// TIA Portal V17 export
// export: Created 2025-03-05T08:00:20.8649217Z, ExportSetting WithDefaults, DisplayName Totally Integrated Automation Portal, DisplayVersion V17 Update 8, DisplayName TIA Portal Openness, DisplayVersion V17 Update 8, DisplayName TIA Portal Version Control Interface, DisplayVersion V17, DisplayName SINAMICS Startdrive Advanced, DisplayVersion V17 SP2, DisplayName SINAMICS Startdrive G110M, G120, G120C, G120D, G120P, G115D, DisplayVersion V17 SP2, DisplayName SINAMICS Startdrive G130, G150, S120, S150, SINAMICS MV, S210, DisplayVersion V17 SP2, DisplayName STEP 7 Professional, DisplayVersion V17 Update 8, DisplayName SINUMERIK ONE STEP 7 Toolbox, DisplayVersion V17 Update 12, DisplayName SINUMERIK 840D sl STEP 7 Toolbox, DisplayVersion V17 Update 12, DisplayName STEP 7 Safety, DisplayVersion V17 Update 6, DisplayName WinCC Advanced, DisplayVersion V17 Update 8
FUNCTION "FC31_CLADDING_SPINDLES" : Void   // FC31, LAD
{ S7_Optimized_Access := 'FALSE' }
AUTHOR : ETXETAR
VERSION : 1.0
// stored: AutoNumber false, IsIECCheckEnabled false, SetENOAutomatically false, UDAEnableTagReadback false
   VAR_TEMP   // added for the SCL form of the ladder/FBD networks
      _w1 : Bool;
      _w2 : Bool;
   END_VAR
BEGIN

REGION Network 1: CALL FB31 SPINDLE C11
   // 2#0000_0001 OPTIONS 0 BIT 0 MEASURING SYSTEM 2 OPTION
   // 2#0000_0010 OPTIONS 0 BIT 1 BELT BROKEN OPTION
   // 2#0000_0100 OPTIONS 0 BIT 2 COOLING OPTION
   // 2#0000_1000 OPTIONS 0 BIT 3 MQL OR HP OPTION
   // 2#0001_0000 OPTIONS 0 BIT 4 ANALOG TEMPERATURE SENSOR OPTION
   // 2#0010_0000 OPTIONS 0 BIT 5 PTC TEMPERATURE SENSOR OPTION
   // 2#0100_0000 OPTIONS 0 BIT 6 TWIN KESSLER VPM READY OPTION
   // 2#1000_0000 OPTIONS 0 BIT 7 MPP SPINDLE OVERRIDE OPTION
   // 
   // 2#0000_0001 OPTIONS 1 BIT 0 SPARE OPTION
   // 2#0000_0010 OPTIONS 1 BIT 1 SPARE OPTION
   // 2#0000_0100 OPTIONS 1 BIT 2 SPARE OPTION
   // 2#0000_1000 OPTIONS 1 BIT 3 SPARE OPTION
   // 2#0001_0000 OPTIONS 1 BIT 4 SPARE OPTION
   // 2#0010_0000 OPTIONS 1 BIT 5 SPARE OPTION
   // 2#0100_0000 OPTIONS 1 BIT 6 SPARE OPTION
   // 2#1000_0000 OPTIONS 1 BIT 7 SPARE OPTION
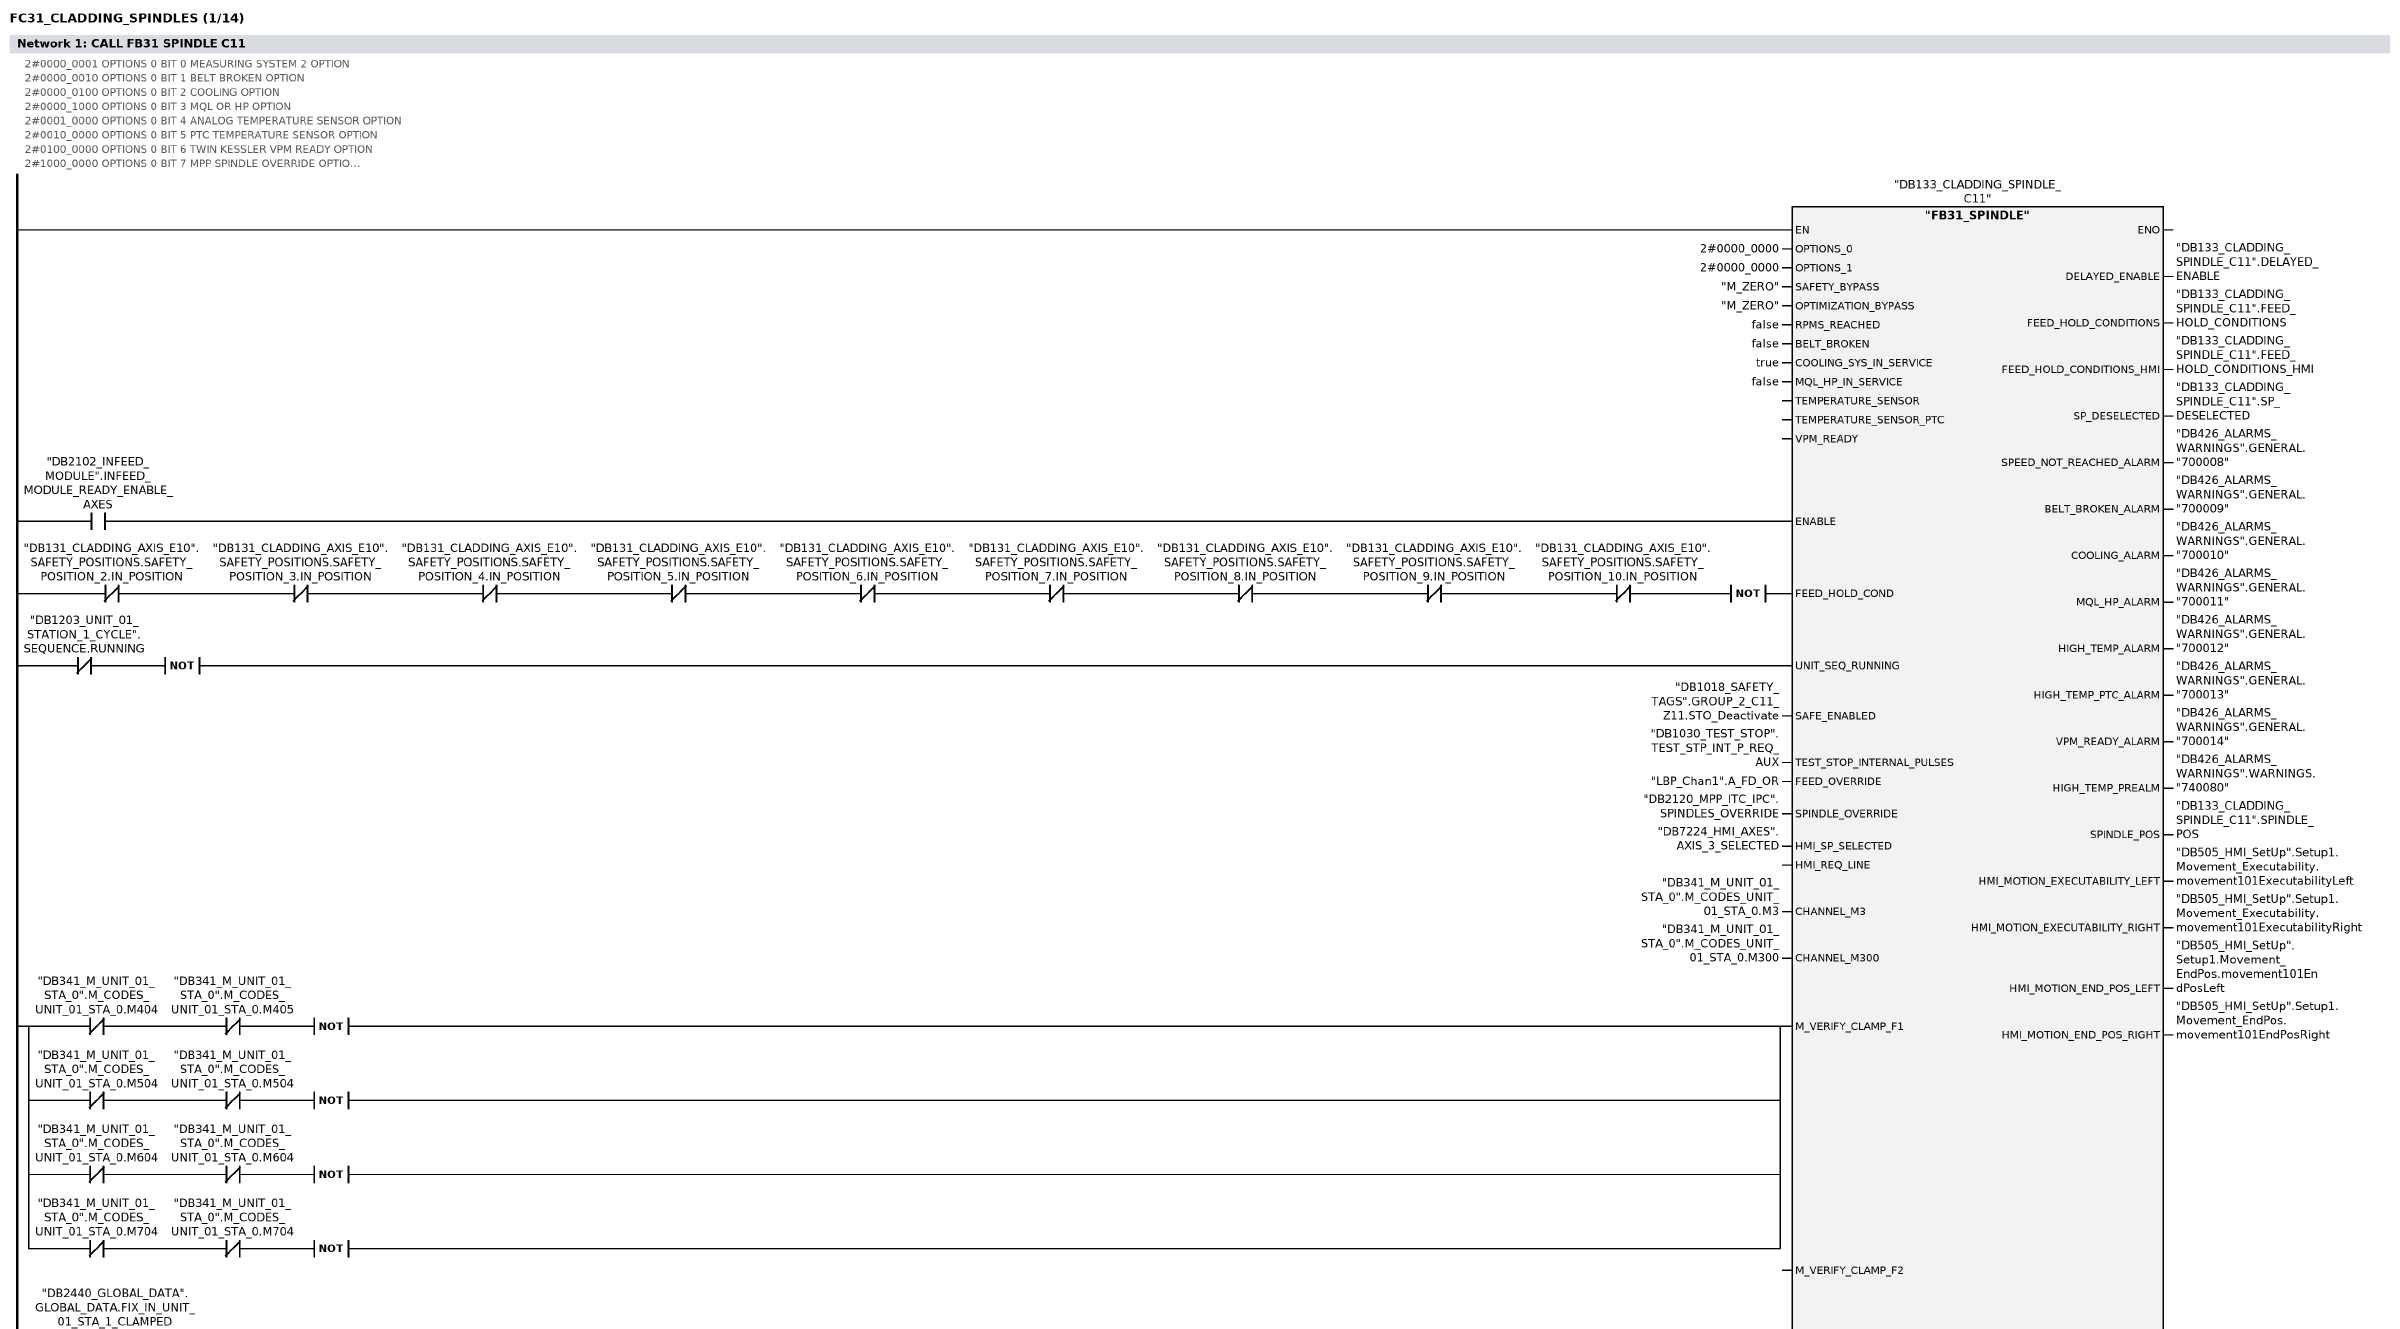
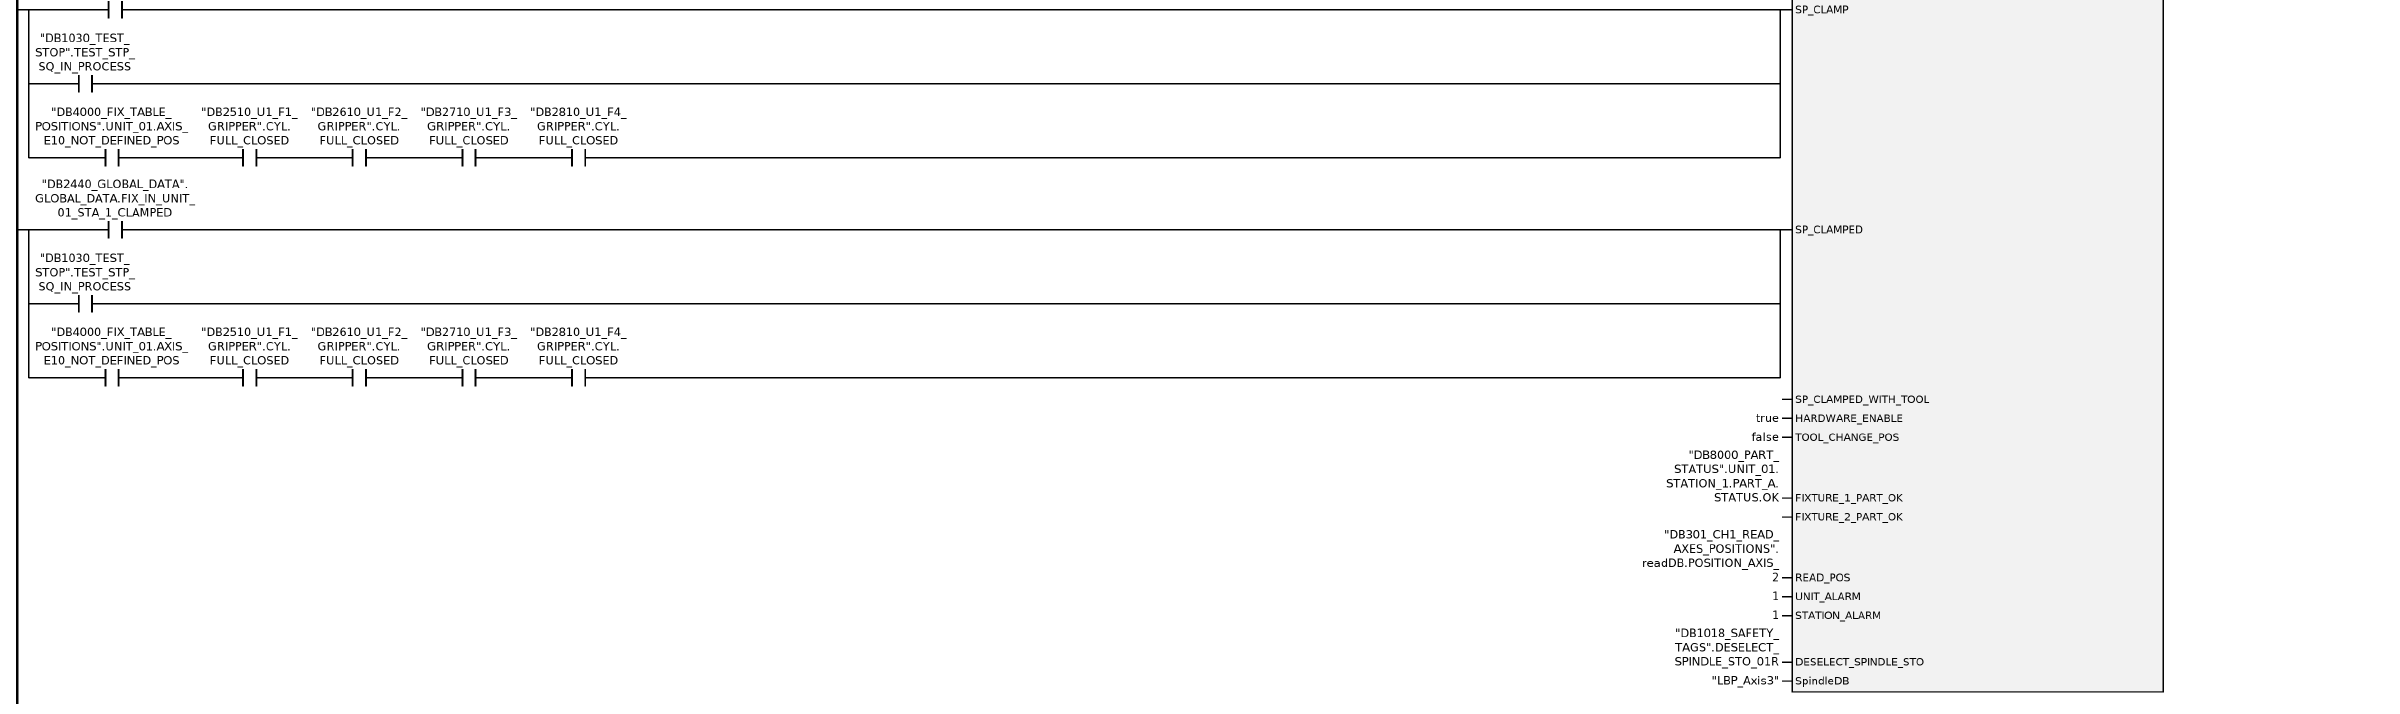
   RUNG wire#powerrail
      "DB133_CLADDING_SPINDLE_C11"(ENABLE := wire#w1, FEED_HOLD_COND := wire#w2, UNIT_SEQ_RUNNING := wire#w3, M_VERIFY_CLAMP_F1 := wire#w4, SP_CLAMP := wire#w5, SP_CLAMPED := wire#w6, OPTIONS_0 := 2#0000_0000, OPTIONS_1 := 2#0000_0000, SAFETY_BYPASS := "M_ZERO", OPTIMIZATION_BYPASS := "M_ZERO", RPMS_REACHED := false, BELT_BROKEN := false, COOLING_SYS_IN_SERVICE := true, MQL_HP_IN_SERVICE := false, TEMPERATURE_SENSOR :=, TEMPERATURE_SENSOR_PTC :=, VPM_READY :=, SAFE_ENABLED := "DB1018_SAFETY_TAGS".GROUP_2_C11_Z11.STO_Deactivate, TEST_STOP_INTERNAL_PULSES := "DB1030_TEST_STOP".TEST_STP_INT_P_REQ_AUX, FEED_OVERRIDE := "LBP_Chan1".A_FD_OR, SPINDLE_OVERRIDE := "DB2120_MPP_ITC_IPC".SPINDLES_OVERRIDE, HMI_SP_SELECTED := "DB7224_HMI_AXES".AXIS_3_SELECTED, HMI_REQ_LINE :=, CHANNEL_M3 := "DB341_M_UNIT_01_STA_0".M_CODES_UNIT_01_STA_0.M3, CHANNEL_M300 := "DB341_M_UNIT_01_STA_0".M_CODES_UNIT_01_STA_0.M300, M_VERIFY_CLAMP_F2 :=, SP_CLAMPED_WITH_TOOL :=, HARDWARE_ENABLE := true, TOOL_CHANGE_POS := false, FIXTURE_1_PART_OK := "DB8000_PART_STATUS".UNIT_01.STATION_1.PART_A.STATUS.OK, FIXTURE_2_PART_OK :=, READ_POS := "DB301_CH1_READ_AXES_POSITIONS".readDB.POSITION_AXIS_2, UNIT_ALARM := 1, STATION_ALARM := 1, DESELECT_SPINDLE_STO := "DB1018_SAFETY_TAGS".DESELECT_SPINDLE_STO_01R, SpindleDB := "LBP_Axis3", DELAYED_ENABLE => "DB133_CLADDING_SPINDLE_C11".DELAYED_ENABLE, FEED_HOLD_CONDITIONS => "DB133_CLADDING_SPINDLE_C11".FEED_HOLD_CONDITIONS, FEED_HOLD_CONDITIONS_HMI => "DB133_CLADDING_SPINDLE_C11".FEED_HOLD_CONDITIONS_HMI, SP_DESELECTED => "DB133_CLADDING_SPINDLE_C11".SP_DESELECTED, SPEED_NOT_REACHED_ALARM => "DB426_ALARMS_WARNINGS".GENERAL."700008", BELT_BROKEN_ALARM => "DB426_ALARMS_WARNINGS".GENERAL."700009", COOLING_ALARM => "DB426_ALARMS_WARNINGS".GENERAL."700010", MQL_HP_ALARM => "DB426_ALARMS_WARNINGS".GENERAL."700011", HIGH_TEMP_ALARM => "DB426_ALARMS_WARNINGS".GENERAL."700012", HIGH_TEMP_PTC_ALARM => "DB426_ALARMS_WARNINGS".GENERAL."700013", VPM_READY_ALARM => "DB426_ALARMS_WARNINGS".GENERAL."700014", HIGH_TEMP_PREALM => "DB426_ALARMS_WARNINGS".WARNINGS."740080", SPINDLE_POS => "DB133_CLADDING_SPINDLE_C11".SPINDLE_POS, HMI_MOTION_EXECUTABILITY_LEFT => "DB505_HMI_SetUp".Setup1.Movement_Executability.movement101ExecutabilityLeft, HMI_MOTION_EXECUTABILITY_RIGHT => "DB505_HMI_SetUp".Setup1.Movement_Executability.movement101ExecutabilityRight, HMI_MOTION_END_POS_LEFT => "DB505_HMI_SetUp".Setup1.Movement_EndPos.movement101EndPosLeft, HMI_MOTION_END_POS_RIGHT => "DB505_HMI_SetUp".Setup1.Movement_EndPos.movement101EndPosRight)
   END_RUNG
   RUNG wire#powerrail
      Contact( "DB2102_INFEED_MODULE".INFEED_MODULE_READY_ENABLE_AXES )
   END_RUNG wire#w1
   RUNG wire#powerrail
      I_Contact( "DB131_CLADDING_AXIS_E10".SAFETY_POSITIONS.SAFETY_POSITION_2.IN_POSITION )
      I_Contact( "DB131_CLADDING_AXIS_E10".SAFETY_POSITIONS.SAFETY_POSITION_3.IN_POSITION )
      I_Contact( "DB131_CLADDING_AXIS_E10".SAFETY_POSITIONS.SAFETY_POSITION_4.IN_POSITION )
      I_Contact( "DB131_CLADDING_AXIS_E10".SAFETY_POSITIONS.SAFETY_POSITION_5.IN_POSITION )
      I_Contact( "DB131_CLADDING_AXIS_E10".SAFETY_POSITIONS.SAFETY_POSITION_6.IN_POSITION )
      I_Contact( "DB131_CLADDING_AXIS_E10".SAFETY_POSITIONS.SAFETY_POSITION_7.IN_POSITION )
      I_Contact( "DB131_CLADDING_AXIS_E10".SAFETY_POSITIONS.SAFETY_POSITION_8.IN_POSITION )
      I_Contact( "DB131_CLADDING_AXIS_E10".SAFETY_POSITIONS.SAFETY_POSITION_9.IN_POSITION )
      I_Contact( "DB131_CLADDING_AXIS_E10".SAFETY_POSITIONS.SAFETY_POSITION_10.IN_POSITION )
      Not()
   END_RUNG wire#w2
   RUNG wire#powerrail
      I_Contact( "DB1203_UNIT_01_STATION_1_CYCLE".SEQUENCE.RUNNING )
      Not()
   END_RUNG wire#w3
   RUNG wire#powerrail
      I_Contact( "DB341_M_UNIT_01_STA_0".M_CODES_UNIT_01_STA_0.M404 )
      I_Contact( "DB341_M_UNIT_01_STA_0".M_CODES_UNIT_01_STA_0.M405 )
      Not()
   END_RUNG wire#w4
   RUNG wire#powerrail
      I_Contact( "DB341_M_UNIT_01_STA_0".M_CODES_UNIT_01_STA_0.M504 )
      I_Contact( "DB341_M_UNIT_01_STA_0".M_CODES_UNIT_01_STA_0.M504 )
      Not()
   END_RUNG wire#w4
   RUNG wire#powerrail
      I_Contact( "DB341_M_UNIT_01_STA_0".M_CODES_UNIT_01_STA_0.M604 )
      I_Contact( "DB341_M_UNIT_01_STA_0".M_CODES_UNIT_01_STA_0.M604 )
      Not()
   END_RUNG wire#w4
   RUNG wire#powerrail
      I_Contact( "DB341_M_UNIT_01_STA_0".M_CODES_UNIT_01_STA_0.M704 )
      I_Contact( "DB341_M_UNIT_01_STA_0".M_CODES_UNIT_01_STA_0.M704 )
      Not()
   END_RUNG wire#w4
   RUNG wire#powerrail
      Contact( "DB2440_GLOBAL_DATA".GLOBAL_DATA.FIX_IN_UNIT_01_STA_1_CLAMPED )
   END_RUNG wire#w5
   RUNG wire#powerrail
      Contact( "DB1030_TEST_STOP".TEST_STP_SQ_IN_PROCESS )
   END_RUNG wire#w5
   RUNG wire#powerrail
      Contact( "DB4000_FIX_TABLE_POSITIONS".UNIT_01.AXIS_E10_NOT_DEFINED_POS )
      Contact( "DB2510_U1_F1_GRIPPER".CYL.FULL_CLOSED )
      Contact( "DB2610_U1_F2_GRIPPER".CYL.FULL_CLOSED )
      Contact( "DB2710_U1_F3_GRIPPER".CYL.FULL_CLOSED )
      Contact( "DB2810_U1_F4_GRIPPER".CYL.FULL_CLOSED )
   END_RUNG wire#w5
   RUNG wire#powerrail
      Contact( "DB2440_GLOBAL_DATA".GLOBAL_DATA.FIX_IN_UNIT_01_STA_1_CLAMPED )
   END_RUNG wire#w6
   RUNG wire#powerrail
      Contact( "DB1030_TEST_STOP".TEST_STP_SQ_IN_PROCESS )
   END_RUNG wire#w6
   RUNG wire#powerrail
      Contact( "DB4000_FIX_TABLE_POSITIONS".UNIT_01.AXIS_E10_NOT_DEFINED_POS )
      Contact( "DB2510_U1_F1_GRIPPER".CYL.FULL_CLOSED )
      Contact( "DB2610_U1_F2_GRIPPER".CYL.FULL_CLOSED )
      Contact( "DB2710_U1_F3_GRIPPER".CYL.FULL_CLOSED )
      Contact( "DB2810_U1_F4_GRIPPER".CYL.FULL_CLOSED )
   END_RUNG wire#w6
   // the same network as SCL:
   "DB133_CLADDING_SPINDLE_C11"(OPTIONS_0 := 2#0000_0000,   // "FB31_SPINDLE"
                           OPTIONS_1 := 2#0000_0000,
                           SAFETY_BYPASS := "M_ZERO",
                           OPTIMIZATION_BYPASS := "M_ZERO",
                           RPMS_REACHED := false,
                           BELT_BROKEN := false,
                           COOLING_SYS_IN_SERVICE := true,
                           MQL_HP_IN_SERVICE := false,
                           ENABLE := "DB2102_INFEED_MODULE".INFEED_MODULE_READY_ENABLE_AXES,
                           FEED_HOLD_COND := NOT (NOT "DB131_CLADDING_AXIS_E10".SAFETY_POSITIONS.SAFETY_POSITION_2.IN_POSITION AND NOT "DB131_CLADDING_AXIS_E10".SAFETY_POSITIONS.SAFETY_POSITION_3.IN_POSITION AND NOT "DB131_CLADDING_AXIS_E10".SAFETY_POSITIONS.SAFETY_POSITION_4.IN_POSITION AND NOT "DB131_CLADDING_AXIS_E10".SAFETY_POSITIONS.SAFETY_POSITION_5.IN_POSITION AND NOT "DB131_CLADDING_AXIS_E10".SAFETY_POSITIONS.SAFETY_POSITION_6.IN_POSITION AND NOT "DB131_CLADDING_AXIS_E10".SAFETY_POSITIONS.SAFETY_POSITION_7.IN_POSITION AND NOT "DB131_CLADDING_AXIS_E10".SAFETY_POSITIONS.SAFETY_POSITION_8.IN_POSITION AND NOT "DB131_CLADDING_AXIS_E10".SAFETY_POSITIONS.SAFETY_POSITION_9.IN_POSITION AND NOT "DB131_CLADDING_AXIS_E10".SAFETY_POSITIONS.SAFETY_POSITION_10.IN_POSITION),
                           UNIT_SEQ_RUNNING := NOT (NOT "DB1203_UNIT_01_STATION_1_CYCLE".SEQUENCE.RUNNING),
                           SAFE_ENABLED := "DB1018_SAFETY_TAGS".GROUP_2_C11_Z11.STO_Deactivate,
                           TEST_STOP_INTERNAL_PULSES := "DB1030_TEST_STOP".TEST_STP_INT_P_REQ_AUX,
                           FEED_OVERRIDE := "LBP_Chan1".A_FD_OR,
                           SPINDLE_OVERRIDE := "DB2120_MPP_ITC_IPC".SPINDLES_OVERRIDE,
                           HMI_SP_SELECTED := "DB7224_HMI_AXES".AXIS_3_SELECTED,
                           CHANNEL_M3 := "DB341_M_UNIT_01_STA_0".M_CODES_UNIT_01_STA_0.M3,
                           CHANNEL_M300 := "DB341_M_UNIT_01_STA_0".M_CODES_UNIT_01_STA_0.M300,
                           M_VERIFY_CLAMP_F1 := NOT (NOT "DB341_M_UNIT_01_STA_0".M_CODES_UNIT_01_STA_0.M404 AND NOT "DB341_M_UNIT_01_STA_0".M_CODES_UNIT_01_STA_0.M405) OR NOT (NOT "DB341_M_UNIT_01_STA_0".M_CODES_UNIT_01_STA_0.M504 AND NOT "DB341_M_UNIT_01_STA_0".M_CODES_UNIT_01_STA_0.M504) OR NOT (NOT "DB341_M_UNIT_01_STA_0".M_CODES_UNIT_01_STA_0.M604 AND NOT "DB341_M_UNIT_01_STA_0".M_CODES_UNIT_01_STA_0.M604) OR NOT (NOT "DB341_M_UNIT_01_STA_0".M_CODES_UNIT_01_STA_0.M704 AND NOT "DB341_M_UNIT_01_STA_0".M_CODES_UNIT_01_STA_0.M704),
                           SP_CLAMP := "DB2440_GLOBAL_DATA".GLOBAL_DATA.FIX_IN_UNIT_01_STA_1_CLAMPED OR "DB1030_TEST_STOP".TEST_STP_SQ_IN_PROCESS OR ("DB4000_FIX_TABLE_POSITIONS".UNIT_01.AXIS_E10_NOT_DEFINED_POS AND "DB2510_U1_F1_GRIPPER".CYL.FULL_CLOSED AND "DB2610_U1_F2_GRIPPER".CYL.FULL_CLOSED AND "DB2710_U1_F3_GRIPPER".CYL.FULL_CLOSED AND "DB2810_U1_F4_GRIPPER".CYL.FULL_CLOSED),
                           SP_CLAMPED := "DB2440_GLOBAL_DATA".GLOBAL_DATA.FIX_IN_UNIT_01_STA_1_CLAMPED OR "DB1030_TEST_STOP".TEST_STP_SQ_IN_PROCESS OR ("DB4000_FIX_TABLE_POSITIONS".UNIT_01.AXIS_E10_NOT_DEFINED_POS AND "DB2510_U1_F1_GRIPPER".CYL.FULL_CLOSED AND "DB2610_U1_F2_GRIPPER".CYL.FULL_CLOSED AND "DB2710_U1_F3_GRIPPER".CYL.FULL_CLOSED AND "DB2810_U1_F4_GRIPPER".CYL.FULL_CLOSED),
                           HARDWARE_ENABLE := true,
                           TOOL_CHANGE_POS := false,
                           FIXTURE_1_PART_OK := "DB8000_PART_STATUS".UNIT_01.STATION_1.PART_A.STATUS.OK,
                           READ_POS := "DB301_CH1_READ_AXES_POSITIONS".readDB.POSITION_AXIS_2,
                           UNIT_ALARM := 1,
                           STATION_ALARM := 1,
                           DESELECT_SPINDLE_STO := "DB1018_SAFETY_TAGS".DESELECT_SPINDLE_STO_01R,
                           SpindleDB := "LBP_Axis3",
                           DELAYED_ENABLE => "DB133_CLADDING_SPINDLE_C11".DELAYED_ENABLE,
                           FEED_HOLD_CONDITIONS => "DB133_CLADDING_SPINDLE_C11".FEED_HOLD_CONDITIONS,
                           FEED_HOLD_CONDITIONS_HMI => "DB133_CLADDING_SPINDLE_C11".FEED_HOLD_CONDITIONS_HMI,
                           SP_DESELECTED => "DB133_CLADDING_SPINDLE_C11".SP_DESELECTED,
                           SPEED_NOT_REACHED_ALARM => "DB426_ALARMS_WARNINGS".GENERAL."700008",
                           BELT_BROKEN_ALARM => "DB426_ALARMS_WARNINGS".GENERAL."700009",
                           COOLING_ALARM => "DB426_ALARMS_WARNINGS".GENERAL."700010",
                           MQL_HP_ALARM => "DB426_ALARMS_WARNINGS".GENERAL."700011",
                           HIGH_TEMP_ALARM => "DB426_ALARMS_WARNINGS".GENERAL."700012",
                           HIGH_TEMP_PTC_ALARM => "DB426_ALARMS_WARNINGS".GENERAL."700013",
                           VPM_READY_ALARM => "DB426_ALARMS_WARNINGS".GENERAL."700014",
                           HIGH_TEMP_PREALM => "DB426_ALARMS_WARNINGS".WARNINGS."740080",
                           SPINDLE_POS => "DB133_CLADDING_SPINDLE_C11".SPINDLE_POS,
                           HMI_MOTION_EXECUTABILITY_LEFT => "DB505_HMI_SetUp".Setup1.Movement_Executability.movement101ExecutabilityLeft,
                           HMI_MOTION_EXECUTABILITY_RIGHT => "DB505_HMI_SetUp".Setup1.Movement_Executability.movement101ExecutabilityRight,
                           HMI_MOTION_END_POS_LEFT => "DB505_HMI_SetUp".Setup1.Movement_EndPos.movement101EndPosLeft,
                           HMI_MOTION_END_POS_RIGHT => "DB505_HMI_SetUp".Setup1.Movement_EndPos.movement101EndPosRight);
END_REGION

REGION Network 2: SPINDLE C11 OPERATOR HELP
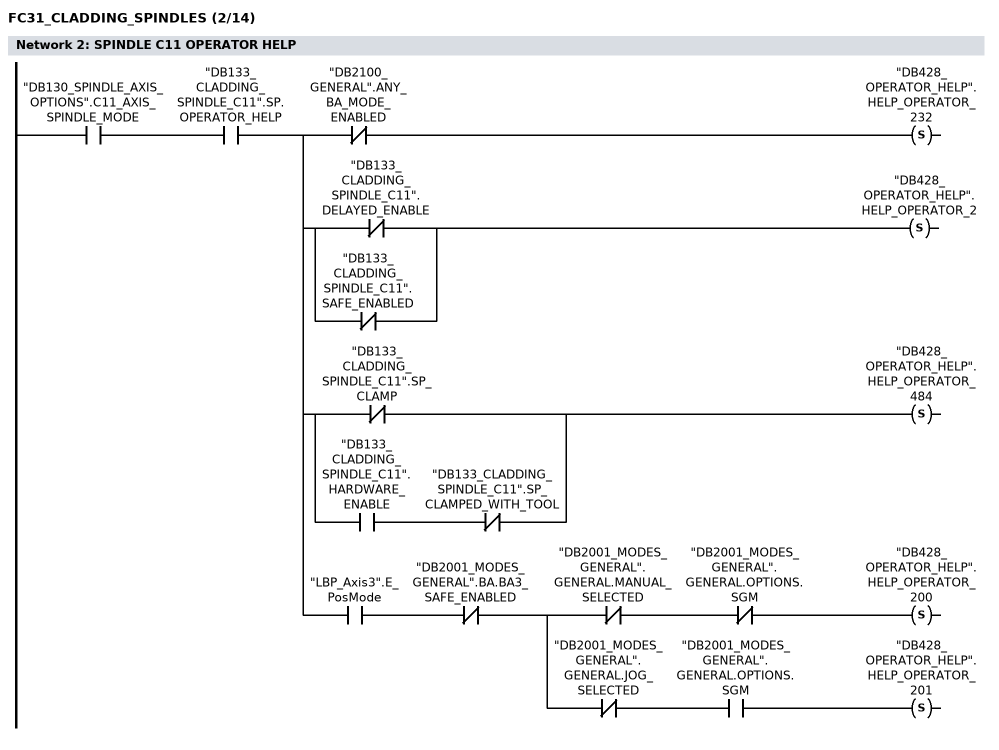
   RUNG wire#powerrail
      Contact( "DB130_SPINDLE_AXIS_OPTIONS".C11_AXIS_SPINDLE_MODE )
      Contact( "DB133_CLADDING_SPINDLE_C11".SP.OPERATOR_HELP )
      wire#w1
      I_Contact( "DB2100_GENERAL".ANY_BA_MODE_ENABLED )
      S_Coil( "DB428_OPERATOR_HELP".HELP_OPERATOR_232 )
   END_RUNG
   RUNG wire#w1
      I_Contact( "DB133_CLADDING_SPINDLE_C11".DELAYED_ENABLE )
      wire#w2
      S_Coil( "DB428_OPERATOR_HELP".HELP_OPERATOR_2 )
   END_RUNG
   RUNG wire#w1
      I_Contact( "DB133_CLADDING_SPINDLE_C11".SAFE_ENABLED )
   END_RUNG wire#w2
   RUNG wire#w1
      I_Contact( "DB133_CLADDING_SPINDLE_C11".SP_CLAMP )
      wire#w3
      S_Coil( "DB428_OPERATOR_HELP".HELP_OPERATOR_484 )
   END_RUNG
   RUNG wire#w1
      Contact( "DB133_CLADDING_SPINDLE_C11".HARDWARE_ENABLE )
      I_Contact( "DB133_CLADDING_SPINDLE_C11".SP_CLAMPED_WITH_TOOL )
   END_RUNG wire#w3
   RUNG wire#w1
      Contact( "LBP_Axis3".E_PosMode )
      I_Contact( "DB2001_MODES_GENERAL".BA.BA3_SAFE_ENABLED )
      wire#w4
      I_Contact( "DB2001_MODES_GENERAL".GENERAL.MANUAL_SELECTED )
      I_Contact( "DB2001_MODES_GENERAL".GENERAL.OPTIONS.SGM )
      S_Coil( "DB428_OPERATOR_HELP".HELP_OPERATOR_200 )
   END_RUNG
   RUNG wire#w4
      I_Contact( "DB2001_MODES_GENERAL".GENERAL.JOG_SELECTED )
      Contact( "DB2001_MODES_GENERAL".GENERAL.OPTIONS.SGM )
      S_Coil( "DB428_OPERATOR_HELP".HELP_OPERATOR_201 )
   END_RUNG
   // the same network as SCL:
   #_w1 := "DB130_SPINDLE_AXIS_OPTIONS".C11_AXIS_SPINDLE_MODE AND "DB133_CLADDING_SPINDLE_C11".SP.OPERATOR_HELP;
   IF #_w1 AND NOT "DB2100_GENERAL".ANY_BA_MODE_ENABLED THEN
       "DB428_OPERATOR_HELP".HELP_OPERATOR_232 := TRUE;
   END_IF;
   IF #_w1 AND (NOT "DB133_CLADDING_SPINDLE_C11".DELAYED_ENABLE OR NOT "DB133_CLADDING_SPINDLE_C11".SAFE_ENABLED) THEN
       "DB428_OPERATOR_HELP".HELP_OPERATOR_2 := TRUE;
   END_IF;
   IF #_w1 AND (NOT "DB133_CLADDING_SPINDLE_C11".SP_CLAMP OR ("DB133_CLADDING_SPINDLE_C11".HARDWARE_ENABLE AND NOT "DB133_CLADDING_SPINDLE_C11".SP_CLAMPED_WITH_TOOL)) THEN
       "DB428_OPERATOR_HELP".HELP_OPERATOR_484 := TRUE;
   END_IF;
   #_w2 := #_w1 AND "LBP_Axis3".E_PosMode AND NOT "DB2001_MODES_GENERAL".BA.BA3_SAFE_ENABLED;
   IF #_w2 AND NOT "DB2001_MODES_GENERAL".GENERAL.MANUAL_SELECTED AND NOT "DB2001_MODES_GENERAL".GENERAL.OPTIONS.SGM THEN
       "DB428_OPERATOR_HELP".HELP_OPERATOR_200 := TRUE;
   END_IF;
   IF #_w2 AND NOT "DB2001_MODES_GENERAL".GENERAL.JOG_SELECTED AND "DB2001_MODES_GENERAL".GENERAL.OPTIONS.SGM THEN
       "DB428_OPERATOR_HELP".HELP_OPERATOR_201 := TRUE;
   END_IF;
END_REGION

REGION Network 3: CALL FB31 SPINDLE C12
   // 2#0000_0001 OPTIONS 0 BIT 0 MEASURING SYSTEM 2 OPTION
   // 2#0000_0010 OPTIONS 0 BIT 1 BELT BROKEN OPTION
   // 2#0000_0100 OPTIONS 0 BIT 2 COOLING OPTION
   // 2#0000_1000 OPTIONS 0 BIT 3 MQL OR HP OPTION
   // 2#0001_0000 OPTIONS 0 BIT 4 ANALOG TEMPERATURE SENSOR OPTION
   // 2#0010_0000 OPTIONS 0 BIT 5 PTC TEMPERATURE SENSOR OPTION
   // 2#0100_0000 OPTIONS 0 BIT 6 TWIN KESSLER VPM READY OPTION
   // 2#1000_0000 OPTIONS 0 BIT 7 MPP SPINDLE OVERRIDE OPTION
   // 
   // 2#0000_0001 OPTIONS 1 BIT 0 SPARE OPTION
   // 2#0000_0010 OPTIONS 1 BIT 1 SPARE OPTION
   // 2#0000_0100 OPTIONS 1 BIT 2 SPARE OPTION
   // 2#0000_1000 OPTIONS 1 BIT 3 SPARE OPTION
   // 2#0001_0000 OPTIONS 1 BIT 4 SPARE OPTION
   // 2#0010_0000 OPTIONS 1 BIT 5 SPARE OPTION
   // 2#0100_0000 OPTIONS 1 BIT 6 SPARE OPTION
   // 2#1000_0000 OPTIONS 1 BIT 7 SPARE OPTION
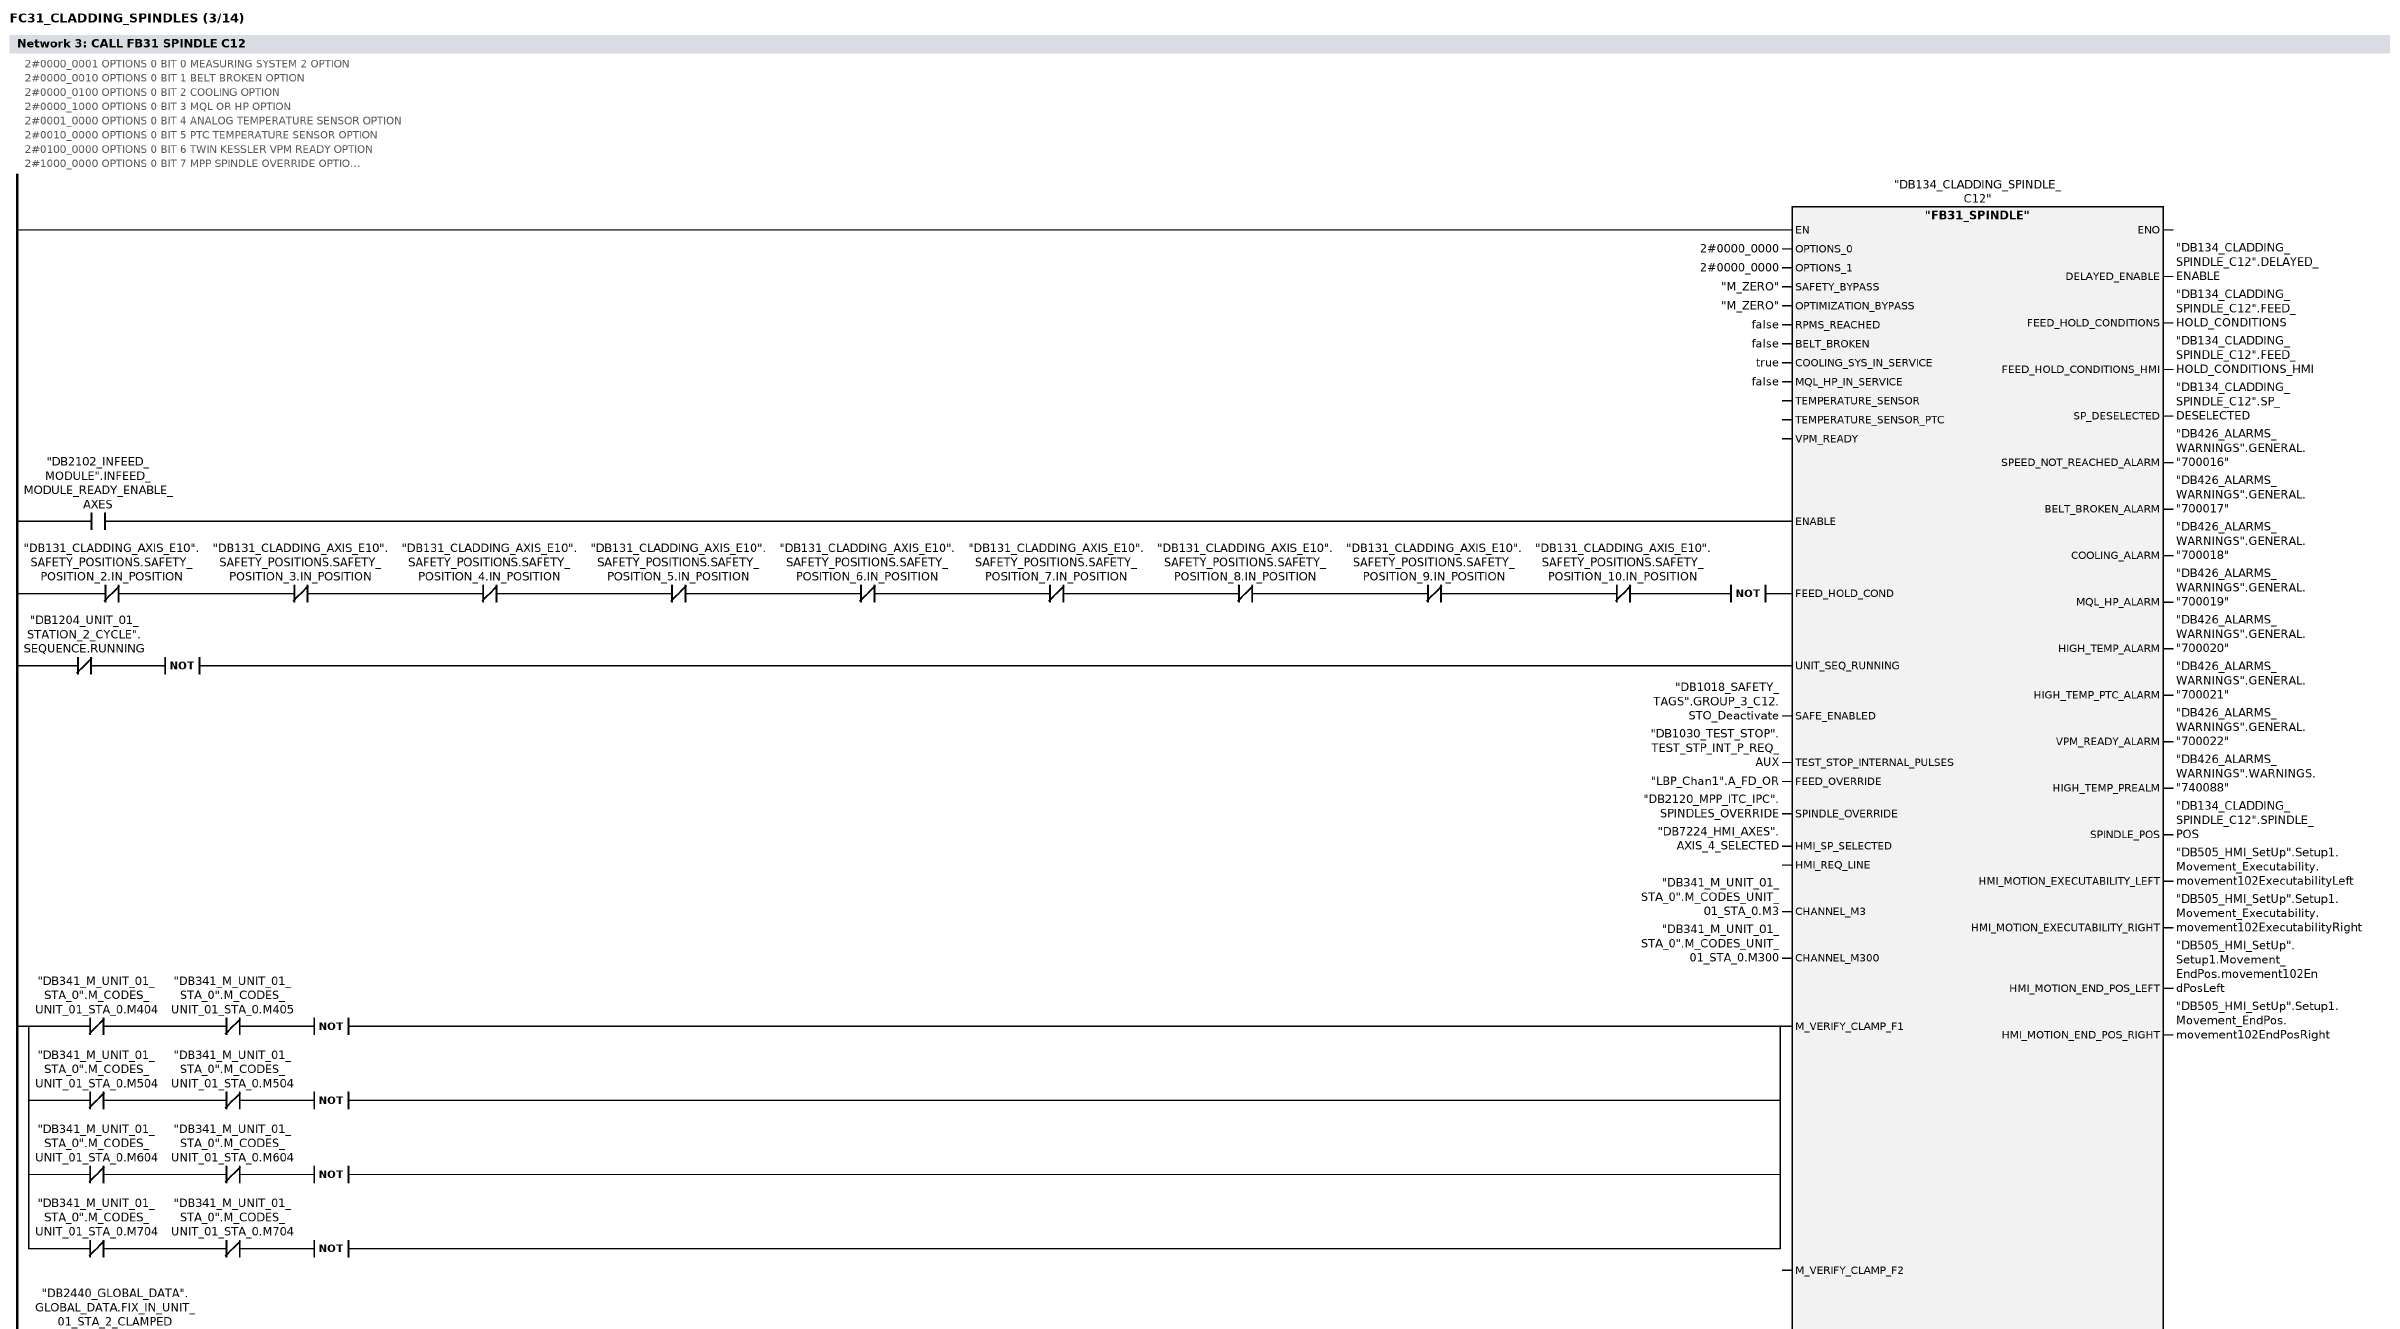
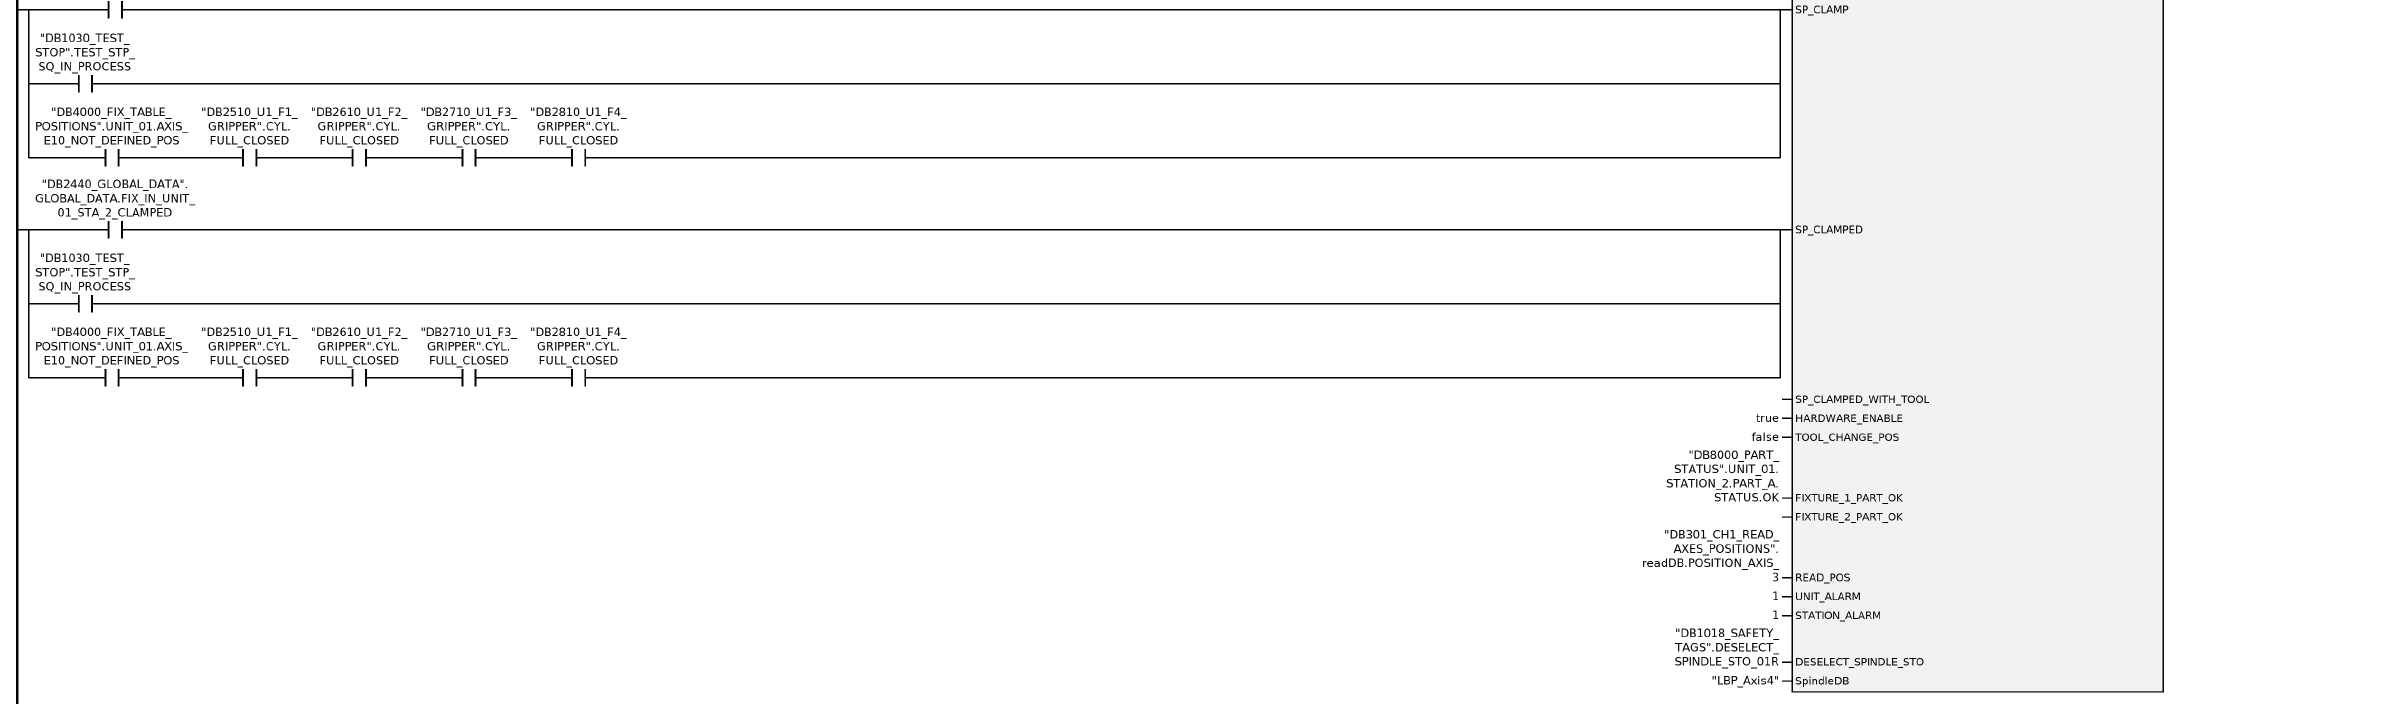
   RUNG wire#powerrail
      "DB134_CLADDING_SPINDLE_C12"(ENABLE := wire#w1, FEED_HOLD_COND := wire#w2, UNIT_SEQ_RUNNING := wire#w3, M_VERIFY_CLAMP_F1 := wire#w4, SP_CLAMP := wire#w5, SP_CLAMPED := wire#w6, OPTIONS_0 := 2#0000_0000, OPTIONS_1 := 2#0000_0000, SAFETY_BYPASS := "M_ZERO", OPTIMIZATION_BYPASS := "M_ZERO", RPMS_REACHED := false, BELT_BROKEN := false, COOLING_SYS_IN_SERVICE := true, MQL_HP_IN_SERVICE := false, TEMPERATURE_SENSOR :=, TEMPERATURE_SENSOR_PTC :=, VPM_READY :=, SAFE_ENABLED := "DB1018_SAFETY_TAGS".GROUP_3_C12.STO_Deactivate, TEST_STOP_INTERNAL_PULSES := "DB1030_TEST_STOP".TEST_STP_INT_P_REQ_AUX, FEED_OVERRIDE := "LBP_Chan1".A_FD_OR, SPINDLE_OVERRIDE := "DB2120_MPP_ITC_IPC".SPINDLES_OVERRIDE, HMI_SP_SELECTED := "DB7224_HMI_AXES".AXIS_4_SELECTED, HMI_REQ_LINE :=, CHANNEL_M3 := "DB341_M_UNIT_01_STA_0".M_CODES_UNIT_01_STA_0.M3, CHANNEL_M300 := "DB341_M_UNIT_01_STA_0".M_CODES_UNIT_01_STA_0.M300, M_VERIFY_CLAMP_F2 :=, SP_CLAMPED_WITH_TOOL :=, HARDWARE_ENABLE := true, TOOL_CHANGE_POS := false, FIXTURE_1_PART_OK := "DB8000_PART_STATUS".UNIT_01.STATION_2.PART_A.STATUS.OK, FIXTURE_2_PART_OK :=, READ_POS := "DB301_CH1_READ_AXES_POSITIONS".readDB.POSITION_AXIS_3, UNIT_ALARM := 1, STATION_ALARM := 1, DESELECT_SPINDLE_STO := "DB1018_SAFETY_TAGS".DESELECT_SPINDLE_STO_01R, SpindleDB := "LBP_Axis4", DELAYED_ENABLE => "DB134_CLADDING_SPINDLE_C12".DELAYED_ENABLE, FEED_HOLD_CONDITIONS => "DB134_CLADDING_SPINDLE_C12".FEED_HOLD_CONDITIONS, FEED_HOLD_CONDITIONS_HMI => "DB134_CLADDING_SPINDLE_C12".FEED_HOLD_CONDITIONS_HMI, SP_DESELECTED => "DB134_CLADDING_SPINDLE_C12".SP_DESELECTED, SPEED_NOT_REACHED_ALARM => "DB426_ALARMS_WARNINGS".GENERAL."700016", BELT_BROKEN_ALARM => "DB426_ALARMS_WARNINGS".GENERAL."700017", COOLING_ALARM => "DB426_ALARMS_WARNINGS".GENERAL."700018", MQL_HP_ALARM => "DB426_ALARMS_WARNINGS".GENERAL."700019", HIGH_TEMP_ALARM => "DB426_ALARMS_WARNINGS".GENERAL."700020", HIGH_TEMP_PTC_ALARM => "DB426_ALARMS_WARNINGS".GENERAL."700021", VPM_READY_ALARM => "DB426_ALARMS_WARNINGS".GENERAL."700022", HIGH_TEMP_PREALM => "DB426_ALARMS_WARNINGS".WARNINGS."740088", SPINDLE_POS => "DB134_CLADDING_SPINDLE_C12".SPINDLE_POS, HMI_MOTION_EXECUTABILITY_LEFT => "DB505_HMI_SetUp".Setup1.Movement_Executability.movement102ExecutabilityLeft, HMI_MOTION_EXECUTABILITY_RIGHT => "DB505_HMI_SetUp".Setup1.Movement_Executability.movement102ExecutabilityRight, HMI_MOTION_END_POS_LEFT => "DB505_HMI_SetUp".Setup1.Movement_EndPos.movement102EndPosLeft, HMI_MOTION_END_POS_RIGHT => "DB505_HMI_SetUp".Setup1.Movement_EndPos.movement102EndPosRight)
   END_RUNG
   RUNG wire#powerrail
      Contact( "DB2102_INFEED_MODULE".INFEED_MODULE_READY_ENABLE_AXES )
   END_RUNG wire#w1
   RUNG wire#powerrail
      I_Contact( "DB131_CLADDING_AXIS_E10".SAFETY_POSITIONS.SAFETY_POSITION_2.IN_POSITION )
      I_Contact( "DB131_CLADDING_AXIS_E10".SAFETY_POSITIONS.SAFETY_POSITION_3.IN_POSITION )
      I_Contact( "DB131_CLADDING_AXIS_E10".SAFETY_POSITIONS.SAFETY_POSITION_4.IN_POSITION )
      I_Contact( "DB131_CLADDING_AXIS_E10".SAFETY_POSITIONS.SAFETY_POSITION_5.IN_POSITION )
      I_Contact( "DB131_CLADDING_AXIS_E10".SAFETY_POSITIONS.SAFETY_POSITION_6.IN_POSITION )
      I_Contact( "DB131_CLADDING_AXIS_E10".SAFETY_POSITIONS.SAFETY_POSITION_7.IN_POSITION )
      I_Contact( "DB131_CLADDING_AXIS_E10".SAFETY_POSITIONS.SAFETY_POSITION_8.IN_POSITION )
      I_Contact( "DB131_CLADDING_AXIS_E10".SAFETY_POSITIONS.SAFETY_POSITION_9.IN_POSITION )
      I_Contact( "DB131_CLADDING_AXIS_E10".SAFETY_POSITIONS.SAFETY_POSITION_10.IN_POSITION )
      Not()
   END_RUNG wire#w2
   RUNG wire#powerrail
      I_Contact( "DB1204_UNIT_01_STATION_2_CYCLE".SEQUENCE.RUNNING )
      Not()
   END_RUNG wire#w3
   RUNG wire#powerrail
      I_Contact( "DB341_M_UNIT_01_STA_0".M_CODES_UNIT_01_STA_0.M404 )
      I_Contact( "DB341_M_UNIT_01_STA_0".M_CODES_UNIT_01_STA_0.M405 )
      Not()
   END_RUNG wire#w4
   RUNG wire#powerrail
      I_Contact( "DB341_M_UNIT_01_STA_0".M_CODES_UNIT_01_STA_0.M504 )
      I_Contact( "DB341_M_UNIT_01_STA_0".M_CODES_UNIT_01_STA_0.M504 )
      Not()
   END_RUNG wire#w4
   RUNG wire#powerrail
      I_Contact( "DB341_M_UNIT_01_STA_0".M_CODES_UNIT_01_STA_0.M604 )
      I_Contact( "DB341_M_UNIT_01_STA_0".M_CODES_UNIT_01_STA_0.M604 )
      Not()
   END_RUNG wire#w4
   RUNG wire#powerrail
      I_Contact( "DB341_M_UNIT_01_STA_0".M_CODES_UNIT_01_STA_0.M704 )
      I_Contact( "DB341_M_UNIT_01_STA_0".M_CODES_UNIT_01_STA_0.M704 )
      Not()
   END_RUNG wire#w4
   RUNG wire#powerrail
      Contact( "DB2440_GLOBAL_DATA".GLOBAL_DATA.FIX_IN_UNIT_01_STA_2_CLAMPED )
   END_RUNG wire#w5
   RUNG wire#powerrail
      Contact( "DB1030_TEST_STOP".TEST_STP_SQ_IN_PROCESS )
   END_RUNG wire#w5
   RUNG wire#powerrail
      Contact( "DB4000_FIX_TABLE_POSITIONS".UNIT_01.AXIS_E10_NOT_DEFINED_POS )
      Contact( "DB2510_U1_F1_GRIPPER".CYL.FULL_CLOSED )
      Contact( "DB2610_U1_F2_GRIPPER".CYL.FULL_CLOSED )
      Contact( "DB2710_U1_F3_GRIPPER".CYL.FULL_CLOSED )
      Contact( "DB2810_U1_F4_GRIPPER".CYL.FULL_CLOSED )
   END_RUNG wire#w5
   RUNG wire#powerrail
      Contact( "DB2440_GLOBAL_DATA".GLOBAL_DATA.FIX_IN_UNIT_01_STA_2_CLAMPED )
   END_RUNG wire#w6
   RUNG wire#powerrail
      Contact( "DB1030_TEST_STOP".TEST_STP_SQ_IN_PROCESS )
   END_RUNG wire#w6
   RUNG wire#powerrail
      Contact( "DB4000_FIX_TABLE_POSITIONS".UNIT_01.AXIS_E10_NOT_DEFINED_POS )
      Contact( "DB2510_U1_F1_GRIPPER".CYL.FULL_CLOSED )
      Contact( "DB2610_U1_F2_GRIPPER".CYL.FULL_CLOSED )
      Contact( "DB2710_U1_F3_GRIPPER".CYL.FULL_CLOSED )
      Contact( "DB2810_U1_F4_GRIPPER".CYL.FULL_CLOSED )
   END_RUNG wire#w6
   // the same network as SCL:
   "DB134_CLADDING_SPINDLE_C12"(OPTIONS_0 := 2#0000_0000,   // "FB31_SPINDLE"
                           OPTIONS_1 := 2#0000_0000,
                           SAFETY_BYPASS := "M_ZERO",
                           OPTIMIZATION_BYPASS := "M_ZERO",
                           RPMS_REACHED := false,
                           BELT_BROKEN := false,
                           COOLING_SYS_IN_SERVICE := true,
                           MQL_HP_IN_SERVICE := false,
                           ENABLE := "DB2102_INFEED_MODULE".INFEED_MODULE_READY_ENABLE_AXES,
                           FEED_HOLD_COND := NOT (NOT "DB131_CLADDING_AXIS_E10".SAFETY_POSITIONS.SAFETY_POSITION_2.IN_POSITION AND NOT "DB131_CLADDING_AXIS_E10".SAFETY_POSITIONS.SAFETY_POSITION_3.IN_POSITION AND NOT "DB131_CLADDING_AXIS_E10".SAFETY_POSITIONS.SAFETY_POSITION_4.IN_POSITION AND NOT "DB131_CLADDING_AXIS_E10".SAFETY_POSITIONS.SAFETY_POSITION_5.IN_POSITION AND NOT "DB131_CLADDING_AXIS_E10".SAFETY_POSITIONS.SAFETY_POSITION_6.IN_POSITION AND NOT "DB131_CLADDING_AXIS_E10".SAFETY_POSITIONS.SAFETY_POSITION_7.IN_POSITION AND NOT "DB131_CLADDING_AXIS_E10".SAFETY_POSITIONS.SAFETY_POSITION_8.IN_POSITION AND NOT "DB131_CLADDING_AXIS_E10".SAFETY_POSITIONS.SAFETY_POSITION_9.IN_POSITION AND NOT "DB131_CLADDING_AXIS_E10".SAFETY_POSITIONS.SAFETY_POSITION_10.IN_POSITION),
                           UNIT_SEQ_RUNNING := NOT (NOT "DB1204_UNIT_01_STATION_2_CYCLE".SEQUENCE.RUNNING),
                           SAFE_ENABLED := "DB1018_SAFETY_TAGS".GROUP_3_C12.STO_Deactivate,
                           TEST_STOP_INTERNAL_PULSES := "DB1030_TEST_STOP".TEST_STP_INT_P_REQ_AUX,
                           FEED_OVERRIDE := "LBP_Chan1".A_FD_OR,
                           SPINDLE_OVERRIDE := "DB2120_MPP_ITC_IPC".SPINDLES_OVERRIDE,
                           HMI_SP_SELECTED := "DB7224_HMI_AXES".AXIS_4_SELECTED,
                           CHANNEL_M3 := "DB341_M_UNIT_01_STA_0".M_CODES_UNIT_01_STA_0.M3,
                           CHANNEL_M300 := "DB341_M_UNIT_01_STA_0".M_CODES_UNIT_01_STA_0.M300,
                           M_VERIFY_CLAMP_F1 := NOT (NOT "DB341_M_UNIT_01_STA_0".M_CODES_UNIT_01_STA_0.M404 AND NOT "DB341_M_UNIT_01_STA_0".M_CODES_UNIT_01_STA_0.M405) OR NOT (NOT "DB341_M_UNIT_01_STA_0".M_CODES_UNIT_01_STA_0.M504 AND NOT "DB341_M_UNIT_01_STA_0".M_CODES_UNIT_01_STA_0.M504) OR NOT (NOT "DB341_M_UNIT_01_STA_0".M_CODES_UNIT_01_STA_0.M604 AND NOT "DB341_M_UNIT_01_STA_0".M_CODES_UNIT_01_STA_0.M604) OR NOT (NOT "DB341_M_UNIT_01_STA_0".M_CODES_UNIT_01_STA_0.M704 AND NOT "DB341_M_UNIT_01_STA_0".M_CODES_UNIT_01_STA_0.M704),
                           SP_CLAMP := "DB2440_GLOBAL_DATA".GLOBAL_DATA.FIX_IN_UNIT_01_STA_2_CLAMPED OR "DB1030_TEST_STOP".TEST_STP_SQ_IN_PROCESS OR ("DB4000_FIX_TABLE_POSITIONS".UNIT_01.AXIS_E10_NOT_DEFINED_POS AND "DB2510_U1_F1_GRIPPER".CYL.FULL_CLOSED AND "DB2610_U1_F2_GRIPPER".CYL.FULL_CLOSED AND "DB2710_U1_F3_GRIPPER".CYL.FULL_CLOSED AND "DB2810_U1_F4_GRIPPER".CYL.FULL_CLOSED),
                           SP_CLAMPED := "DB2440_GLOBAL_DATA".GLOBAL_DATA.FIX_IN_UNIT_01_STA_2_CLAMPED OR "DB1030_TEST_STOP".TEST_STP_SQ_IN_PROCESS OR ("DB4000_FIX_TABLE_POSITIONS".UNIT_01.AXIS_E10_NOT_DEFINED_POS AND "DB2510_U1_F1_GRIPPER".CYL.FULL_CLOSED AND "DB2610_U1_F2_GRIPPER".CYL.FULL_CLOSED AND "DB2710_U1_F3_GRIPPER".CYL.FULL_CLOSED AND "DB2810_U1_F4_GRIPPER".CYL.FULL_CLOSED),
                           HARDWARE_ENABLE := true,
                           TOOL_CHANGE_POS := false,
                           FIXTURE_1_PART_OK := "DB8000_PART_STATUS".UNIT_01.STATION_2.PART_A.STATUS.OK,
                           READ_POS := "DB301_CH1_READ_AXES_POSITIONS".readDB.POSITION_AXIS_3,
                           UNIT_ALARM := 1,
                           STATION_ALARM := 1,
                           DESELECT_SPINDLE_STO := "DB1018_SAFETY_TAGS".DESELECT_SPINDLE_STO_01R,
                           SpindleDB := "LBP_Axis4",
                           DELAYED_ENABLE => "DB134_CLADDING_SPINDLE_C12".DELAYED_ENABLE,
                           FEED_HOLD_CONDITIONS => "DB134_CLADDING_SPINDLE_C12".FEED_HOLD_CONDITIONS,
                           FEED_HOLD_CONDITIONS_HMI => "DB134_CLADDING_SPINDLE_C12".FEED_HOLD_CONDITIONS_HMI,
                           SP_DESELECTED => "DB134_CLADDING_SPINDLE_C12".SP_DESELECTED,
                           SPEED_NOT_REACHED_ALARM => "DB426_ALARMS_WARNINGS".GENERAL."700016",
                           BELT_BROKEN_ALARM => "DB426_ALARMS_WARNINGS".GENERAL."700017",
                           COOLING_ALARM => "DB426_ALARMS_WARNINGS".GENERAL."700018",
                           MQL_HP_ALARM => "DB426_ALARMS_WARNINGS".GENERAL."700019",
                           HIGH_TEMP_ALARM => "DB426_ALARMS_WARNINGS".GENERAL."700020",
                           HIGH_TEMP_PTC_ALARM => "DB426_ALARMS_WARNINGS".GENERAL."700021",
                           VPM_READY_ALARM => "DB426_ALARMS_WARNINGS".GENERAL."700022",
                           HIGH_TEMP_PREALM => "DB426_ALARMS_WARNINGS".WARNINGS."740088",
                           SPINDLE_POS => "DB134_CLADDING_SPINDLE_C12".SPINDLE_POS,
                           HMI_MOTION_EXECUTABILITY_LEFT => "DB505_HMI_SetUp".Setup1.Movement_Executability.movement102ExecutabilityLeft,
                           HMI_MOTION_EXECUTABILITY_RIGHT => "DB505_HMI_SetUp".Setup1.Movement_Executability.movement102ExecutabilityRight,
                           HMI_MOTION_END_POS_LEFT => "DB505_HMI_SetUp".Setup1.Movement_EndPos.movement102EndPosLeft,
                           HMI_MOTION_END_POS_RIGHT => "DB505_HMI_SetUp".Setup1.Movement_EndPos.movement102EndPosRight);
END_REGION

REGION Network 4: SPINDLE C12 OPERATOR HELP
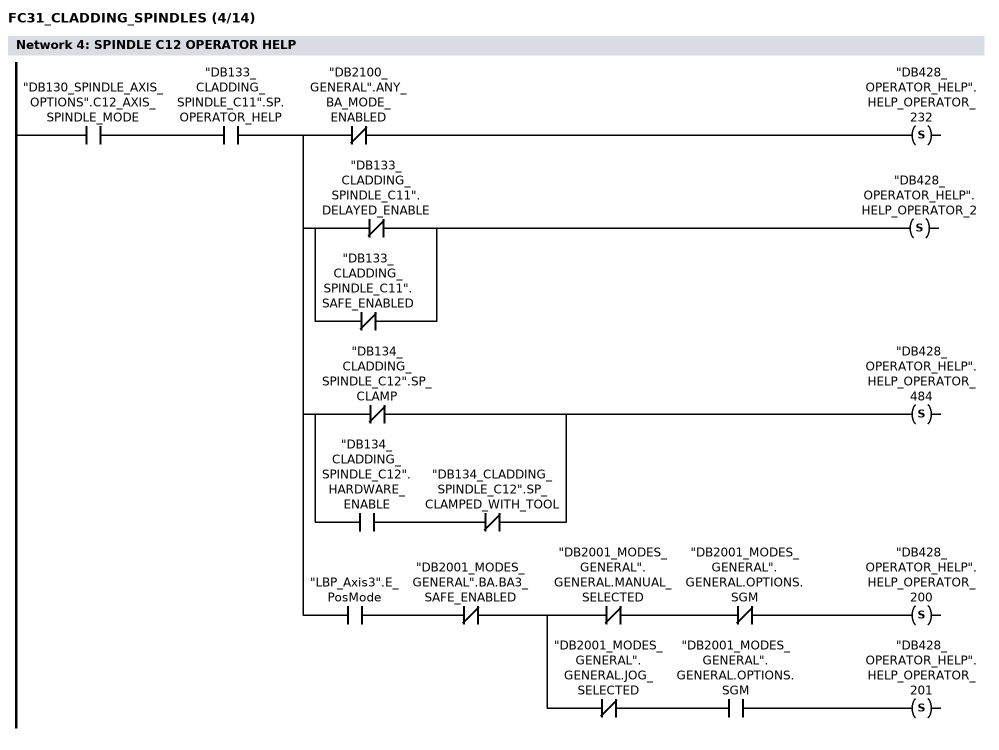
   RUNG wire#powerrail
      Contact( "DB130_SPINDLE_AXIS_OPTIONS".C12_AXIS_SPINDLE_MODE )
      Contact( "DB133_CLADDING_SPINDLE_C11".SP.OPERATOR_HELP )
      wire#w1
      I_Contact( "DB2100_GENERAL".ANY_BA_MODE_ENABLED )
      S_Coil( "DB428_OPERATOR_HELP".HELP_OPERATOR_232 )
   END_RUNG
   RUNG wire#w1
      I_Contact( "DB133_CLADDING_SPINDLE_C11".DELAYED_ENABLE )
      wire#w2
      S_Coil( "DB428_OPERATOR_HELP".HELP_OPERATOR_2 )
   END_RUNG
   RUNG wire#w1
      I_Contact( "DB133_CLADDING_SPINDLE_C11".SAFE_ENABLED )
   END_RUNG wire#w2
   RUNG wire#w1
      I_Contact( "DB134_CLADDING_SPINDLE_C12".SP_CLAMP )
      wire#w3
      S_Coil( "DB428_OPERATOR_HELP".HELP_OPERATOR_484 )
   END_RUNG
   RUNG wire#w1
      Contact( "DB134_CLADDING_SPINDLE_C12".HARDWARE_ENABLE )
      I_Contact( "DB134_CLADDING_SPINDLE_C12".SP_CLAMPED_WITH_TOOL )
   END_RUNG wire#w3
   RUNG wire#w1
      Contact( "LBP_Axis3".E_PosMode )
      I_Contact( "DB2001_MODES_GENERAL".BA.BA3_SAFE_ENABLED )
      wire#w4
      I_Contact( "DB2001_MODES_GENERAL".GENERAL.MANUAL_SELECTED )
      I_Contact( "DB2001_MODES_GENERAL".GENERAL.OPTIONS.SGM )
      S_Coil( "DB428_OPERATOR_HELP".HELP_OPERATOR_200 )
   END_RUNG
   RUNG wire#w4
      I_Contact( "DB2001_MODES_GENERAL".GENERAL.JOG_SELECTED )
      Contact( "DB2001_MODES_GENERAL".GENERAL.OPTIONS.SGM )
      S_Coil( "DB428_OPERATOR_HELP".HELP_OPERATOR_201 )
   END_RUNG
   // the same network as SCL:
   #_w1 := "DB130_SPINDLE_AXIS_OPTIONS".C12_AXIS_SPINDLE_MODE AND "DB133_CLADDING_SPINDLE_C11".SP.OPERATOR_HELP;
   IF #_w1 AND NOT "DB2100_GENERAL".ANY_BA_MODE_ENABLED THEN
       "DB428_OPERATOR_HELP".HELP_OPERATOR_232 := TRUE;
   END_IF;
   IF #_w1 AND (NOT "DB133_CLADDING_SPINDLE_C11".DELAYED_ENABLE OR NOT "DB133_CLADDING_SPINDLE_C11".SAFE_ENABLED) THEN
       "DB428_OPERATOR_HELP".HELP_OPERATOR_2 := TRUE;
   END_IF;
   IF #_w1 AND (NOT "DB134_CLADDING_SPINDLE_C12".SP_CLAMP OR ("DB134_CLADDING_SPINDLE_C12".HARDWARE_ENABLE AND NOT "DB134_CLADDING_SPINDLE_C12".SP_CLAMPED_WITH_TOOL)) THEN
       "DB428_OPERATOR_HELP".HELP_OPERATOR_484 := TRUE;
   END_IF;
   #_w2 := #_w1 AND "LBP_Axis3".E_PosMode AND NOT "DB2001_MODES_GENERAL".BA.BA3_SAFE_ENABLED;
   IF #_w2 AND NOT "DB2001_MODES_GENERAL".GENERAL.MANUAL_SELECTED AND NOT "DB2001_MODES_GENERAL".GENERAL.OPTIONS.SGM THEN
       "DB428_OPERATOR_HELP".HELP_OPERATOR_200 := TRUE;
   END_IF;
   IF #_w2 AND NOT "DB2001_MODES_GENERAL".GENERAL.JOG_SELECTED AND "DB2001_MODES_GENERAL".GENERAL.OPTIONS.SGM THEN
       "DB428_OPERATOR_HELP".HELP_OPERATOR_201 := TRUE;
   END_IF;
END_REGION

REGION Network 5: CALL FB31 SPINDLE C13
   // 2#0000_0001 OPTIONS 0 BIT 0 MEASURING SYSTEM 2 OPTION
   // 2#0000_0010 OPTIONS 0 BIT 1 BELT BROKEN OPTION
   // 2#0000_0100 OPTIONS 0 BIT 2 COOLING OPTION
   // 2#0000_1000 OPTIONS 0 BIT 3 MQL OR HP OPTION
   // 2#0001_0000 OPTIONS 0 BIT 4 ANALOG TEMPERATURE SENSOR OPTION
   // 2#0010_0000 OPTIONS 0 BIT 5 PTC TEMPERATURE SENSOR OPTION
   // 2#0100_0000 OPTIONS 0 BIT 6 TWIN KESSLER VPM READY OPTION
   // 2#1000_0000 OPTIONS 0 BIT 7 MPP SPINDLE OVERRIDE OPTION
   // 
   // 2#0000_0001 OPTIONS 1 BIT 0 SPARE OPTION
   // 2#0000_0010 OPTIONS 1 BIT 1 SPARE OPTION
   // 2#0000_0100 OPTIONS 1 BIT 2 SPARE OPTION
   // 2#0000_1000 OPTIONS 1 BIT 3 SPARE OPTION
   // 2#0001_0000 OPTIONS 1 BIT 4 SPARE OPTION
   // 2#0010_0000 OPTIONS 1 BIT 5 SPARE OPTION
   // 2#0100_0000 OPTIONS 1 BIT 6 SPARE OPTION
   // 2#1000_0000 OPTIONS 1 BIT 7 SPARE OPTION
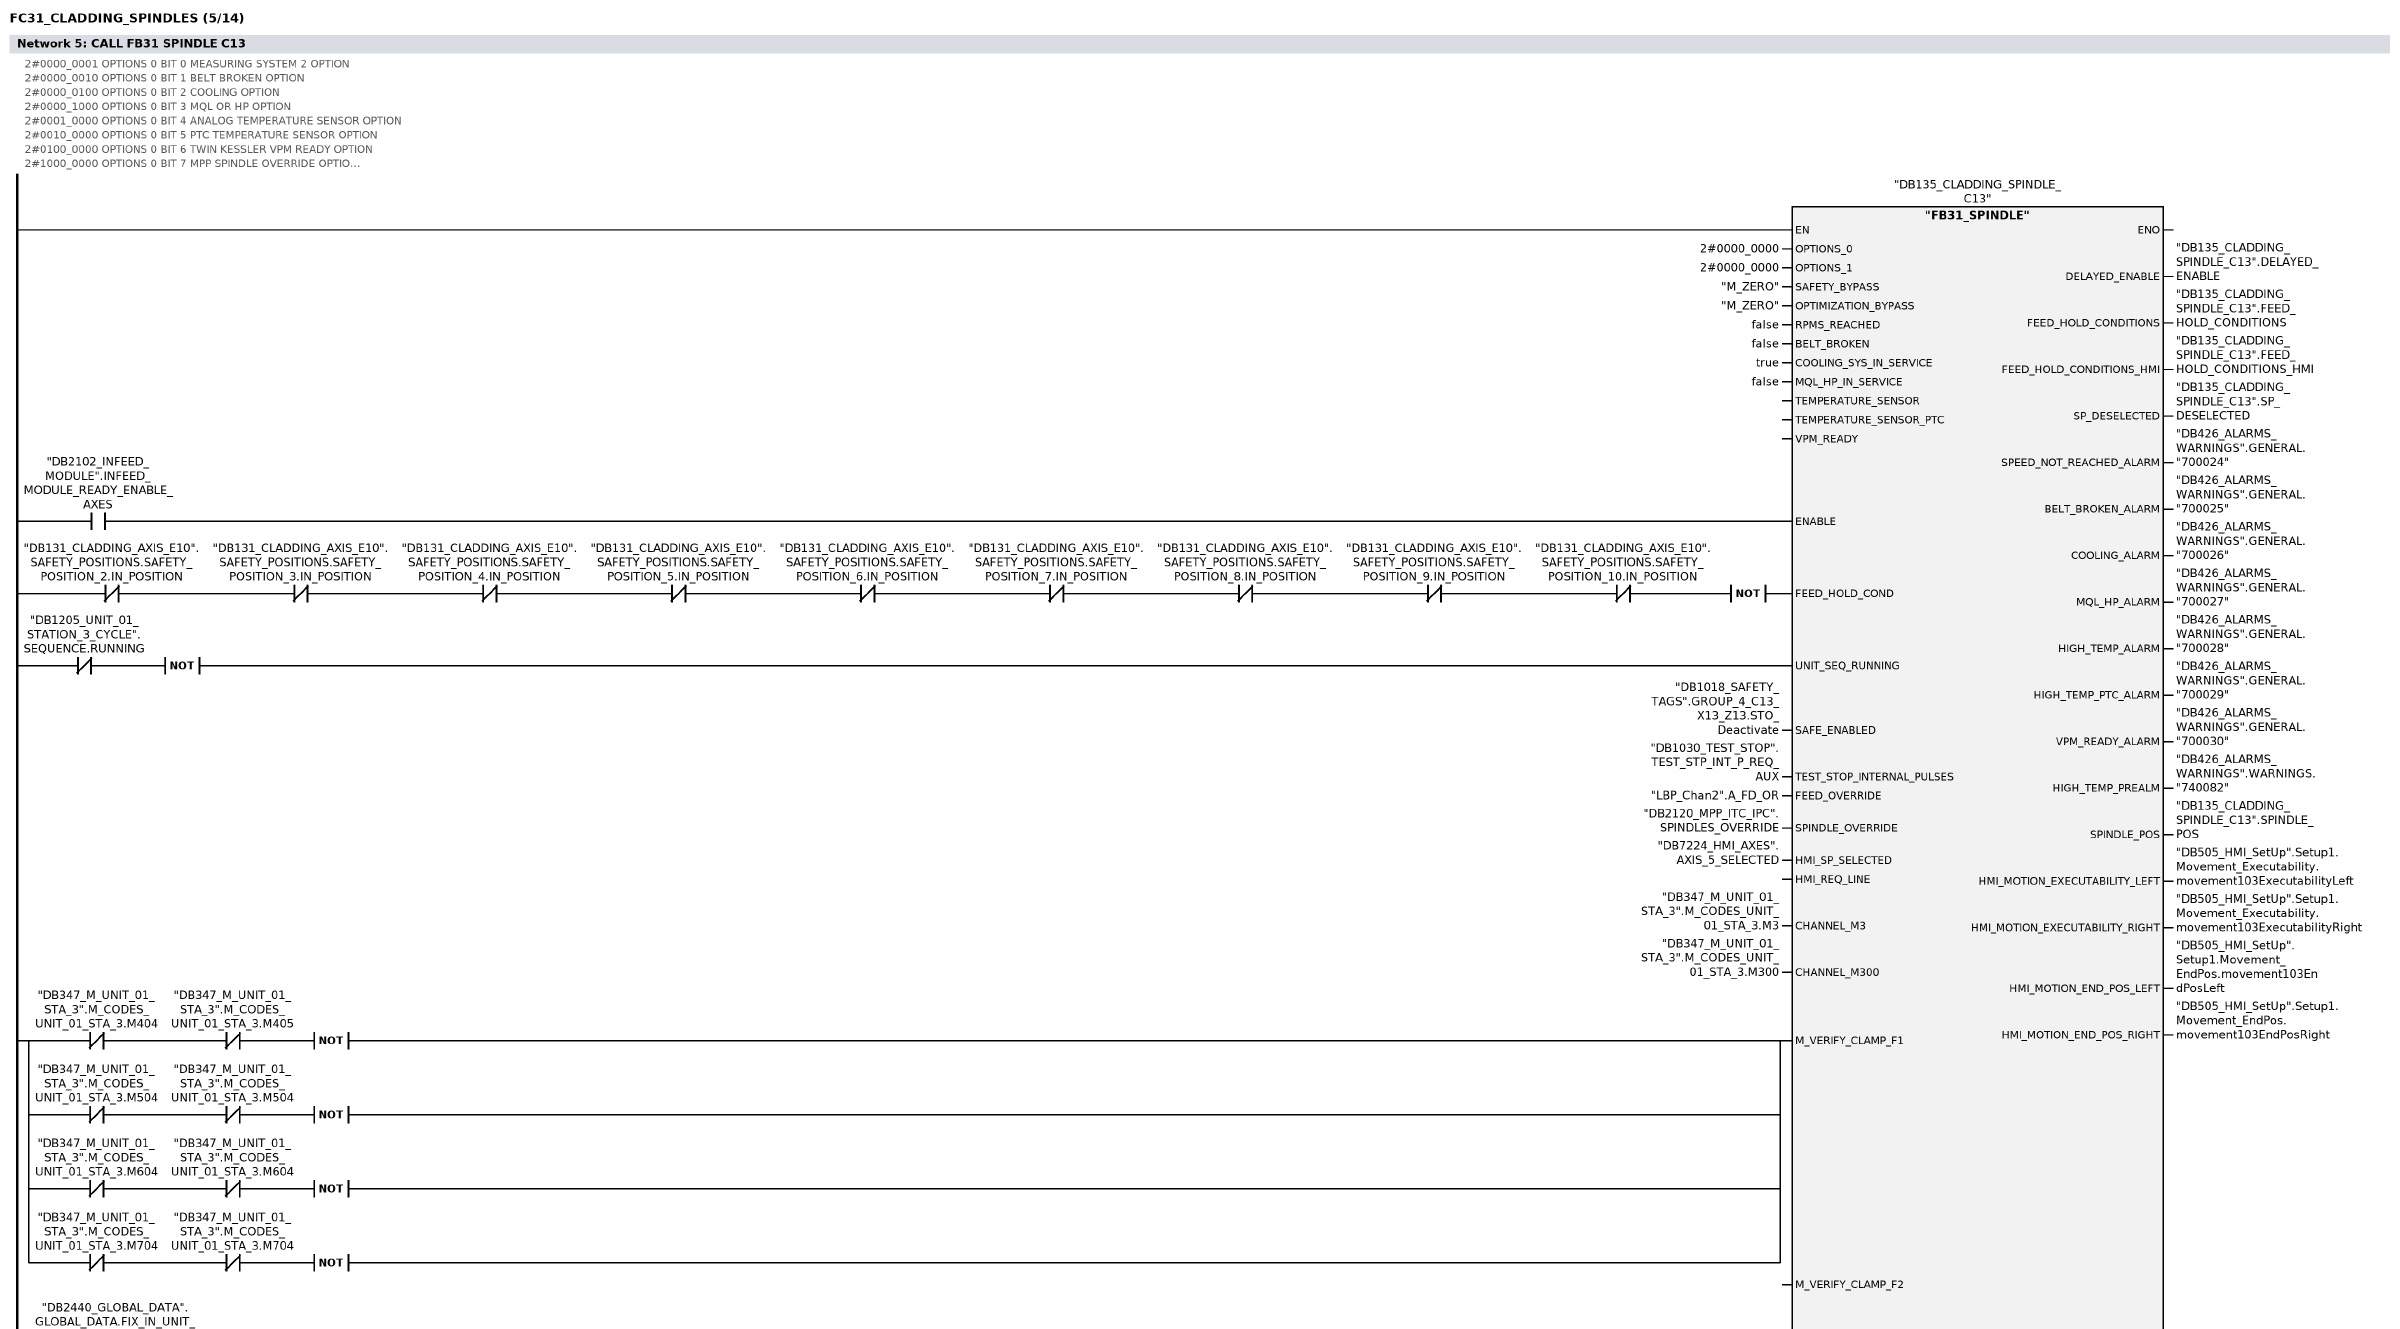
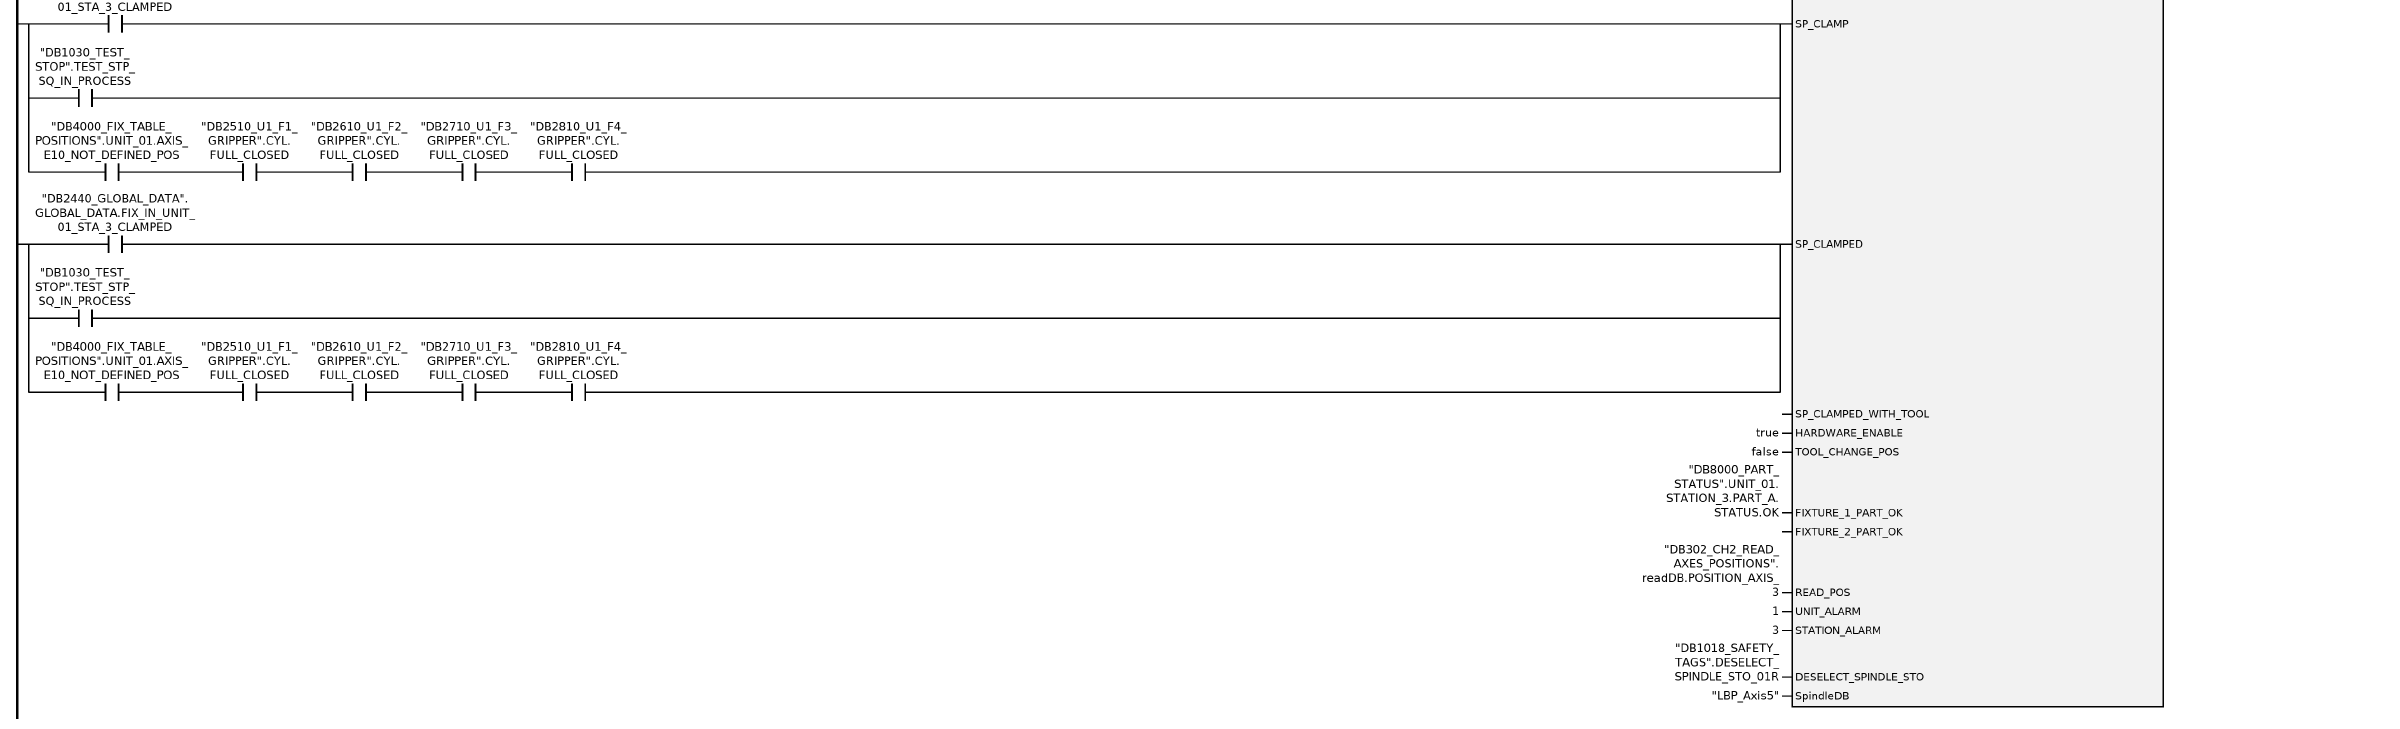
   RUNG wire#powerrail
      "DB135_CLADDING_SPINDLE_C13"(ENABLE := wire#w1, FEED_HOLD_COND := wire#w2, UNIT_SEQ_RUNNING := wire#w3, M_VERIFY_CLAMP_F1 := wire#w4, SP_CLAMP := wire#w5, SP_CLAMPED := wire#w6, OPTIONS_0 := 2#0000_0000, OPTIONS_1 := 2#0000_0000, SAFETY_BYPASS := "M_ZERO", OPTIMIZATION_BYPASS := "M_ZERO", RPMS_REACHED := false, BELT_BROKEN := false, COOLING_SYS_IN_SERVICE := true, MQL_HP_IN_SERVICE := false, TEMPERATURE_SENSOR :=, TEMPERATURE_SENSOR_PTC :=, VPM_READY :=, SAFE_ENABLED := "DB1018_SAFETY_TAGS".GROUP_4_C13_X13_Z13.STO_Deactivate, TEST_STOP_INTERNAL_PULSES := "DB1030_TEST_STOP".TEST_STP_INT_P_REQ_AUX, FEED_OVERRIDE := "LBP_Chan2".A_FD_OR, SPINDLE_OVERRIDE := "DB2120_MPP_ITC_IPC".SPINDLES_OVERRIDE, HMI_SP_SELECTED := "DB7224_HMI_AXES".AXIS_5_SELECTED, HMI_REQ_LINE :=, CHANNEL_M3 := "DB347_M_UNIT_01_STA_3".M_CODES_UNIT_01_STA_3.M3, CHANNEL_M300 := "DB347_M_UNIT_01_STA_3".M_CODES_UNIT_01_STA_3.M300, M_VERIFY_CLAMP_F2 :=, SP_CLAMPED_WITH_TOOL :=, HARDWARE_ENABLE := true, TOOL_CHANGE_POS := false, FIXTURE_1_PART_OK := "DB8000_PART_STATUS".UNIT_01.STATION_3.PART_A.STATUS.OK, FIXTURE_2_PART_OK :=, READ_POS := "DB302_CH2_READ_AXES_POSITIONS".readDB.POSITION_AXIS_3, UNIT_ALARM := 1, STATION_ALARM := 3, DESELECT_SPINDLE_STO := "DB1018_SAFETY_TAGS".DESELECT_SPINDLE_STO_01R, SpindleDB := "LBP_Axis5", DELAYED_ENABLE => "DB135_CLADDING_SPINDLE_C13".DELAYED_ENABLE, FEED_HOLD_CONDITIONS => "DB135_CLADDING_SPINDLE_C13".FEED_HOLD_CONDITIONS, FEED_HOLD_CONDITIONS_HMI => "DB135_CLADDING_SPINDLE_C13".FEED_HOLD_CONDITIONS_HMI, SP_DESELECTED => "DB135_CLADDING_SPINDLE_C13".SP_DESELECTED, SPEED_NOT_REACHED_ALARM => "DB426_ALARMS_WARNINGS".GENERAL."700024", BELT_BROKEN_ALARM => "DB426_ALARMS_WARNINGS".GENERAL."700025", COOLING_ALARM => "DB426_ALARMS_WARNINGS".GENERAL."700026", MQL_HP_ALARM => "DB426_ALARMS_WARNINGS".GENERAL."700027", HIGH_TEMP_ALARM => "DB426_ALARMS_WARNINGS".GENERAL."700028", HIGH_TEMP_PTC_ALARM => "DB426_ALARMS_WARNINGS".GENERAL."700029", VPM_READY_ALARM => "DB426_ALARMS_WARNINGS".GENERAL."700030", HIGH_TEMP_PREALM => "DB426_ALARMS_WARNINGS".WARNINGS."740082", SPINDLE_POS => "DB135_CLADDING_SPINDLE_C13".SPINDLE_POS, HMI_MOTION_EXECUTABILITY_LEFT => "DB505_HMI_SetUp".Setup1.Movement_Executability.movement103ExecutabilityLeft, HMI_MOTION_EXECUTABILITY_RIGHT => "DB505_HMI_SetUp".Setup1.Movement_Executability.movement103ExecutabilityRight, HMI_MOTION_END_POS_LEFT => "DB505_HMI_SetUp".Setup1.Movement_EndPos.movement103EndPosLeft, HMI_MOTION_END_POS_RIGHT => "DB505_HMI_SetUp".Setup1.Movement_EndPos.movement103EndPosRight)
   END_RUNG
   RUNG wire#powerrail
      Contact( "DB2102_INFEED_MODULE".INFEED_MODULE_READY_ENABLE_AXES )
   END_RUNG wire#w1
   RUNG wire#powerrail
      I_Contact( "DB131_CLADDING_AXIS_E10".SAFETY_POSITIONS.SAFETY_POSITION_2.IN_POSITION )
      I_Contact( "DB131_CLADDING_AXIS_E10".SAFETY_POSITIONS.SAFETY_POSITION_3.IN_POSITION )
      I_Contact( "DB131_CLADDING_AXIS_E10".SAFETY_POSITIONS.SAFETY_POSITION_4.IN_POSITION )
      I_Contact( "DB131_CLADDING_AXIS_E10".SAFETY_POSITIONS.SAFETY_POSITION_5.IN_POSITION )
      I_Contact( "DB131_CLADDING_AXIS_E10".SAFETY_POSITIONS.SAFETY_POSITION_6.IN_POSITION )
      I_Contact( "DB131_CLADDING_AXIS_E10".SAFETY_POSITIONS.SAFETY_POSITION_7.IN_POSITION )
      I_Contact( "DB131_CLADDING_AXIS_E10".SAFETY_POSITIONS.SAFETY_POSITION_8.IN_POSITION )
      I_Contact( "DB131_CLADDING_AXIS_E10".SAFETY_POSITIONS.SAFETY_POSITION_9.IN_POSITION )
      I_Contact( "DB131_CLADDING_AXIS_E10".SAFETY_POSITIONS.SAFETY_POSITION_10.IN_POSITION )
      Not()
   END_RUNG wire#w2
   RUNG wire#powerrail
      I_Contact( "DB1205_UNIT_01_STATION_3_CYCLE".SEQUENCE.RUNNING )
      Not()
   END_RUNG wire#w3
   RUNG wire#powerrail
      I_Contact( "DB347_M_UNIT_01_STA_3".M_CODES_UNIT_01_STA_3.M404 )
      I_Contact( "DB347_M_UNIT_01_STA_3".M_CODES_UNIT_01_STA_3.M405 )
      Not()
   END_RUNG wire#w4
   RUNG wire#powerrail
      I_Contact( "DB347_M_UNIT_01_STA_3".M_CODES_UNIT_01_STA_3.M504 )
      I_Contact( "DB347_M_UNIT_01_STA_3".M_CODES_UNIT_01_STA_3.M504 )
      Not()
   END_RUNG wire#w4
   RUNG wire#powerrail
      I_Contact( "DB347_M_UNIT_01_STA_3".M_CODES_UNIT_01_STA_3.M604 )
      I_Contact( "DB347_M_UNIT_01_STA_3".M_CODES_UNIT_01_STA_3.M604 )
      Not()
   END_RUNG wire#w4
   RUNG wire#powerrail
      I_Contact( "DB347_M_UNIT_01_STA_3".M_CODES_UNIT_01_STA_3.M704 )
      I_Contact( "DB347_M_UNIT_01_STA_3".M_CODES_UNIT_01_STA_3.M704 )
      Not()
   END_RUNG wire#w4
   RUNG wire#powerrail
      Contact( "DB2440_GLOBAL_DATA".GLOBAL_DATA.FIX_IN_UNIT_01_STA_3_CLAMPED )
   END_RUNG wire#w5
   RUNG wire#powerrail
      Contact( "DB1030_TEST_STOP".TEST_STP_SQ_IN_PROCESS )
   END_RUNG wire#w5
   RUNG wire#powerrail
      Contact( "DB4000_FIX_TABLE_POSITIONS".UNIT_01.AXIS_E10_NOT_DEFINED_POS )
      Contact( "DB2510_U1_F1_GRIPPER".CYL.FULL_CLOSED )
      Contact( "DB2610_U1_F2_GRIPPER".CYL.FULL_CLOSED )
      Contact( "DB2710_U1_F3_GRIPPER".CYL.FULL_CLOSED )
      Contact( "DB2810_U1_F4_GRIPPER".CYL.FULL_CLOSED )
   END_RUNG wire#w5
   RUNG wire#powerrail
      Contact( "DB2440_GLOBAL_DATA".GLOBAL_DATA.FIX_IN_UNIT_01_STA_3_CLAMPED )
   END_RUNG wire#w6
   RUNG wire#powerrail
      Contact( "DB1030_TEST_STOP".TEST_STP_SQ_IN_PROCESS )
   END_RUNG wire#w6
   RUNG wire#powerrail
      Contact( "DB4000_FIX_TABLE_POSITIONS".UNIT_01.AXIS_E10_NOT_DEFINED_POS )
      Contact( "DB2510_U1_F1_GRIPPER".CYL.FULL_CLOSED )
      Contact( "DB2610_U1_F2_GRIPPER".CYL.FULL_CLOSED )
      Contact( "DB2710_U1_F3_GRIPPER".CYL.FULL_CLOSED )
      Contact( "DB2810_U1_F4_GRIPPER".CYL.FULL_CLOSED )
   END_RUNG wire#w6
   // the same network as SCL:
   "DB135_CLADDING_SPINDLE_C13"(OPTIONS_0 := 2#0000_0000,   // "FB31_SPINDLE"
                           OPTIONS_1 := 2#0000_0000,
                           SAFETY_BYPASS := "M_ZERO",
                           OPTIMIZATION_BYPASS := "M_ZERO",
                           RPMS_REACHED := false,
                           BELT_BROKEN := false,
                           COOLING_SYS_IN_SERVICE := true,
                           MQL_HP_IN_SERVICE := false,
                           ENABLE := "DB2102_INFEED_MODULE".INFEED_MODULE_READY_ENABLE_AXES,
                           FEED_HOLD_COND := NOT (NOT "DB131_CLADDING_AXIS_E10".SAFETY_POSITIONS.SAFETY_POSITION_2.IN_POSITION AND NOT "DB131_CLADDING_AXIS_E10".SAFETY_POSITIONS.SAFETY_POSITION_3.IN_POSITION AND NOT "DB131_CLADDING_AXIS_E10".SAFETY_POSITIONS.SAFETY_POSITION_4.IN_POSITION AND NOT "DB131_CLADDING_AXIS_E10".SAFETY_POSITIONS.SAFETY_POSITION_5.IN_POSITION AND NOT "DB131_CLADDING_AXIS_E10".SAFETY_POSITIONS.SAFETY_POSITION_6.IN_POSITION AND NOT "DB131_CLADDING_AXIS_E10".SAFETY_POSITIONS.SAFETY_POSITION_7.IN_POSITION AND NOT "DB131_CLADDING_AXIS_E10".SAFETY_POSITIONS.SAFETY_POSITION_8.IN_POSITION AND NOT "DB131_CLADDING_AXIS_E10".SAFETY_POSITIONS.SAFETY_POSITION_9.IN_POSITION AND NOT "DB131_CLADDING_AXIS_E10".SAFETY_POSITIONS.SAFETY_POSITION_10.IN_POSITION),
                           UNIT_SEQ_RUNNING := NOT (NOT "DB1205_UNIT_01_STATION_3_CYCLE".SEQUENCE.RUNNING),
                           SAFE_ENABLED := "DB1018_SAFETY_TAGS".GROUP_4_C13_X13_Z13.STO_Deactivate,
                           TEST_STOP_INTERNAL_PULSES := "DB1030_TEST_STOP".TEST_STP_INT_P_REQ_AUX,
                           FEED_OVERRIDE := "LBP_Chan2".A_FD_OR,
                           SPINDLE_OVERRIDE := "DB2120_MPP_ITC_IPC".SPINDLES_OVERRIDE,
                           HMI_SP_SELECTED := "DB7224_HMI_AXES".AXIS_5_SELECTED,
                           CHANNEL_M3 := "DB347_M_UNIT_01_STA_3".M_CODES_UNIT_01_STA_3.M3,
                           CHANNEL_M300 := "DB347_M_UNIT_01_STA_3".M_CODES_UNIT_01_STA_3.M300,
                           M_VERIFY_CLAMP_F1 := NOT (NOT "DB347_M_UNIT_01_STA_3".M_CODES_UNIT_01_STA_3.M404 AND NOT "DB347_M_UNIT_01_STA_3".M_CODES_UNIT_01_STA_3.M405) OR NOT (NOT "DB347_M_UNIT_01_STA_3".M_CODES_UNIT_01_STA_3.M504 AND NOT "DB347_M_UNIT_01_STA_3".M_CODES_UNIT_01_STA_3.M504) OR NOT (NOT "DB347_M_UNIT_01_STA_3".M_CODES_UNIT_01_STA_3.M604 AND NOT "DB347_M_UNIT_01_STA_3".M_CODES_UNIT_01_STA_3.M604) OR NOT (NOT "DB347_M_UNIT_01_STA_3".M_CODES_UNIT_01_STA_3.M704 AND NOT "DB347_M_UNIT_01_STA_3".M_CODES_UNIT_01_STA_3.M704),
                           SP_CLAMP := "DB2440_GLOBAL_DATA".GLOBAL_DATA.FIX_IN_UNIT_01_STA_3_CLAMPED OR "DB1030_TEST_STOP".TEST_STP_SQ_IN_PROCESS OR ("DB4000_FIX_TABLE_POSITIONS".UNIT_01.AXIS_E10_NOT_DEFINED_POS AND "DB2510_U1_F1_GRIPPER".CYL.FULL_CLOSED AND "DB2610_U1_F2_GRIPPER".CYL.FULL_CLOSED AND "DB2710_U1_F3_GRIPPER".CYL.FULL_CLOSED AND "DB2810_U1_F4_GRIPPER".CYL.FULL_CLOSED),
                           SP_CLAMPED := "DB2440_GLOBAL_DATA".GLOBAL_DATA.FIX_IN_UNIT_01_STA_3_CLAMPED OR "DB1030_TEST_STOP".TEST_STP_SQ_IN_PROCESS OR ("DB4000_FIX_TABLE_POSITIONS".UNIT_01.AXIS_E10_NOT_DEFINED_POS AND "DB2510_U1_F1_GRIPPER".CYL.FULL_CLOSED AND "DB2610_U1_F2_GRIPPER".CYL.FULL_CLOSED AND "DB2710_U1_F3_GRIPPER".CYL.FULL_CLOSED AND "DB2810_U1_F4_GRIPPER".CYL.FULL_CLOSED),
                           HARDWARE_ENABLE := true,
                           TOOL_CHANGE_POS := false,
                           FIXTURE_1_PART_OK := "DB8000_PART_STATUS".UNIT_01.STATION_3.PART_A.STATUS.OK,
                           READ_POS := "DB302_CH2_READ_AXES_POSITIONS".readDB.POSITION_AXIS_3,
                           UNIT_ALARM := 1,
                           STATION_ALARM := 3,
                           DESELECT_SPINDLE_STO := "DB1018_SAFETY_TAGS".DESELECT_SPINDLE_STO_01R,
                           SpindleDB := "LBP_Axis5",
                           DELAYED_ENABLE => "DB135_CLADDING_SPINDLE_C13".DELAYED_ENABLE,
                           FEED_HOLD_CONDITIONS => "DB135_CLADDING_SPINDLE_C13".FEED_HOLD_CONDITIONS,
                           FEED_HOLD_CONDITIONS_HMI => "DB135_CLADDING_SPINDLE_C13".FEED_HOLD_CONDITIONS_HMI,
                           SP_DESELECTED => "DB135_CLADDING_SPINDLE_C13".SP_DESELECTED,
                           SPEED_NOT_REACHED_ALARM => "DB426_ALARMS_WARNINGS".GENERAL."700024",
                           BELT_BROKEN_ALARM => "DB426_ALARMS_WARNINGS".GENERAL."700025",
                           COOLING_ALARM => "DB426_ALARMS_WARNINGS".GENERAL."700026",
                           MQL_HP_ALARM => "DB426_ALARMS_WARNINGS".GENERAL."700027",
                           HIGH_TEMP_ALARM => "DB426_ALARMS_WARNINGS".GENERAL."700028",
                           HIGH_TEMP_PTC_ALARM => "DB426_ALARMS_WARNINGS".GENERAL."700029",
                           VPM_READY_ALARM => "DB426_ALARMS_WARNINGS".GENERAL."700030",
                           HIGH_TEMP_PREALM => "DB426_ALARMS_WARNINGS".WARNINGS."740082",
                           SPINDLE_POS => "DB135_CLADDING_SPINDLE_C13".SPINDLE_POS,
                           HMI_MOTION_EXECUTABILITY_LEFT => "DB505_HMI_SetUp".Setup1.Movement_Executability.movement103ExecutabilityLeft,
                           HMI_MOTION_EXECUTABILITY_RIGHT => "DB505_HMI_SetUp".Setup1.Movement_Executability.movement103ExecutabilityRight,
                           HMI_MOTION_END_POS_LEFT => "DB505_HMI_SetUp".Setup1.Movement_EndPos.movement103EndPosLeft,
                           HMI_MOTION_END_POS_RIGHT => "DB505_HMI_SetUp".Setup1.Movement_EndPos.movement103EndPosRight);
END_REGION

REGION Network 6: SPINDLE C13 OPERATOR HELP
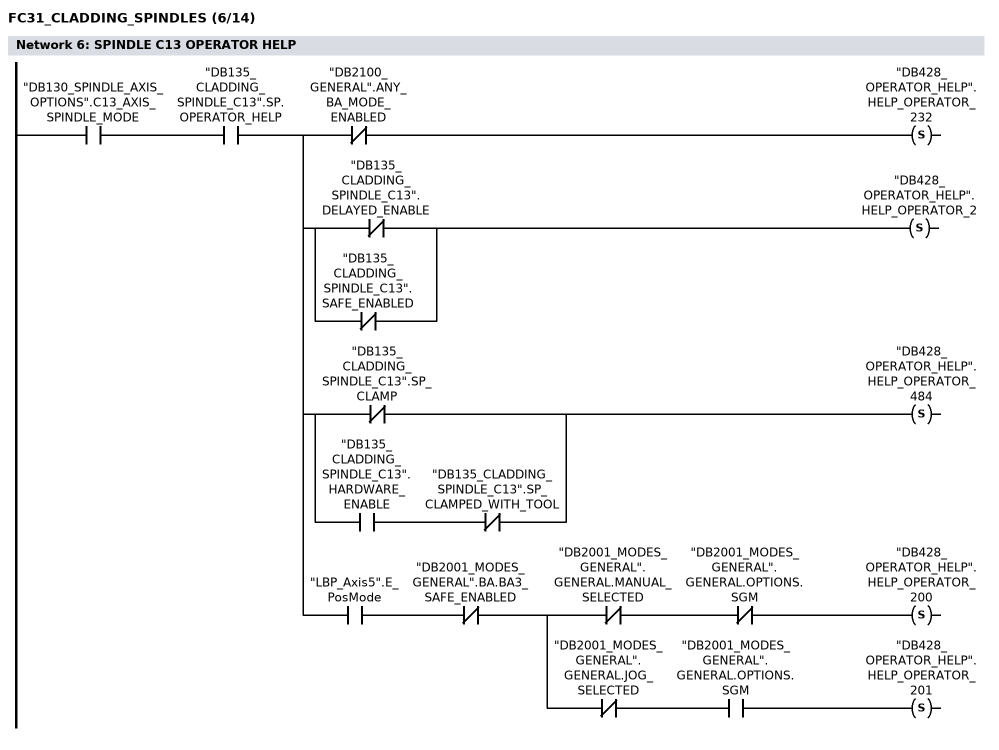
   RUNG wire#powerrail
      Contact( "DB130_SPINDLE_AXIS_OPTIONS".C13_AXIS_SPINDLE_MODE )
      Contact( "DB135_CLADDING_SPINDLE_C13".SP.OPERATOR_HELP )
      wire#w1
      I_Contact( "DB2100_GENERAL".ANY_BA_MODE_ENABLED )
      S_Coil( "DB428_OPERATOR_HELP".HELP_OPERATOR_232 )
   END_RUNG
   RUNG wire#w1
      I_Contact( "DB135_CLADDING_SPINDLE_C13".DELAYED_ENABLE )
      wire#w2
      S_Coil( "DB428_OPERATOR_HELP".HELP_OPERATOR_2 )
   END_RUNG
   RUNG wire#w1
      I_Contact( "DB135_CLADDING_SPINDLE_C13".SAFE_ENABLED )
   END_RUNG wire#w2
   RUNG wire#w1
      I_Contact( "DB135_CLADDING_SPINDLE_C13".SP_CLAMP )
      wire#w3
      S_Coil( "DB428_OPERATOR_HELP".HELP_OPERATOR_484 )
   END_RUNG
   RUNG wire#w1
      Contact( "DB135_CLADDING_SPINDLE_C13".HARDWARE_ENABLE )
      I_Contact( "DB135_CLADDING_SPINDLE_C13".SP_CLAMPED_WITH_TOOL )
   END_RUNG wire#w3
   RUNG wire#w1
      Contact( "LBP_Axis5".E_PosMode )
      I_Contact( "DB2001_MODES_GENERAL".BA.BA3_SAFE_ENABLED )
      wire#w4
      I_Contact( "DB2001_MODES_GENERAL".GENERAL.MANUAL_SELECTED )
      I_Contact( "DB2001_MODES_GENERAL".GENERAL.OPTIONS.SGM )
      S_Coil( "DB428_OPERATOR_HELP".HELP_OPERATOR_200 )
   END_RUNG
   RUNG wire#w4
      I_Contact( "DB2001_MODES_GENERAL".GENERAL.JOG_SELECTED )
      Contact( "DB2001_MODES_GENERAL".GENERAL.OPTIONS.SGM )
      S_Coil( "DB428_OPERATOR_HELP".HELP_OPERATOR_201 )
   END_RUNG
   // the same network as SCL:
   #_w1 := "DB130_SPINDLE_AXIS_OPTIONS".C13_AXIS_SPINDLE_MODE AND "DB135_CLADDING_SPINDLE_C13".SP.OPERATOR_HELP;
   IF #_w1 AND NOT "DB2100_GENERAL".ANY_BA_MODE_ENABLED THEN
       "DB428_OPERATOR_HELP".HELP_OPERATOR_232 := TRUE;
   END_IF;
   IF #_w1 AND (NOT "DB135_CLADDING_SPINDLE_C13".DELAYED_ENABLE OR NOT "DB135_CLADDING_SPINDLE_C13".SAFE_ENABLED) THEN
       "DB428_OPERATOR_HELP".HELP_OPERATOR_2 := TRUE;
   END_IF;
   IF #_w1 AND (NOT "DB135_CLADDING_SPINDLE_C13".SP_CLAMP OR ("DB135_CLADDING_SPINDLE_C13".HARDWARE_ENABLE AND NOT "DB135_CLADDING_SPINDLE_C13".SP_CLAMPED_WITH_TOOL)) THEN
       "DB428_OPERATOR_HELP".HELP_OPERATOR_484 := TRUE;
   END_IF;
   #_w2 := #_w1 AND "LBP_Axis5".E_PosMode AND NOT "DB2001_MODES_GENERAL".BA.BA3_SAFE_ENABLED;
   IF #_w2 AND NOT "DB2001_MODES_GENERAL".GENERAL.MANUAL_SELECTED AND NOT "DB2001_MODES_GENERAL".GENERAL.OPTIONS.SGM THEN
       "DB428_OPERATOR_HELP".HELP_OPERATOR_200 := TRUE;
   END_IF;
   IF #_w2 AND NOT "DB2001_MODES_GENERAL".GENERAL.JOG_SELECTED AND "DB2001_MODES_GENERAL".GENERAL.OPTIONS.SGM THEN
       "DB428_OPERATOR_HELP".HELP_OPERATOR_201 := TRUE;
   END_IF;
END_REGION

REGION Network 7: CALL FB31 SPINDLE C14
   // 2#0000_0001 OPTIONS 0 BIT 0 MEASURING SYSTEM 2 OPTION
   // 2#0000_0010 OPTIONS 0 BIT 1 BELT BROKEN OPTION
   // 2#0000_0100 OPTIONS 0 BIT 2 COOLING OPTION
   // 2#0000_1000 OPTIONS 0 BIT 3 MQL OR HP OPTION
   // 2#0001_0000 OPTIONS 0 BIT 4 ANALOG TEMPERATURE SENSOR OPTION
   // 2#0010_0000 OPTIONS 0 BIT 5 PTC TEMPERATURE SENSOR OPTION
   // 2#0100_0000 OPTIONS 0 BIT 6 TWIN KESSLER VPM READY OPTION
   // 2#1000_0000 OPTIONS 0 BIT 7 MPP SPINDLE OVERRIDE OPTION
   // 
   // 2#0000_0001 OPTIONS 1 BIT 0 SPARE OPTION
   // 2#0000_0010 OPTIONS 1 BIT 1 SPARE OPTION
   // 2#0000_0100 OPTIONS 1 BIT 2 SPARE OPTION
   // 2#0000_1000 OPTIONS 1 BIT 3 SPARE OPTION
   // 2#0001_0000 OPTIONS 1 BIT 4 SPARE OPTION
   // 2#0010_0000 OPTIONS 1 BIT 5 SPARE OPTION
   // 2#0100_0000 OPTIONS 1 BIT 6 SPARE OPTION
   // 2#1000_0000 OPTIONS 1 BIT 7 SPARE OPTION
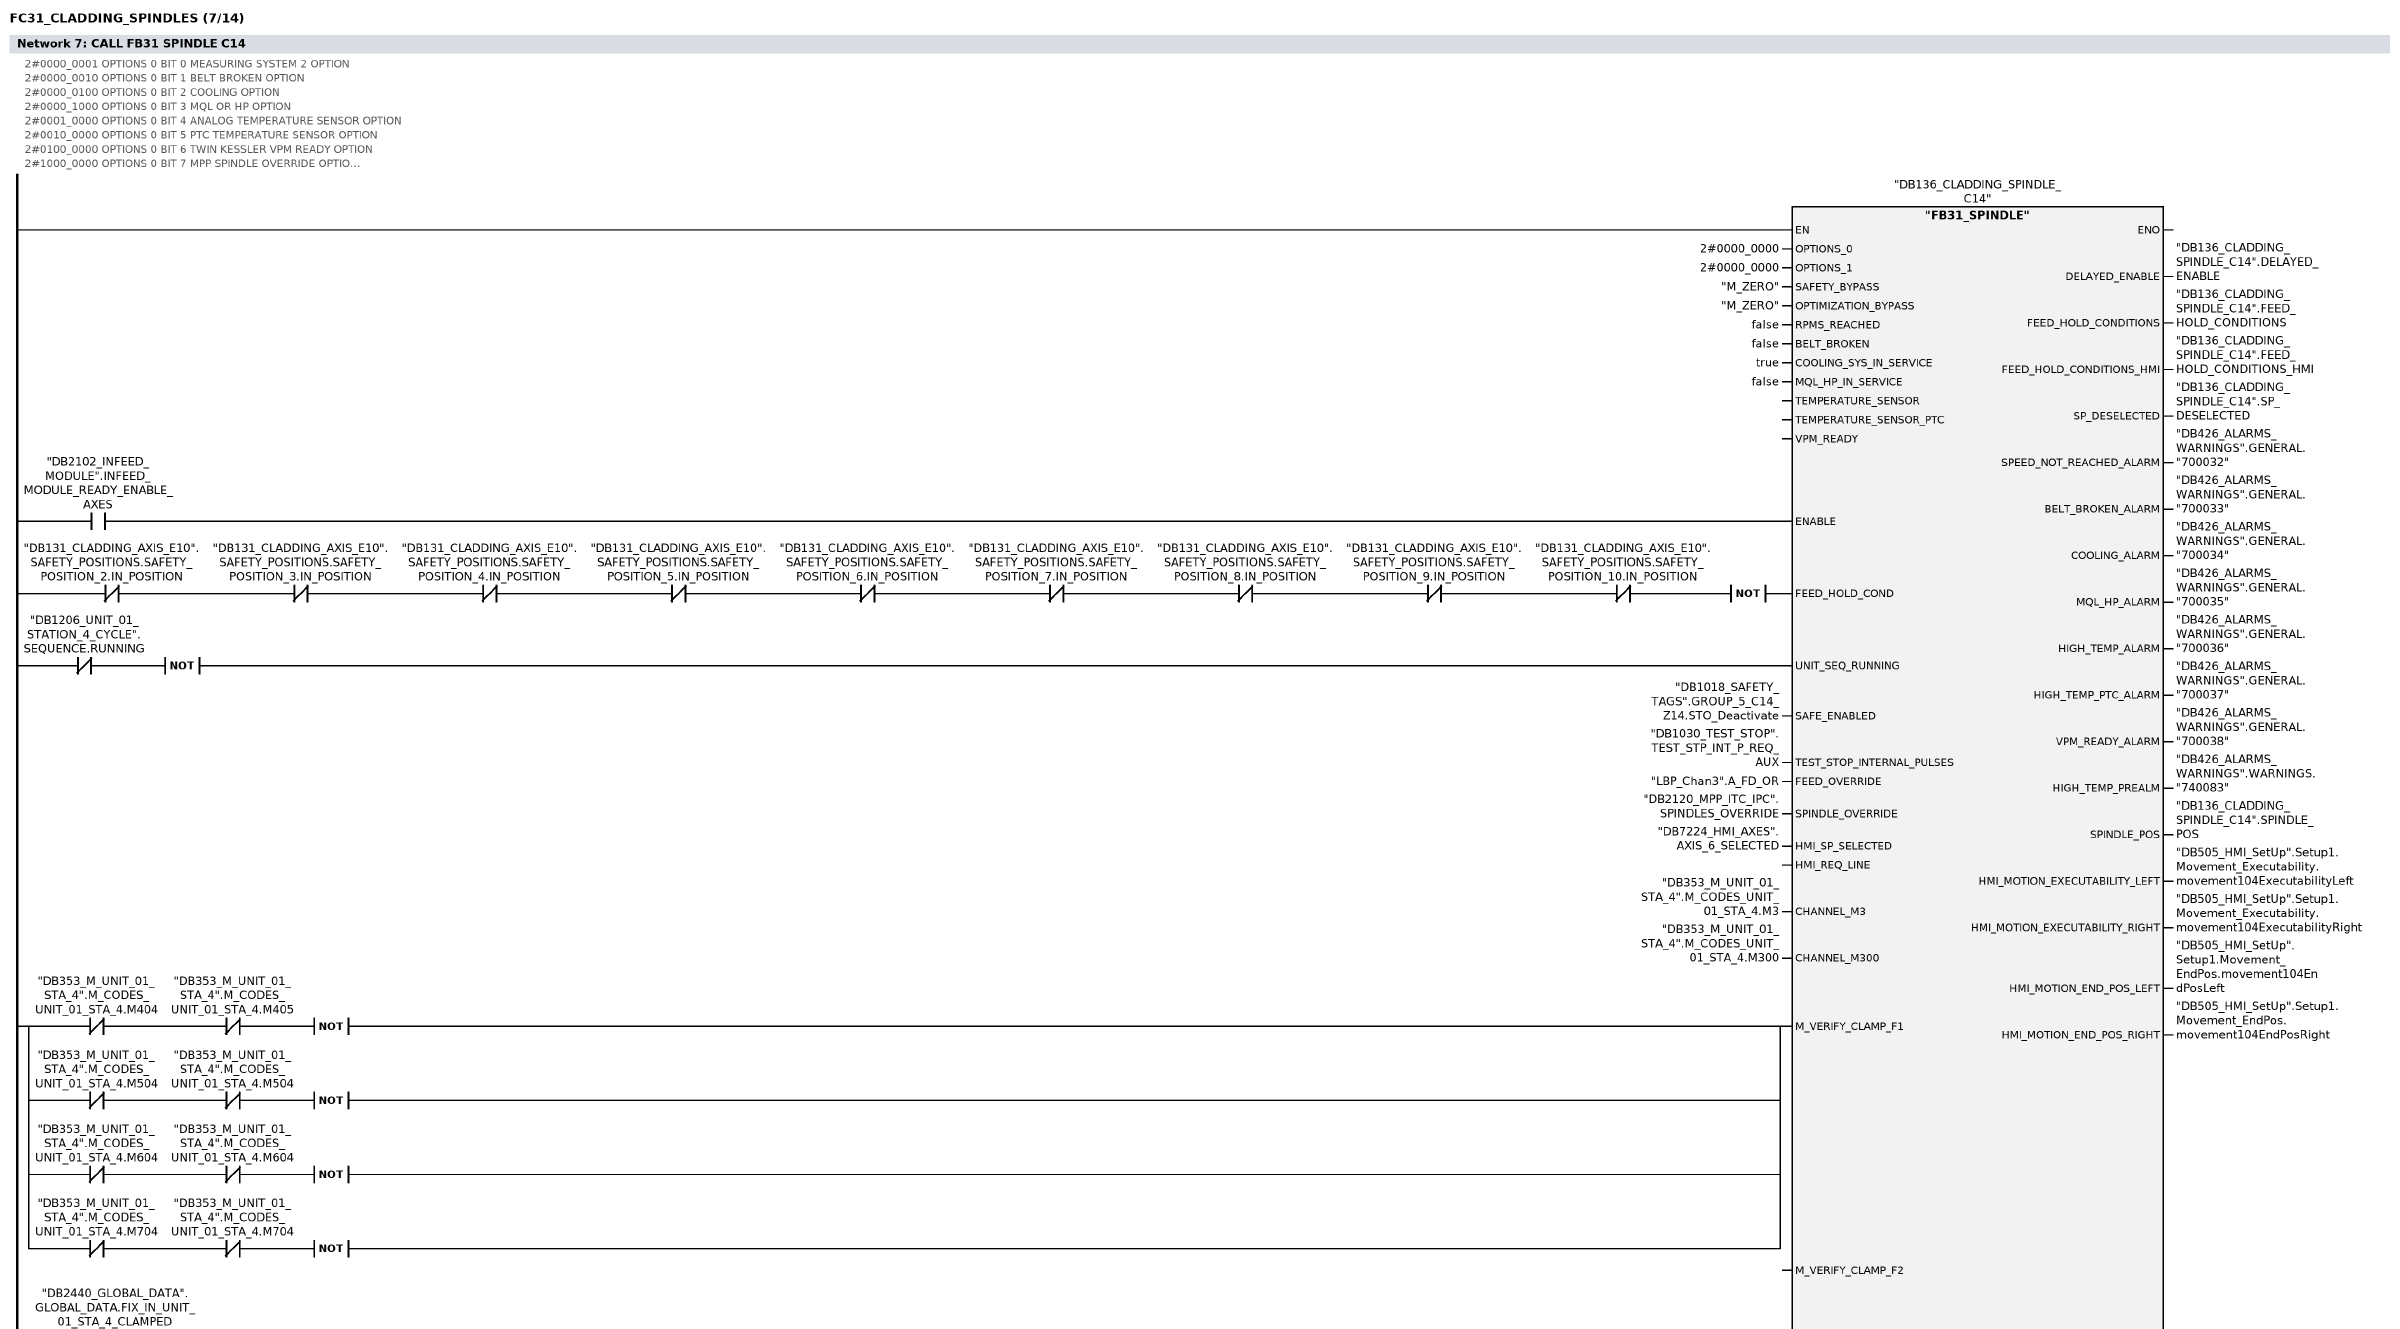
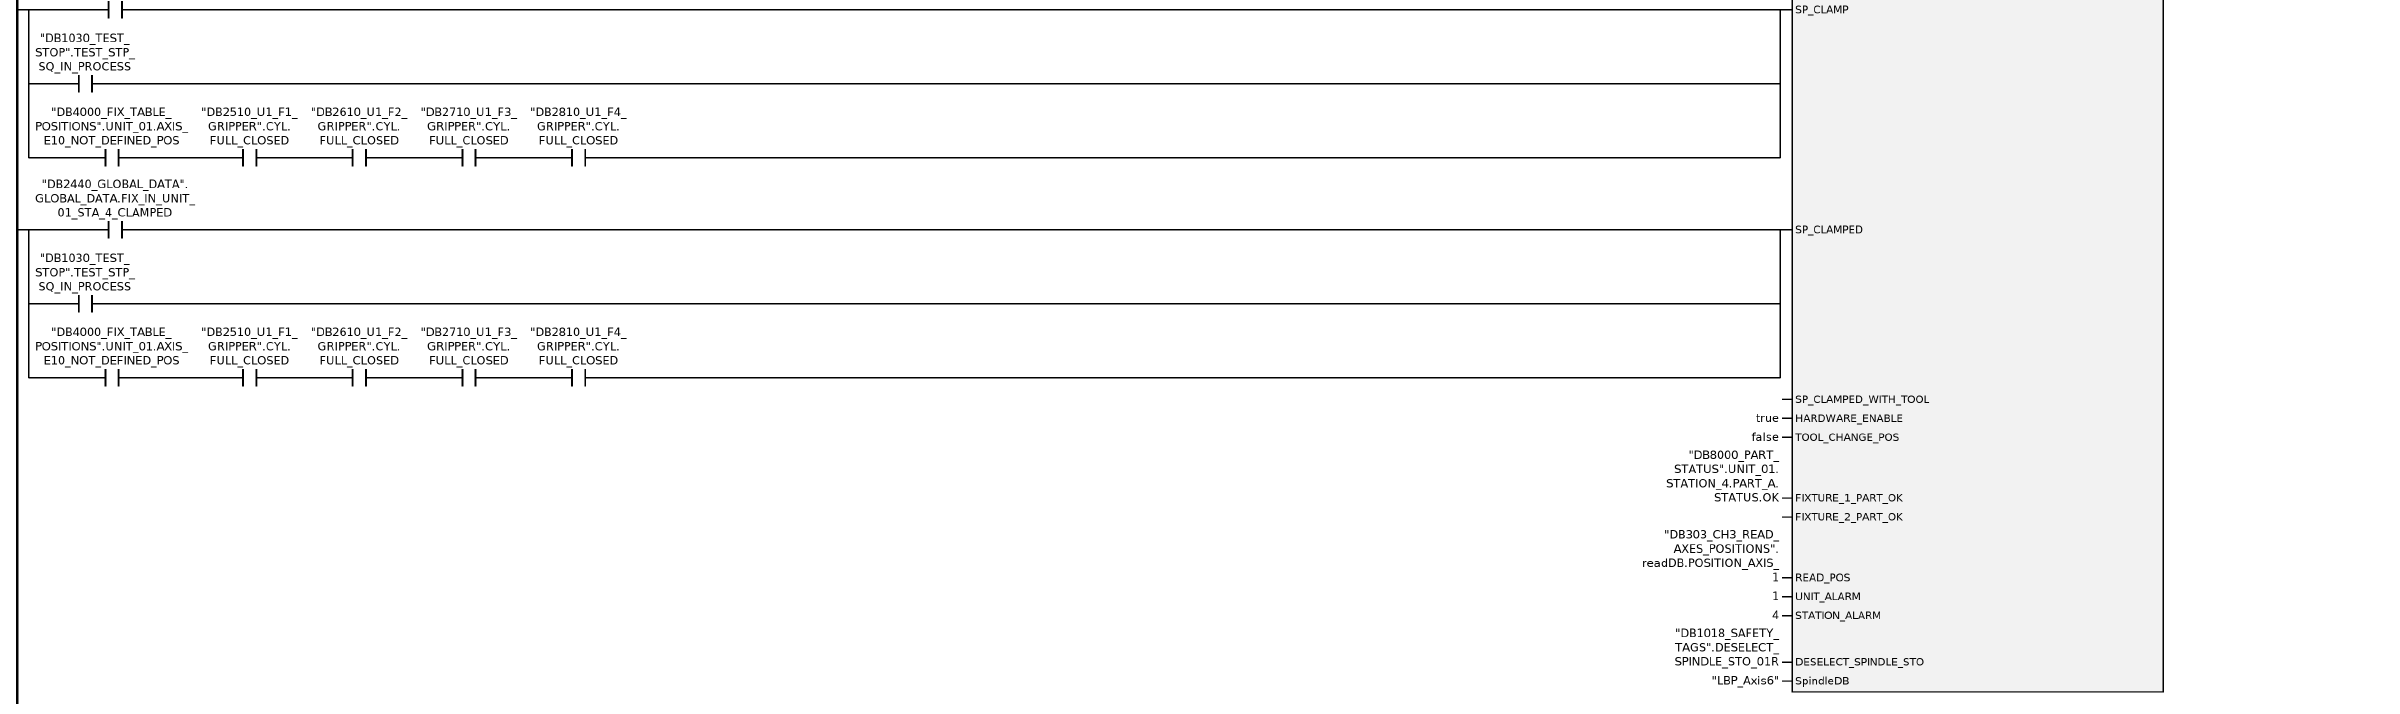
   RUNG wire#powerrail
      "DB136_CLADDING_SPINDLE_C14"(ENABLE := wire#w1, FEED_HOLD_COND := wire#w2, UNIT_SEQ_RUNNING := wire#w3, M_VERIFY_CLAMP_F1 := wire#w4, SP_CLAMP := wire#w5, SP_CLAMPED := wire#w6, OPTIONS_0 := 2#0000_0000, OPTIONS_1 := 2#0000_0000, SAFETY_BYPASS := "M_ZERO", OPTIMIZATION_BYPASS := "M_ZERO", RPMS_REACHED := false, BELT_BROKEN := false, COOLING_SYS_IN_SERVICE := true, MQL_HP_IN_SERVICE := false, TEMPERATURE_SENSOR :=, TEMPERATURE_SENSOR_PTC :=, VPM_READY :=, SAFE_ENABLED := "DB1018_SAFETY_TAGS".GROUP_5_C14_Z14.STO_Deactivate, TEST_STOP_INTERNAL_PULSES := "DB1030_TEST_STOP".TEST_STP_INT_P_REQ_AUX, FEED_OVERRIDE := "LBP_Chan3".A_FD_OR, SPINDLE_OVERRIDE := "DB2120_MPP_ITC_IPC".SPINDLES_OVERRIDE, HMI_SP_SELECTED := "DB7224_HMI_AXES".AXIS_6_SELECTED, HMI_REQ_LINE :=, CHANNEL_M3 := "DB353_M_UNIT_01_STA_4".M_CODES_UNIT_01_STA_4.M3, CHANNEL_M300 := "DB353_M_UNIT_01_STA_4".M_CODES_UNIT_01_STA_4.M300, M_VERIFY_CLAMP_F2 :=, SP_CLAMPED_WITH_TOOL :=, HARDWARE_ENABLE := true, TOOL_CHANGE_POS := false, FIXTURE_1_PART_OK := "DB8000_PART_STATUS".UNIT_01.STATION_4.PART_A.STATUS.OK, FIXTURE_2_PART_OK :=, READ_POS := "DB303_CH3_READ_AXES_POSITIONS".readDB.POSITION_AXIS_1, UNIT_ALARM := 1, STATION_ALARM := 4, DESELECT_SPINDLE_STO := "DB1018_SAFETY_TAGS".DESELECT_SPINDLE_STO_01R, SpindleDB := "LBP_Axis6", DELAYED_ENABLE => "DB136_CLADDING_SPINDLE_C14".DELAYED_ENABLE, FEED_HOLD_CONDITIONS => "DB136_CLADDING_SPINDLE_C14".FEED_HOLD_CONDITIONS, FEED_HOLD_CONDITIONS_HMI => "DB136_CLADDING_SPINDLE_C14".FEED_HOLD_CONDITIONS_HMI, SP_DESELECTED => "DB136_CLADDING_SPINDLE_C14".SP_DESELECTED, SPEED_NOT_REACHED_ALARM => "DB426_ALARMS_WARNINGS".GENERAL."700032", BELT_BROKEN_ALARM => "DB426_ALARMS_WARNINGS".GENERAL."700033", COOLING_ALARM => "DB426_ALARMS_WARNINGS".GENERAL."700034", MQL_HP_ALARM => "DB426_ALARMS_WARNINGS".GENERAL."700035", HIGH_TEMP_ALARM => "DB426_ALARMS_WARNINGS".GENERAL."700036", HIGH_TEMP_PTC_ALARM => "DB426_ALARMS_WARNINGS".GENERAL."700037", VPM_READY_ALARM => "DB426_ALARMS_WARNINGS".GENERAL."700038", HIGH_TEMP_PREALM => "DB426_ALARMS_WARNINGS".WARNINGS."740083", SPINDLE_POS => "DB136_CLADDING_SPINDLE_C14".SPINDLE_POS, HMI_MOTION_EXECUTABILITY_LEFT => "DB505_HMI_SetUp".Setup1.Movement_Executability.movement104ExecutabilityLeft, HMI_MOTION_EXECUTABILITY_RIGHT => "DB505_HMI_SetUp".Setup1.Movement_Executability.movement104ExecutabilityRight, HMI_MOTION_END_POS_LEFT => "DB505_HMI_SetUp".Setup1.Movement_EndPos.movement104EndPosLeft, HMI_MOTION_END_POS_RIGHT => "DB505_HMI_SetUp".Setup1.Movement_EndPos.movement104EndPosRight)
   END_RUNG
   RUNG wire#powerrail
      Contact( "DB2102_INFEED_MODULE".INFEED_MODULE_READY_ENABLE_AXES )
   END_RUNG wire#w1
   RUNG wire#powerrail
      I_Contact( "DB131_CLADDING_AXIS_E10".SAFETY_POSITIONS.SAFETY_POSITION_2.IN_POSITION )
      I_Contact( "DB131_CLADDING_AXIS_E10".SAFETY_POSITIONS.SAFETY_POSITION_3.IN_POSITION )
      I_Contact( "DB131_CLADDING_AXIS_E10".SAFETY_POSITIONS.SAFETY_POSITION_4.IN_POSITION )
      I_Contact( "DB131_CLADDING_AXIS_E10".SAFETY_POSITIONS.SAFETY_POSITION_5.IN_POSITION )
      I_Contact( "DB131_CLADDING_AXIS_E10".SAFETY_POSITIONS.SAFETY_POSITION_6.IN_POSITION )
      I_Contact( "DB131_CLADDING_AXIS_E10".SAFETY_POSITIONS.SAFETY_POSITION_7.IN_POSITION )
      I_Contact( "DB131_CLADDING_AXIS_E10".SAFETY_POSITIONS.SAFETY_POSITION_8.IN_POSITION )
      I_Contact( "DB131_CLADDING_AXIS_E10".SAFETY_POSITIONS.SAFETY_POSITION_9.IN_POSITION )
      I_Contact( "DB131_CLADDING_AXIS_E10".SAFETY_POSITIONS.SAFETY_POSITION_10.IN_POSITION )
      Not()
   END_RUNG wire#w2
   RUNG wire#powerrail
      I_Contact( "DB1206_UNIT_01_STATION_4_CYCLE".SEQUENCE.RUNNING )
      Not()
   END_RUNG wire#w3
   RUNG wire#powerrail
      I_Contact( "DB353_M_UNIT_01_STA_4".M_CODES_UNIT_01_STA_4.M404 )
      I_Contact( "DB353_M_UNIT_01_STA_4".M_CODES_UNIT_01_STA_4.M405 )
      Not()
   END_RUNG wire#w4
   RUNG wire#powerrail
      I_Contact( "DB353_M_UNIT_01_STA_4".M_CODES_UNIT_01_STA_4.M504 )
      I_Contact( "DB353_M_UNIT_01_STA_4".M_CODES_UNIT_01_STA_4.M504 )
      Not()
   END_RUNG wire#w4
   RUNG wire#powerrail
      I_Contact( "DB353_M_UNIT_01_STA_4".M_CODES_UNIT_01_STA_4.M604 )
      I_Contact( "DB353_M_UNIT_01_STA_4".M_CODES_UNIT_01_STA_4.M604 )
      Not()
   END_RUNG wire#w4
   RUNG wire#powerrail
      I_Contact( "DB353_M_UNIT_01_STA_4".M_CODES_UNIT_01_STA_4.M704 )
      I_Contact( "DB353_M_UNIT_01_STA_4".M_CODES_UNIT_01_STA_4.M704 )
      Not()
   END_RUNG wire#w4
   RUNG wire#powerrail
      Contact( "DB2440_GLOBAL_DATA".GLOBAL_DATA.FIX_IN_UNIT_01_STA_4_CLAMPED )
   END_RUNG wire#w5
   RUNG wire#powerrail
      Contact( "DB1030_TEST_STOP".TEST_STP_SQ_IN_PROCESS )
   END_RUNG wire#w5
   RUNG wire#powerrail
      Contact( "DB4000_FIX_TABLE_POSITIONS".UNIT_01.AXIS_E10_NOT_DEFINED_POS )
      Contact( "DB2510_U1_F1_GRIPPER".CYL.FULL_CLOSED )
      Contact( "DB2610_U1_F2_GRIPPER".CYL.FULL_CLOSED )
      Contact( "DB2710_U1_F3_GRIPPER".CYL.FULL_CLOSED )
      Contact( "DB2810_U1_F4_GRIPPER".CYL.FULL_CLOSED )
   END_RUNG wire#w5
   RUNG wire#powerrail
      Contact( "DB2440_GLOBAL_DATA".GLOBAL_DATA.FIX_IN_UNIT_01_STA_4_CLAMPED )
   END_RUNG wire#w6
   RUNG wire#powerrail
      Contact( "DB1030_TEST_STOP".TEST_STP_SQ_IN_PROCESS )
   END_RUNG wire#w6
   RUNG wire#powerrail
      Contact( "DB4000_FIX_TABLE_POSITIONS".UNIT_01.AXIS_E10_NOT_DEFINED_POS )
      Contact( "DB2510_U1_F1_GRIPPER".CYL.FULL_CLOSED )
      Contact( "DB2610_U1_F2_GRIPPER".CYL.FULL_CLOSED )
      Contact( "DB2710_U1_F3_GRIPPER".CYL.FULL_CLOSED )
      Contact( "DB2810_U1_F4_GRIPPER".CYL.FULL_CLOSED )
   END_RUNG wire#w6
   // the same network as SCL:
   "DB136_CLADDING_SPINDLE_C14"(OPTIONS_0 := 2#0000_0000,   // "FB31_SPINDLE"
                           OPTIONS_1 := 2#0000_0000,
                           SAFETY_BYPASS := "M_ZERO",
                           OPTIMIZATION_BYPASS := "M_ZERO",
                           RPMS_REACHED := false,
                           BELT_BROKEN := false,
                           COOLING_SYS_IN_SERVICE := true,
                           MQL_HP_IN_SERVICE := false,
                           ENABLE := "DB2102_INFEED_MODULE".INFEED_MODULE_READY_ENABLE_AXES,
                           FEED_HOLD_COND := NOT (NOT "DB131_CLADDING_AXIS_E10".SAFETY_POSITIONS.SAFETY_POSITION_2.IN_POSITION AND NOT "DB131_CLADDING_AXIS_E10".SAFETY_POSITIONS.SAFETY_POSITION_3.IN_POSITION AND NOT "DB131_CLADDING_AXIS_E10".SAFETY_POSITIONS.SAFETY_POSITION_4.IN_POSITION AND NOT "DB131_CLADDING_AXIS_E10".SAFETY_POSITIONS.SAFETY_POSITION_5.IN_POSITION AND NOT "DB131_CLADDING_AXIS_E10".SAFETY_POSITIONS.SAFETY_POSITION_6.IN_POSITION AND NOT "DB131_CLADDING_AXIS_E10".SAFETY_POSITIONS.SAFETY_POSITION_7.IN_POSITION AND NOT "DB131_CLADDING_AXIS_E10".SAFETY_POSITIONS.SAFETY_POSITION_8.IN_POSITION AND NOT "DB131_CLADDING_AXIS_E10".SAFETY_POSITIONS.SAFETY_POSITION_9.IN_POSITION AND NOT "DB131_CLADDING_AXIS_E10".SAFETY_POSITIONS.SAFETY_POSITION_10.IN_POSITION),
                           UNIT_SEQ_RUNNING := NOT (NOT "DB1206_UNIT_01_STATION_4_CYCLE".SEQUENCE.RUNNING),
                           SAFE_ENABLED := "DB1018_SAFETY_TAGS".GROUP_5_C14_Z14.STO_Deactivate,
                           TEST_STOP_INTERNAL_PULSES := "DB1030_TEST_STOP".TEST_STP_INT_P_REQ_AUX,
                           FEED_OVERRIDE := "LBP_Chan3".A_FD_OR,
                           SPINDLE_OVERRIDE := "DB2120_MPP_ITC_IPC".SPINDLES_OVERRIDE,
                           HMI_SP_SELECTED := "DB7224_HMI_AXES".AXIS_6_SELECTED,
                           CHANNEL_M3 := "DB353_M_UNIT_01_STA_4".M_CODES_UNIT_01_STA_4.M3,
                           CHANNEL_M300 := "DB353_M_UNIT_01_STA_4".M_CODES_UNIT_01_STA_4.M300,
                           M_VERIFY_CLAMP_F1 := NOT (NOT "DB353_M_UNIT_01_STA_4".M_CODES_UNIT_01_STA_4.M404 AND NOT "DB353_M_UNIT_01_STA_4".M_CODES_UNIT_01_STA_4.M405) OR NOT (NOT "DB353_M_UNIT_01_STA_4".M_CODES_UNIT_01_STA_4.M504 AND NOT "DB353_M_UNIT_01_STA_4".M_CODES_UNIT_01_STA_4.M504) OR NOT (NOT "DB353_M_UNIT_01_STA_4".M_CODES_UNIT_01_STA_4.M604 AND NOT "DB353_M_UNIT_01_STA_4".M_CODES_UNIT_01_STA_4.M604) OR NOT (NOT "DB353_M_UNIT_01_STA_4".M_CODES_UNIT_01_STA_4.M704 AND NOT "DB353_M_UNIT_01_STA_4".M_CODES_UNIT_01_STA_4.M704),
                           SP_CLAMP := "DB2440_GLOBAL_DATA".GLOBAL_DATA.FIX_IN_UNIT_01_STA_4_CLAMPED OR "DB1030_TEST_STOP".TEST_STP_SQ_IN_PROCESS OR ("DB4000_FIX_TABLE_POSITIONS".UNIT_01.AXIS_E10_NOT_DEFINED_POS AND "DB2510_U1_F1_GRIPPER".CYL.FULL_CLOSED AND "DB2610_U1_F2_GRIPPER".CYL.FULL_CLOSED AND "DB2710_U1_F3_GRIPPER".CYL.FULL_CLOSED AND "DB2810_U1_F4_GRIPPER".CYL.FULL_CLOSED),
                           SP_CLAMPED := "DB2440_GLOBAL_DATA".GLOBAL_DATA.FIX_IN_UNIT_01_STA_4_CLAMPED OR "DB1030_TEST_STOP".TEST_STP_SQ_IN_PROCESS OR ("DB4000_FIX_TABLE_POSITIONS".UNIT_01.AXIS_E10_NOT_DEFINED_POS AND "DB2510_U1_F1_GRIPPER".CYL.FULL_CLOSED AND "DB2610_U1_F2_GRIPPER".CYL.FULL_CLOSED AND "DB2710_U1_F3_GRIPPER".CYL.FULL_CLOSED AND "DB2810_U1_F4_GRIPPER".CYL.FULL_CLOSED),
                           HARDWARE_ENABLE := true,
                           TOOL_CHANGE_POS := false,
                           FIXTURE_1_PART_OK := "DB8000_PART_STATUS".UNIT_01.STATION_4.PART_A.STATUS.OK,
                           READ_POS := "DB303_CH3_READ_AXES_POSITIONS".readDB.POSITION_AXIS_1,
                           UNIT_ALARM := 1,
                           STATION_ALARM := 4,
                           DESELECT_SPINDLE_STO := "DB1018_SAFETY_TAGS".DESELECT_SPINDLE_STO_01R,
                           SpindleDB := "LBP_Axis6",
                           DELAYED_ENABLE => "DB136_CLADDING_SPINDLE_C14".DELAYED_ENABLE,
                           FEED_HOLD_CONDITIONS => "DB136_CLADDING_SPINDLE_C14".FEED_HOLD_CONDITIONS,
                           FEED_HOLD_CONDITIONS_HMI => "DB136_CLADDING_SPINDLE_C14".FEED_HOLD_CONDITIONS_HMI,
                           SP_DESELECTED => "DB136_CLADDING_SPINDLE_C14".SP_DESELECTED,
                           SPEED_NOT_REACHED_ALARM => "DB426_ALARMS_WARNINGS".GENERAL."700032",
                           BELT_BROKEN_ALARM => "DB426_ALARMS_WARNINGS".GENERAL."700033",
                           COOLING_ALARM => "DB426_ALARMS_WARNINGS".GENERAL."700034",
                           MQL_HP_ALARM => "DB426_ALARMS_WARNINGS".GENERAL."700035",
                           HIGH_TEMP_ALARM => "DB426_ALARMS_WARNINGS".GENERAL."700036",
                           HIGH_TEMP_PTC_ALARM => "DB426_ALARMS_WARNINGS".GENERAL."700037",
                           VPM_READY_ALARM => "DB426_ALARMS_WARNINGS".GENERAL."700038",
                           HIGH_TEMP_PREALM => "DB426_ALARMS_WARNINGS".WARNINGS."740083",
                           SPINDLE_POS => "DB136_CLADDING_SPINDLE_C14".SPINDLE_POS,
                           HMI_MOTION_EXECUTABILITY_LEFT => "DB505_HMI_SetUp".Setup1.Movement_Executability.movement104ExecutabilityLeft,
                           HMI_MOTION_EXECUTABILITY_RIGHT => "DB505_HMI_SetUp".Setup1.Movement_Executability.movement104ExecutabilityRight,
                           HMI_MOTION_END_POS_LEFT => "DB505_HMI_SetUp".Setup1.Movement_EndPos.movement104EndPosLeft,
                           HMI_MOTION_END_POS_RIGHT => "DB505_HMI_SetUp".Setup1.Movement_EndPos.movement104EndPosRight);
END_REGION

REGION Network 8: SPINDLE C14 OPERATOR HELP
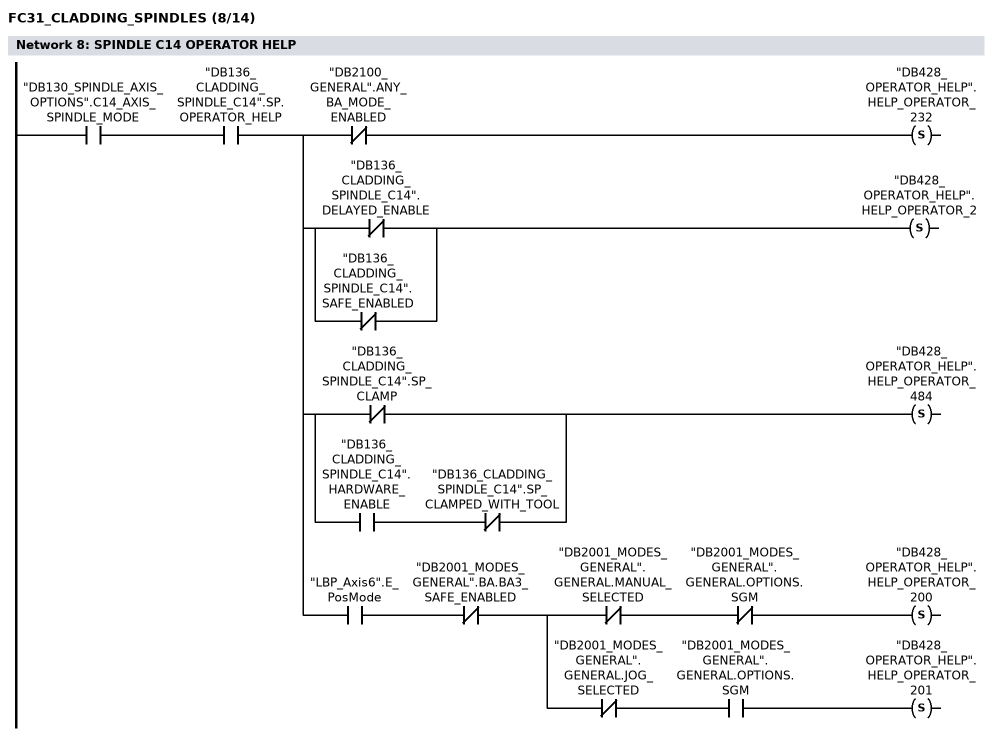
   RUNG wire#powerrail
      Contact( "DB130_SPINDLE_AXIS_OPTIONS".C14_AXIS_SPINDLE_MODE )
      Contact( "DB136_CLADDING_SPINDLE_C14".SP.OPERATOR_HELP )
      wire#w1
      I_Contact( "DB2100_GENERAL".ANY_BA_MODE_ENABLED )
      S_Coil( "DB428_OPERATOR_HELP".HELP_OPERATOR_232 )
   END_RUNG
   RUNG wire#w1
      I_Contact( "DB136_CLADDING_SPINDLE_C14".DELAYED_ENABLE )
      wire#w2
      S_Coil( "DB428_OPERATOR_HELP".HELP_OPERATOR_2 )
   END_RUNG
   RUNG wire#w1
      I_Contact( "DB136_CLADDING_SPINDLE_C14".SAFE_ENABLED )
   END_RUNG wire#w2
   RUNG wire#w1
      I_Contact( "DB136_CLADDING_SPINDLE_C14".SP_CLAMP )
      wire#w3
      S_Coil( "DB428_OPERATOR_HELP".HELP_OPERATOR_484 )
   END_RUNG
   RUNG wire#w1
      Contact( "DB136_CLADDING_SPINDLE_C14".HARDWARE_ENABLE )
      I_Contact( "DB136_CLADDING_SPINDLE_C14".SP_CLAMPED_WITH_TOOL )
   END_RUNG wire#w3
   RUNG wire#w1
      Contact( "LBP_Axis6".E_PosMode )
      I_Contact( "DB2001_MODES_GENERAL".BA.BA3_SAFE_ENABLED )
      wire#w4
      I_Contact( "DB2001_MODES_GENERAL".GENERAL.MANUAL_SELECTED )
      I_Contact( "DB2001_MODES_GENERAL".GENERAL.OPTIONS.SGM )
      S_Coil( "DB428_OPERATOR_HELP".HELP_OPERATOR_200 )
   END_RUNG
   RUNG wire#w4
      I_Contact( "DB2001_MODES_GENERAL".GENERAL.JOG_SELECTED )
      Contact( "DB2001_MODES_GENERAL".GENERAL.OPTIONS.SGM )
      S_Coil( "DB428_OPERATOR_HELP".HELP_OPERATOR_201 )
   END_RUNG
   // the same network as SCL:
   #_w1 := "DB130_SPINDLE_AXIS_OPTIONS".C14_AXIS_SPINDLE_MODE AND "DB136_CLADDING_SPINDLE_C14".SP.OPERATOR_HELP;
   IF #_w1 AND NOT "DB2100_GENERAL".ANY_BA_MODE_ENABLED THEN
       "DB428_OPERATOR_HELP".HELP_OPERATOR_232 := TRUE;
   END_IF;
   IF #_w1 AND (NOT "DB136_CLADDING_SPINDLE_C14".DELAYED_ENABLE OR NOT "DB136_CLADDING_SPINDLE_C14".SAFE_ENABLED) THEN
       "DB428_OPERATOR_HELP".HELP_OPERATOR_2 := TRUE;
   END_IF;
   IF #_w1 AND (NOT "DB136_CLADDING_SPINDLE_C14".SP_CLAMP OR ("DB136_CLADDING_SPINDLE_C14".HARDWARE_ENABLE AND NOT "DB136_CLADDING_SPINDLE_C14".SP_CLAMPED_WITH_TOOL)) THEN
       "DB428_OPERATOR_HELP".HELP_OPERATOR_484 := TRUE;
   END_IF;
   #_w2 := #_w1 AND "LBP_Axis6".E_PosMode AND NOT "DB2001_MODES_GENERAL".BA.BA3_SAFE_ENABLED;
   IF #_w2 AND NOT "DB2001_MODES_GENERAL".GENERAL.MANUAL_SELECTED AND NOT "DB2001_MODES_GENERAL".GENERAL.OPTIONS.SGM THEN
       "DB428_OPERATOR_HELP".HELP_OPERATOR_200 := TRUE;
   END_IF;
   IF #_w2 AND NOT "DB2001_MODES_GENERAL".GENERAL.JOG_SELECTED AND "DB2001_MODES_GENERAL".GENERAL.OPTIONS.SGM THEN
       "DB428_OPERATOR_HELP".HELP_OPERATOR_201 := TRUE;
   END_IF;
END_REGION

REGION Network 9: CALL FB31 SPINDLE C21
   // 2#0000_0001 OPTIONS 0 BIT 0 MEASURING SYSTEM 2 OPTION
   // 2#0000_0010 OPTIONS 0 BIT 1 BELT BROKEN OPTION
   // 2#0000_0100 OPTIONS 0 BIT 2 COOLING OPTION
   // 2#0000_1000 OPTIONS 0 BIT 3 MQL OR HP OPTION
   // 2#0001_0000 OPTIONS 0 BIT 4 ANALOG TEMPERATURE SENSOR OPTION
   // 2#0010_0000 OPTIONS 0 BIT 5 PTC TEMPERATURE SENSOR OPTION
   // 2#0100_0000 OPTIONS 0 BIT 6 TWIN KESSLER VPM READY OPTION
   // 2#1000_0000 OPTIONS 0 BIT 7 MPP SPINDLE OVERRIDE OPTION
   // 
   // 2#0000_0001 OPTIONS 1 BIT 0 SPARE OPTION
   // 2#0000_0010 OPTIONS 1 BIT 1 SPARE OPTION
   // 2#0000_0100 OPTIONS 1 BIT 2 SPARE OPTION
   // 2#0000_1000 OPTIONS 1 BIT 3 SPARE OPTION
   // 2#0001_0000 OPTIONS 1 BIT 4 SPARE OPTION
   // 2#0010_0000 OPTIONS 1 BIT 5 SPARE OPTION
   // 2#0100_0000 OPTIONS 1 BIT 6 SPARE OPTION
   // 2#1000_0000 OPTIONS 1 BIT 7 SPARE OPTION
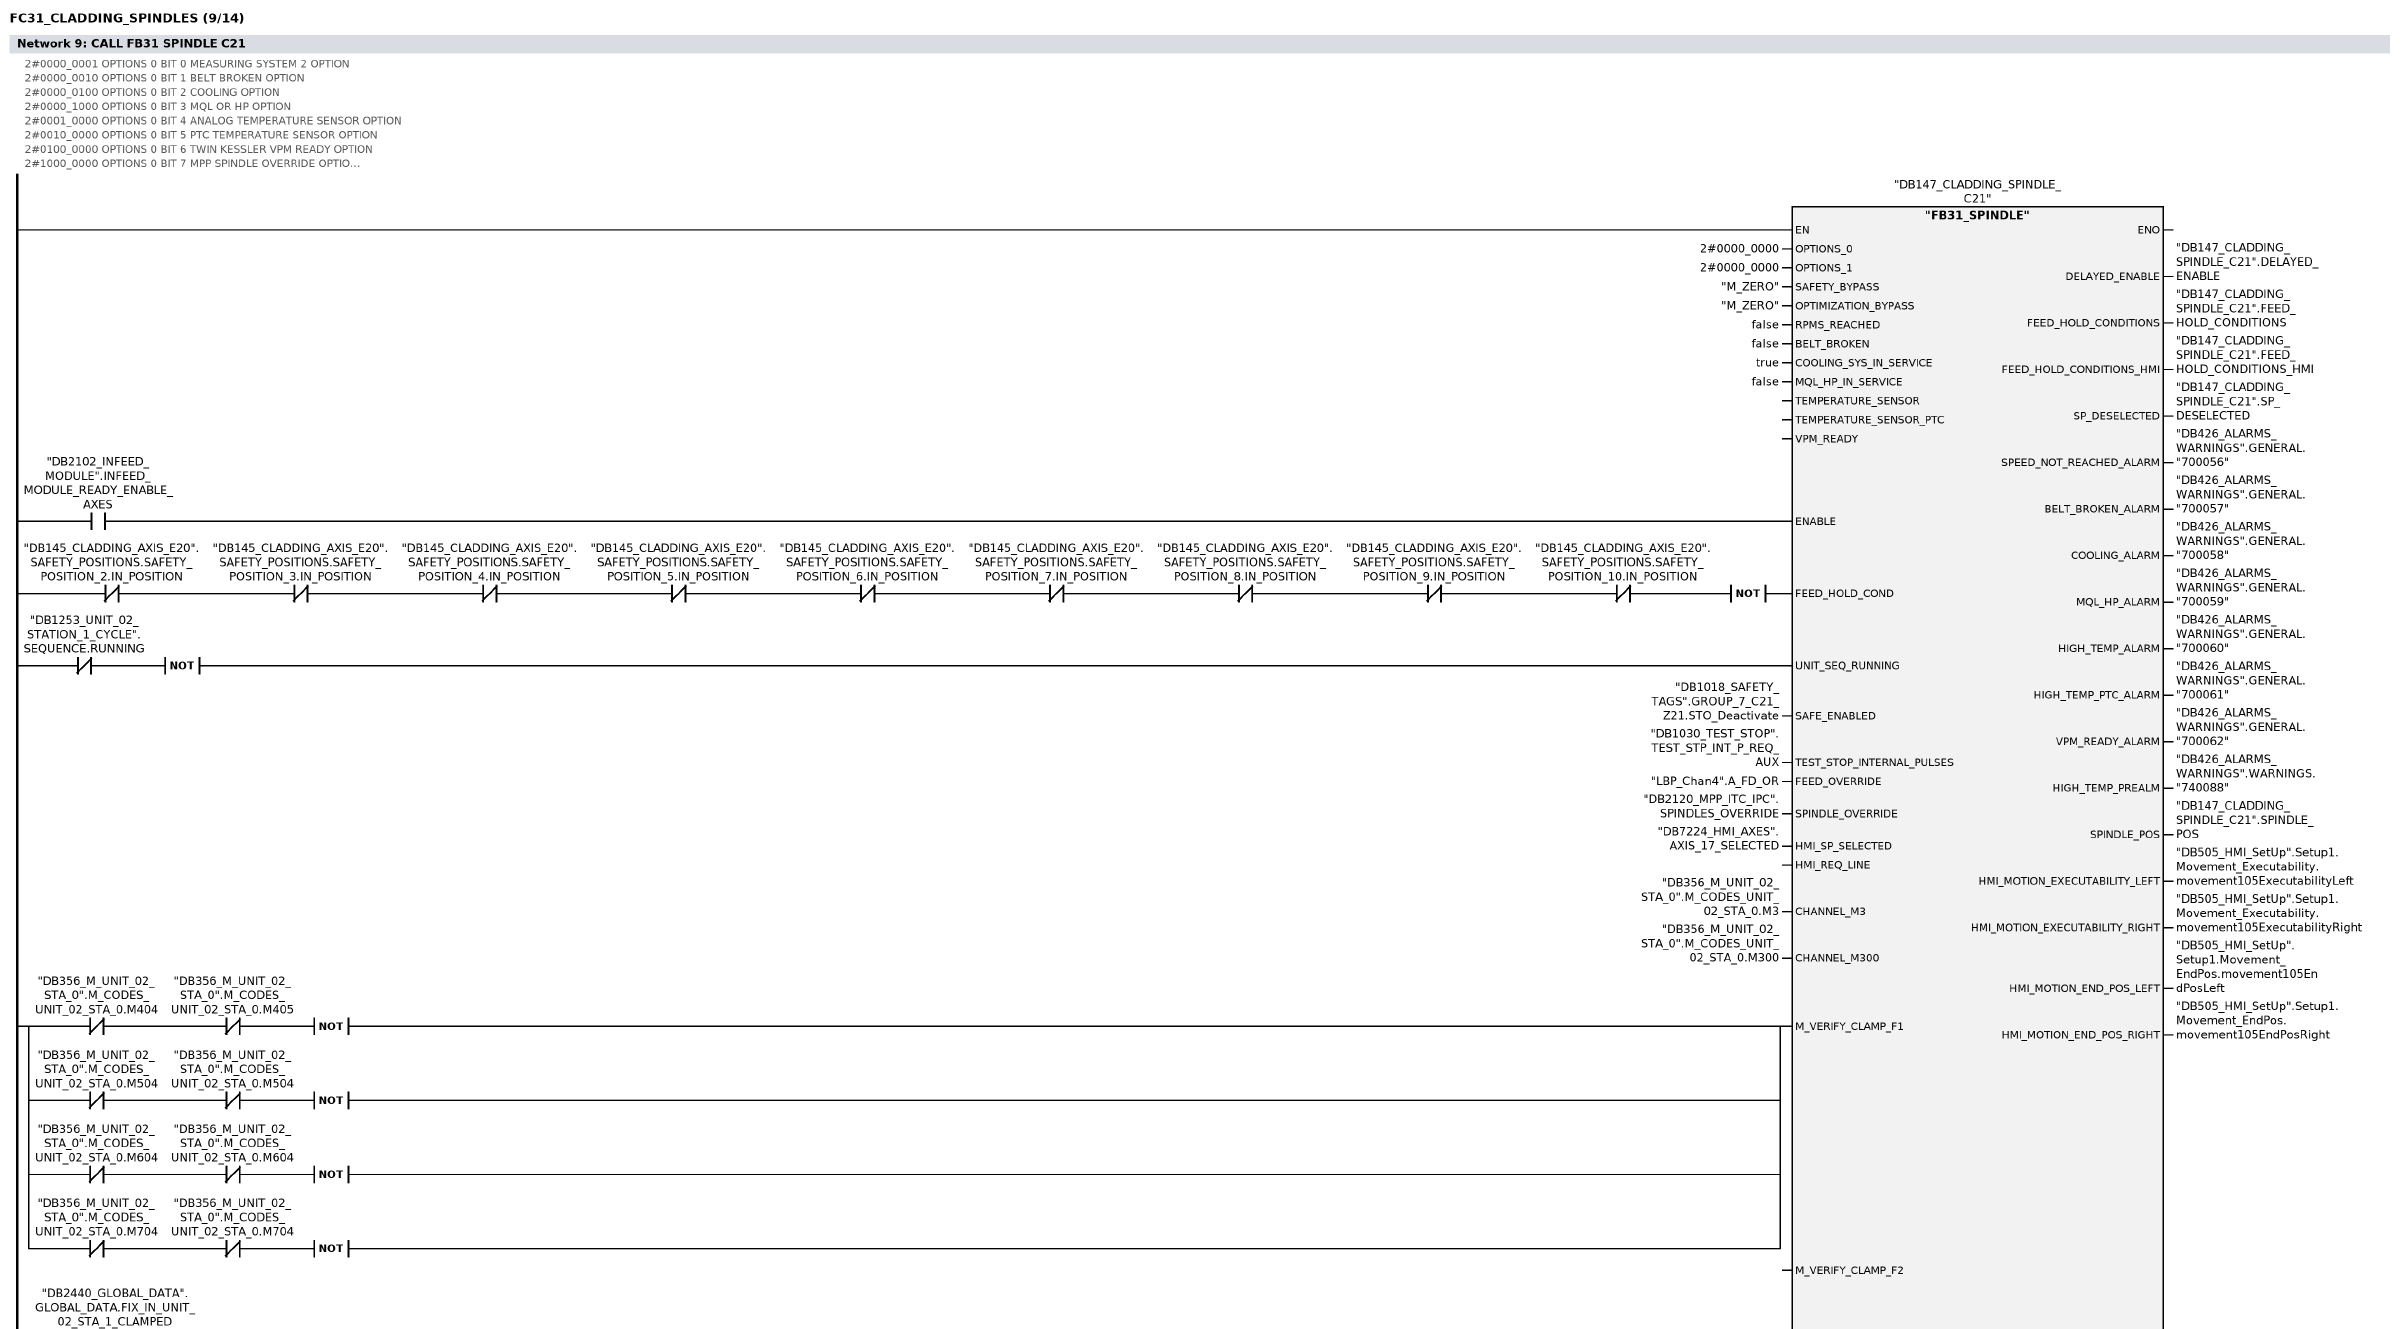
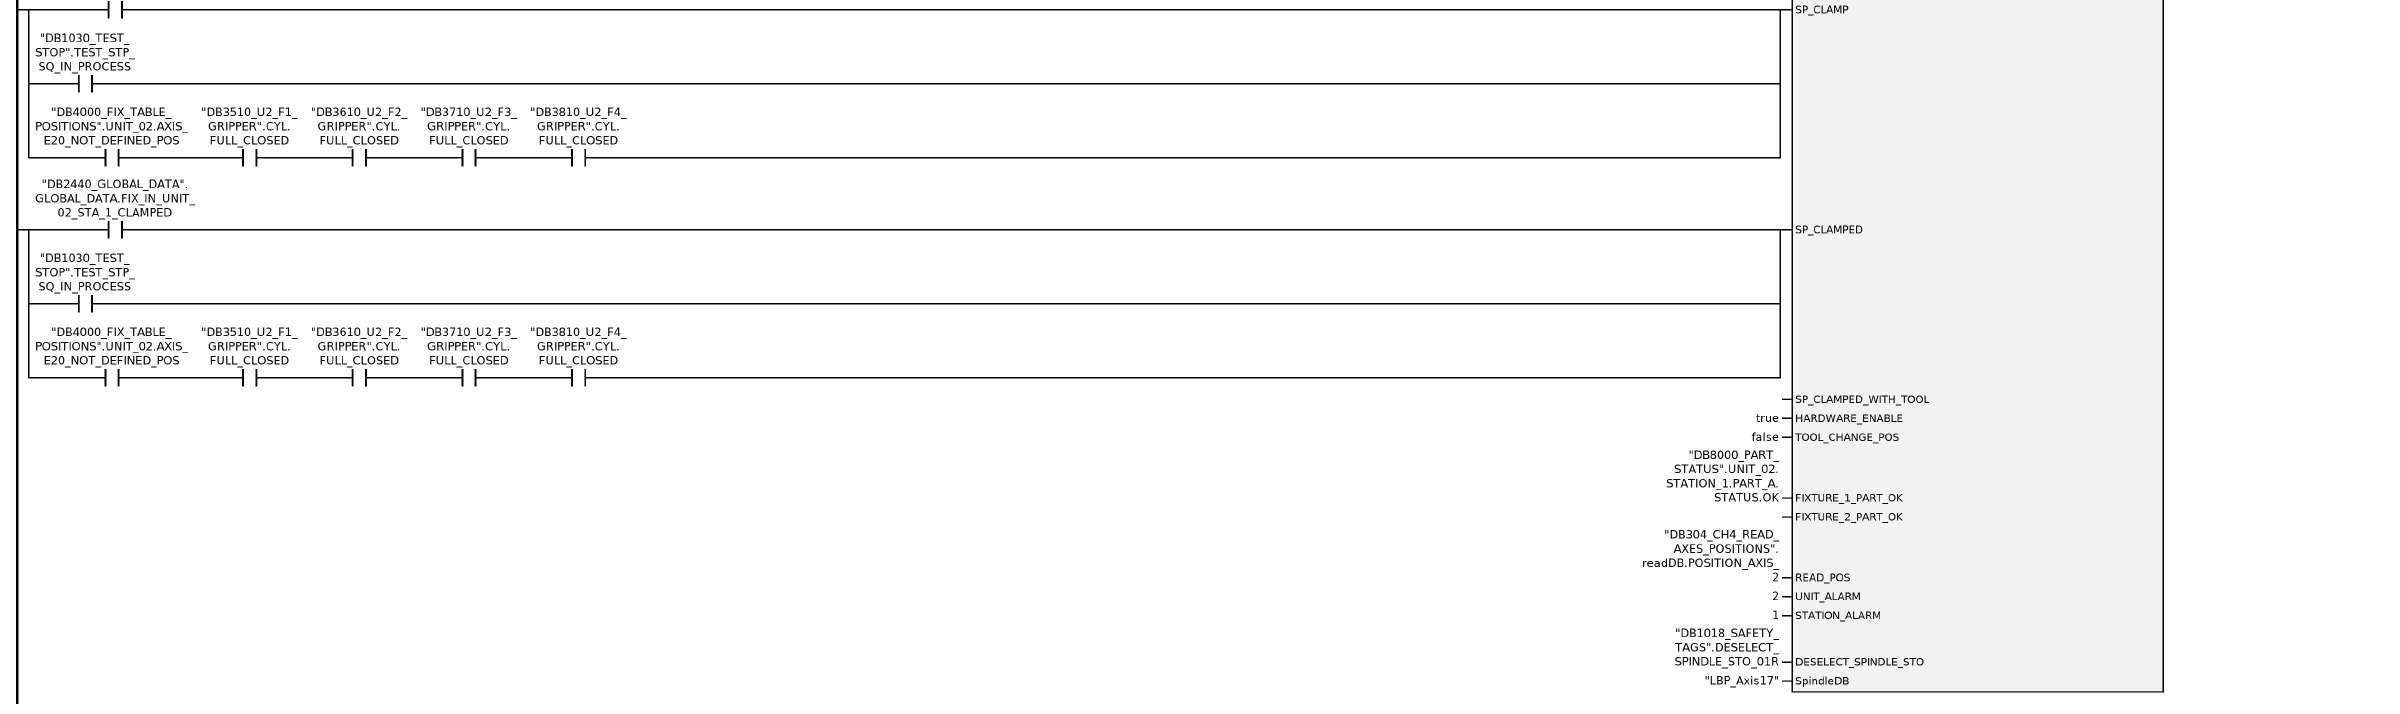
   RUNG wire#powerrail
      "DB147_CLADDING_SPINDLE_C21"(ENABLE := wire#w1, FEED_HOLD_COND := wire#w2, UNIT_SEQ_RUNNING := wire#w3, M_VERIFY_CLAMP_F1 := wire#w4, SP_CLAMP := wire#w5, SP_CLAMPED := wire#w6, OPTIONS_0 := 2#0000_0000, OPTIONS_1 := 2#0000_0000, SAFETY_BYPASS := "M_ZERO", OPTIMIZATION_BYPASS := "M_ZERO", RPMS_REACHED := false, BELT_BROKEN := false, COOLING_SYS_IN_SERVICE := true, MQL_HP_IN_SERVICE := false, TEMPERATURE_SENSOR :=, TEMPERATURE_SENSOR_PTC :=, VPM_READY :=, SAFE_ENABLED := "DB1018_SAFETY_TAGS".GROUP_7_C21_Z21.STO_Deactivate, TEST_STOP_INTERNAL_PULSES := "DB1030_TEST_STOP".TEST_STP_INT_P_REQ_AUX, FEED_OVERRIDE := "LBP_Chan4".A_FD_OR, SPINDLE_OVERRIDE := "DB2120_MPP_ITC_IPC".SPINDLES_OVERRIDE, HMI_SP_SELECTED := "DB7224_HMI_AXES".AXIS_17_SELECTED, HMI_REQ_LINE :=, CHANNEL_M3 := "DB356_M_UNIT_02_STA_0".M_CODES_UNIT_02_STA_0.M3, CHANNEL_M300 := "DB356_M_UNIT_02_STA_0".M_CODES_UNIT_02_STA_0.M300, M_VERIFY_CLAMP_F2 :=, SP_CLAMPED_WITH_TOOL :=, HARDWARE_ENABLE := true, TOOL_CHANGE_POS := false, FIXTURE_1_PART_OK := "DB8000_PART_STATUS".UNIT_02.STATION_1.PART_A.STATUS.OK, FIXTURE_2_PART_OK :=, READ_POS := "DB304_CH4_READ_AXES_POSITIONS".readDB.POSITION_AXIS_2, UNIT_ALARM := 2, STATION_ALARM := 1, DESELECT_SPINDLE_STO := "DB1018_SAFETY_TAGS".DESELECT_SPINDLE_STO_01R, SpindleDB := "LBP_Axis17", DELAYED_ENABLE => "DB147_CLADDING_SPINDLE_C21".DELAYED_ENABLE, FEED_HOLD_CONDITIONS => "DB147_CLADDING_SPINDLE_C21".FEED_HOLD_CONDITIONS, FEED_HOLD_CONDITIONS_HMI => "DB147_CLADDING_SPINDLE_C21".FEED_HOLD_CONDITIONS_HMI, SP_DESELECTED => "DB147_CLADDING_SPINDLE_C21".SP_DESELECTED, SPEED_NOT_REACHED_ALARM => "DB426_ALARMS_WARNINGS".GENERAL."700056", BELT_BROKEN_ALARM => "DB426_ALARMS_WARNINGS".GENERAL."700057", COOLING_ALARM => "DB426_ALARMS_WARNINGS".GENERAL."700058", MQL_HP_ALARM => "DB426_ALARMS_WARNINGS".GENERAL."700059", HIGH_TEMP_ALARM => "DB426_ALARMS_WARNINGS".GENERAL."700060", HIGH_TEMP_PTC_ALARM => "DB426_ALARMS_WARNINGS".GENERAL."700061", VPM_READY_ALARM => "DB426_ALARMS_WARNINGS".GENERAL."700062", HIGH_TEMP_PREALM => "DB426_ALARMS_WARNINGS".WARNINGS."740088", SPINDLE_POS => "DB147_CLADDING_SPINDLE_C21".SPINDLE_POS, HMI_MOTION_EXECUTABILITY_LEFT => "DB505_HMI_SetUp".Setup1.Movement_Executability.movement105ExecutabilityLeft, HMI_MOTION_EXECUTABILITY_RIGHT => "DB505_HMI_SetUp".Setup1.Movement_Executability.movement105ExecutabilityRight, HMI_MOTION_END_POS_LEFT => "DB505_HMI_SetUp".Setup1.Movement_EndPos.movement105EndPosLeft, HMI_MOTION_END_POS_RIGHT => "DB505_HMI_SetUp".Setup1.Movement_EndPos.movement105EndPosRight)
   END_RUNG
   RUNG wire#powerrail
      Contact( "DB2102_INFEED_MODULE".INFEED_MODULE_READY_ENABLE_AXES )
   END_RUNG wire#w1
   RUNG wire#powerrail
      I_Contact( "DB145_CLADDING_AXIS_E20".SAFETY_POSITIONS.SAFETY_POSITION_2.IN_POSITION )
      I_Contact( "DB145_CLADDING_AXIS_E20".SAFETY_POSITIONS.SAFETY_POSITION_3.IN_POSITION )
      I_Contact( "DB145_CLADDING_AXIS_E20".SAFETY_POSITIONS.SAFETY_POSITION_4.IN_POSITION )
      I_Contact( "DB145_CLADDING_AXIS_E20".SAFETY_POSITIONS.SAFETY_POSITION_5.IN_POSITION )
      I_Contact( "DB145_CLADDING_AXIS_E20".SAFETY_POSITIONS.SAFETY_POSITION_6.IN_POSITION )
      I_Contact( "DB145_CLADDING_AXIS_E20".SAFETY_POSITIONS.SAFETY_POSITION_7.IN_POSITION )
      I_Contact( "DB145_CLADDING_AXIS_E20".SAFETY_POSITIONS.SAFETY_POSITION_8.IN_POSITION )
      I_Contact( "DB145_CLADDING_AXIS_E20".SAFETY_POSITIONS.SAFETY_POSITION_9.IN_POSITION )
      I_Contact( "DB145_CLADDING_AXIS_E20".SAFETY_POSITIONS.SAFETY_POSITION_10.IN_POSITION )
      Not()
   END_RUNG wire#w2
   RUNG wire#powerrail
      I_Contact( "DB1253_UNIT_02_STATION_1_CYCLE".SEQUENCE.RUNNING )
      Not()
   END_RUNG wire#w3
   RUNG wire#powerrail
      I_Contact( "DB356_M_UNIT_02_STA_0".M_CODES_UNIT_02_STA_0.M404 )
      I_Contact( "DB356_M_UNIT_02_STA_0".M_CODES_UNIT_02_STA_0.M405 )
      Not()
   END_RUNG wire#w4
   RUNG wire#powerrail
      I_Contact( "DB356_M_UNIT_02_STA_0".M_CODES_UNIT_02_STA_0.M504 )
      I_Contact( "DB356_M_UNIT_02_STA_0".M_CODES_UNIT_02_STA_0.M504 )
      Not()
   END_RUNG wire#w4
   RUNG wire#powerrail
      I_Contact( "DB356_M_UNIT_02_STA_0".M_CODES_UNIT_02_STA_0.M604 )
      I_Contact( "DB356_M_UNIT_02_STA_0".M_CODES_UNIT_02_STA_0.M604 )
      Not()
   END_RUNG wire#w4
   RUNG wire#powerrail
      I_Contact( "DB356_M_UNIT_02_STA_0".M_CODES_UNIT_02_STA_0.M704 )
      I_Contact( "DB356_M_UNIT_02_STA_0".M_CODES_UNIT_02_STA_0.M704 )
      Not()
   END_RUNG wire#w4
   RUNG wire#powerrail
      Contact( "DB2440_GLOBAL_DATA".GLOBAL_DATA.FIX_IN_UNIT_02_STA_1_CLAMPED )
   END_RUNG wire#w5
   RUNG wire#powerrail
      Contact( "DB1030_TEST_STOP".TEST_STP_SQ_IN_PROCESS )
   END_RUNG wire#w5
   RUNG wire#powerrail
      Contact( "DB4000_FIX_TABLE_POSITIONS".UNIT_02.AXIS_E20_NOT_DEFINED_POS )
      Contact( "DB3510_U2_F1_GRIPPER".CYL.FULL_CLOSED )
      Contact( "DB3610_U2_F2_GRIPPER".CYL.FULL_CLOSED )
      Contact( "DB3710_U2_F3_GRIPPER".CYL.FULL_CLOSED )
      Contact( "DB3810_U2_F4_GRIPPER".CYL.FULL_CLOSED )
   END_RUNG wire#w5
   RUNG wire#powerrail
      Contact( "DB2440_GLOBAL_DATA".GLOBAL_DATA.FIX_IN_UNIT_02_STA_1_CLAMPED )
   END_RUNG wire#w6
   RUNG wire#powerrail
      Contact( "DB1030_TEST_STOP".TEST_STP_SQ_IN_PROCESS )
   END_RUNG wire#w6
   RUNG wire#powerrail
      Contact( "DB4000_FIX_TABLE_POSITIONS".UNIT_02.AXIS_E20_NOT_DEFINED_POS )
      Contact( "DB3510_U2_F1_GRIPPER".CYL.FULL_CLOSED )
      Contact( "DB3610_U2_F2_GRIPPER".CYL.FULL_CLOSED )
      Contact( "DB3710_U2_F3_GRIPPER".CYL.FULL_CLOSED )
      Contact( "DB3810_U2_F4_GRIPPER".CYL.FULL_CLOSED )
   END_RUNG wire#w6
   // the same network as SCL:
   "DB147_CLADDING_SPINDLE_C21"(OPTIONS_0 := 2#0000_0000,   // "FB31_SPINDLE"
                           OPTIONS_1 := 2#0000_0000,
                           SAFETY_BYPASS := "M_ZERO",
                           OPTIMIZATION_BYPASS := "M_ZERO",
                           RPMS_REACHED := false,
                           BELT_BROKEN := false,
                           COOLING_SYS_IN_SERVICE := true,
                           MQL_HP_IN_SERVICE := false,
                           ENABLE := "DB2102_INFEED_MODULE".INFEED_MODULE_READY_ENABLE_AXES,
                           FEED_HOLD_COND := NOT (NOT "DB145_CLADDING_AXIS_E20".SAFETY_POSITIONS.SAFETY_POSITION_2.IN_POSITION AND NOT "DB145_CLADDING_AXIS_E20".SAFETY_POSITIONS.SAFETY_POSITION_3.IN_POSITION AND NOT "DB145_CLADDING_AXIS_E20".SAFETY_POSITIONS.SAFETY_POSITION_4.IN_POSITION AND NOT "DB145_CLADDING_AXIS_E20".SAFETY_POSITIONS.SAFETY_POSITION_5.IN_POSITION AND NOT "DB145_CLADDING_AXIS_E20".SAFETY_POSITIONS.SAFETY_POSITION_6.IN_POSITION AND NOT "DB145_CLADDING_AXIS_E20".SAFETY_POSITIONS.SAFETY_POSITION_7.IN_POSITION AND NOT "DB145_CLADDING_AXIS_E20".SAFETY_POSITIONS.SAFETY_POSITION_8.IN_POSITION AND NOT "DB145_CLADDING_AXIS_E20".SAFETY_POSITIONS.SAFETY_POSITION_9.IN_POSITION AND NOT "DB145_CLADDING_AXIS_E20".SAFETY_POSITIONS.SAFETY_POSITION_10.IN_POSITION),
                           UNIT_SEQ_RUNNING := NOT (NOT "DB1253_UNIT_02_STATION_1_CYCLE".SEQUENCE.RUNNING),
                           SAFE_ENABLED := "DB1018_SAFETY_TAGS".GROUP_7_C21_Z21.STO_Deactivate,
                           TEST_STOP_INTERNAL_PULSES := "DB1030_TEST_STOP".TEST_STP_INT_P_REQ_AUX,
                           FEED_OVERRIDE := "LBP_Chan4".A_FD_OR,
                           SPINDLE_OVERRIDE := "DB2120_MPP_ITC_IPC".SPINDLES_OVERRIDE,
                           HMI_SP_SELECTED := "DB7224_HMI_AXES".AXIS_17_SELECTED,
                           CHANNEL_M3 := "DB356_M_UNIT_02_STA_0".M_CODES_UNIT_02_STA_0.M3,
                           CHANNEL_M300 := "DB356_M_UNIT_02_STA_0".M_CODES_UNIT_02_STA_0.M300,
                           M_VERIFY_CLAMP_F1 := NOT (NOT "DB356_M_UNIT_02_STA_0".M_CODES_UNIT_02_STA_0.M404 AND NOT "DB356_M_UNIT_02_STA_0".M_CODES_UNIT_02_STA_0.M405) OR NOT (NOT "DB356_M_UNIT_02_STA_0".M_CODES_UNIT_02_STA_0.M504 AND NOT "DB356_M_UNIT_02_STA_0".M_CODES_UNIT_02_STA_0.M504) OR NOT (NOT "DB356_M_UNIT_02_STA_0".M_CODES_UNIT_02_STA_0.M604 AND NOT "DB356_M_UNIT_02_STA_0".M_CODES_UNIT_02_STA_0.M604) OR NOT (NOT "DB356_M_UNIT_02_STA_0".M_CODES_UNIT_02_STA_0.M704 AND NOT "DB356_M_UNIT_02_STA_0".M_CODES_UNIT_02_STA_0.M704),
                           SP_CLAMP := "DB2440_GLOBAL_DATA".GLOBAL_DATA.FIX_IN_UNIT_02_STA_1_CLAMPED OR "DB1030_TEST_STOP".TEST_STP_SQ_IN_PROCESS OR ("DB4000_FIX_TABLE_POSITIONS".UNIT_02.AXIS_E20_NOT_DEFINED_POS AND "DB3510_U2_F1_GRIPPER".CYL.FULL_CLOSED AND "DB3610_U2_F2_GRIPPER".CYL.FULL_CLOSED AND "DB3710_U2_F3_GRIPPER".CYL.FULL_CLOSED AND "DB3810_U2_F4_GRIPPER".CYL.FULL_CLOSED),
                           SP_CLAMPED := "DB2440_GLOBAL_DATA".GLOBAL_DATA.FIX_IN_UNIT_02_STA_1_CLAMPED OR "DB1030_TEST_STOP".TEST_STP_SQ_IN_PROCESS OR ("DB4000_FIX_TABLE_POSITIONS".UNIT_02.AXIS_E20_NOT_DEFINED_POS AND "DB3510_U2_F1_GRIPPER".CYL.FULL_CLOSED AND "DB3610_U2_F2_GRIPPER".CYL.FULL_CLOSED AND "DB3710_U2_F3_GRIPPER".CYL.FULL_CLOSED AND "DB3810_U2_F4_GRIPPER".CYL.FULL_CLOSED),
                           HARDWARE_ENABLE := true,
                           TOOL_CHANGE_POS := false,
                           FIXTURE_1_PART_OK := "DB8000_PART_STATUS".UNIT_02.STATION_1.PART_A.STATUS.OK,
                           READ_POS := "DB304_CH4_READ_AXES_POSITIONS".readDB.POSITION_AXIS_2,
                           UNIT_ALARM := 2,
                           STATION_ALARM := 1,
                           DESELECT_SPINDLE_STO := "DB1018_SAFETY_TAGS".DESELECT_SPINDLE_STO_01R,
                           SpindleDB := "LBP_Axis17",
                           DELAYED_ENABLE => "DB147_CLADDING_SPINDLE_C21".DELAYED_ENABLE,
                           FEED_HOLD_CONDITIONS => "DB147_CLADDING_SPINDLE_C21".FEED_HOLD_CONDITIONS,
                           FEED_HOLD_CONDITIONS_HMI => "DB147_CLADDING_SPINDLE_C21".FEED_HOLD_CONDITIONS_HMI,
                           SP_DESELECTED => "DB147_CLADDING_SPINDLE_C21".SP_DESELECTED,
                           SPEED_NOT_REACHED_ALARM => "DB426_ALARMS_WARNINGS".GENERAL."700056",
                           BELT_BROKEN_ALARM => "DB426_ALARMS_WARNINGS".GENERAL."700057",
                           COOLING_ALARM => "DB426_ALARMS_WARNINGS".GENERAL."700058",
                           MQL_HP_ALARM => "DB426_ALARMS_WARNINGS".GENERAL."700059",
                           HIGH_TEMP_ALARM => "DB426_ALARMS_WARNINGS".GENERAL."700060",
                           HIGH_TEMP_PTC_ALARM => "DB426_ALARMS_WARNINGS".GENERAL."700061",
                           VPM_READY_ALARM => "DB426_ALARMS_WARNINGS".GENERAL."700062",
                           HIGH_TEMP_PREALM => "DB426_ALARMS_WARNINGS".WARNINGS."740088",
                           SPINDLE_POS => "DB147_CLADDING_SPINDLE_C21".SPINDLE_POS,
                           HMI_MOTION_EXECUTABILITY_LEFT => "DB505_HMI_SetUp".Setup1.Movement_Executability.movement105ExecutabilityLeft,
                           HMI_MOTION_EXECUTABILITY_RIGHT => "DB505_HMI_SetUp".Setup1.Movement_Executability.movement105ExecutabilityRight,
                           HMI_MOTION_END_POS_LEFT => "DB505_HMI_SetUp".Setup1.Movement_EndPos.movement105EndPosLeft,
                           HMI_MOTION_END_POS_RIGHT => "DB505_HMI_SetUp".Setup1.Movement_EndPos.movement105EndPosRight);
END_REGION

REGION Network 10: SPINDLE C21 OPERATOR HELP
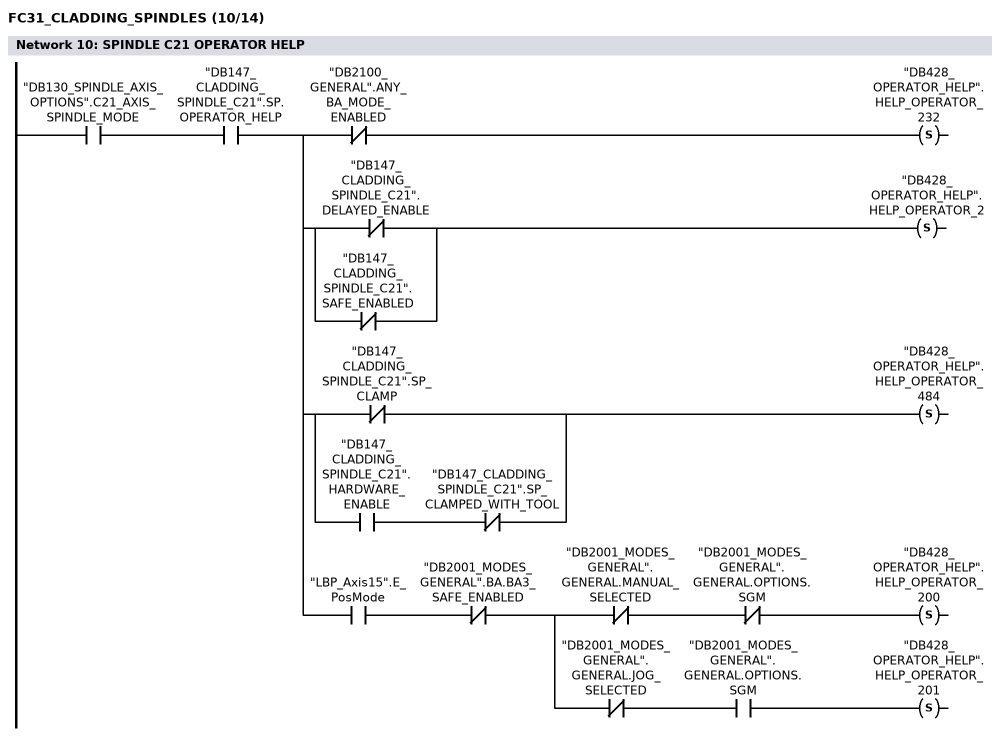
   RUNG wire#powerrail
      Contact( "DB130_SPINDLE_AXIS_OPTIONS".C21_AXIS_SPINDLE_MODE )
      Contact( "DB147_CLADDING_SPINDLE_C21".SP.OPERATOR_HELP )
      wire#w1
      I_Contact( "DB2100_GENERAL".ANY_BA_MODE_ENABLED )
      S_Coil( "DB428_OPERATOR_HELP".HELP_OPERATOR_232 )
   END_RUNG
   RUNG wire#w1
      I_Contact( "DB147_CLADDING_SPINDLE_C21".DELAYED_ENABLE )
      wire#w2
      S_Coil( "DB428_OPERATOR_HELP".HELP_OPERATOR_2 )
   END_RUNG
   RUNG wire#w1
      I_Contact( "DB147_CLADDING_SPINDLE_C21".SAFE_ENABLED )
   END_RUNG wire#w2
   RUNG wire#w1
      I_Contact( "DB147_CLADDING_SPINDLE_C21".SP_CLAMP )
      wire#w3
      S_Coil( "DB428_OPERATOR_HELP".HELP_OPERATOR_484 )
   END_RUNG
   RUNG wire#w1
      Contact( "DB147_CLADDING_SPINDLE_C21".HARDWARE_ENABLE )
      I_Contact( "DB147_CLADDING_SPINDLE_C21".SP_CLAMPED_WITH_TOOL )
   END_RUNG wire#w3
   RUNG wire#w1
      Contact( "LBP_Axis15".E_PosMode )
      I_Contact( "DB2001_MODES_GENERAL".BA.BA3_SAFE_ENABLED )
      wire#w4
      I_Contact( "DB2001_MODES_GENERAL".GENERAL.MANUAL_SELECTED )
      I_Contact( "DB2001_MODES_GENERAL".GENERAL.OPTIONS.SGM )
      S_Coil( "DB428_OPERATOR_HELP".HELP_OPERATOR_200 )
   END_RUNG
   RUNG wire#w4
      I_Contact( "DB2001_MODES_GENERAL".GENERAL.JOG_SELECTED )
      Contact( "DB2001_MODES_GENERAL".GENERAL.OPTIONS.SGM )
      S_Coil( "DB428_OPERATOR_HELP".HELP_OPERATOR_201 )
   END_RUNG
   // the same network as SCL:
   #_w1 := "DB130_SPINDLE_AXIS_OPTIONS".C21_AXIS_SPINDLE_MODE AND "DB147_CLADDING_SPINDLE_C21".SP.OPERATOR_HELP;
   IF #_w1 AND NOT "DB2100_GENERAL".ANY_BA_MODE_ENABLED THEN
       "DB428_OPERATOR_HELP".HELP_OPERATOR_232 := TRUE;
   END_IF;
   IF #_w1 AND (NOT "DB147_CLADDING_SPINDLE_C21".DELAYED_ENABLE OR NOT "DB147_CLADDING_SPINDLE_C21".SAFE_ENABLED) THEN
       "DB428_OPERATOR_HELP".HELP_OPERATOR_2 := TRUE;
   END_IF;
   IF #_w1 AND (NOT "DB147_CLADDING_SPINDLE_C21".SP_CLAMP OR ("DB147_CLADDING_SPINDLE_C21".HARDWARE_ENABLE AND NOT "DB147_CLADDING_SPINDLE_C21".SP_CLAMPED_WITH_TOOL)) THEN
       "DB428_OPERATOR_HELP".HELP_OPERATOR_484 := TRUE;
   END_IF;
   #_w2 := #_w1 AND "LBP_Axis15".E_PosMode AND NOT "DB2001_MODES_GENERAL".BA.BA3_SAFE_ENABLED;
   IF #_w2 AND NOT "DB2001_MODES_GENERAL".GENERAL.MANUAL_SELECTED AND NOT "DB2001_MODES_GENERAL".GENERAL.OPTIONS.SGM THEN
       "DB428_OPERATOR_HELP".HELP_OPERATOR_200 := TRUE;
   END_IF;
   IF #_w2 AND NOT "DB2001_MODES_GENERAL".GENERAL.JOG_SELECTED AND "DB2001_MODES_GENERAL".GENERAL.OPTIONS.SGM THEN
       "DB428_OPERATOR_HELP".HELP_OPERATOR_201 := TRUE;
   END_IF;
END_REGION

REGION Network 11: CALL FB31 SPINDLE C23
   // 2#0000_0001 OPTIONS 0 BIT 0 MEASURING SYSTEM 2 OPTION
   // 2#0000_0010 OPTIONS 0 BIT 1 BELT BROKEN OPTION
   // 2#0000_0100 OPTIONS 0 BIT 2 COOLING OPTION
   // 2#0000_1000 OPTIONS 0 BIT 3 MQL OR HP OPTION
   // 2#0001_0000 OPTIONS 0 BIT 4 ANALOG TEMPERATURE SENSOR OPTION
   // 2#0010_0000 OPTIONS 0 BIT 5 PTC TEMPERATURE SENSOR OPTION
   // 2#0100_0000 OPTIONS 0 BIT 6 TWIN KESSLER VPM READY OPTION
   // 2#1000_0000 OPTIONS 0 BIT 7 MPP SPINDLE OVERRIDE OPTION
   // 
   // 2#0000_0001 OPTIONS 1 BIT 0 SPARE OPTION
   // 2#0000_0010 OPTIONS 1 BIT 1 SPARE OPTION
   // 2#0000_0100 OPTIONS 1 BIT 2 SPARE OPTION
   // 2#0000_1000 OPTIONS 1 BIT 3 SPARE OPTION
   // 2#0001_0000 OPTIONS 1 BIT 4 SPARE OPTION
   // 2#0010_0000 OPTIONS 1 BIT 5 SPARE OPTION
   // 2#0100_0000 OPTIONS 1 BIT 6 SPARE OPTION
   // 2#1000_0000 OPTIONS 1 BIT 7 SPARE OPTION
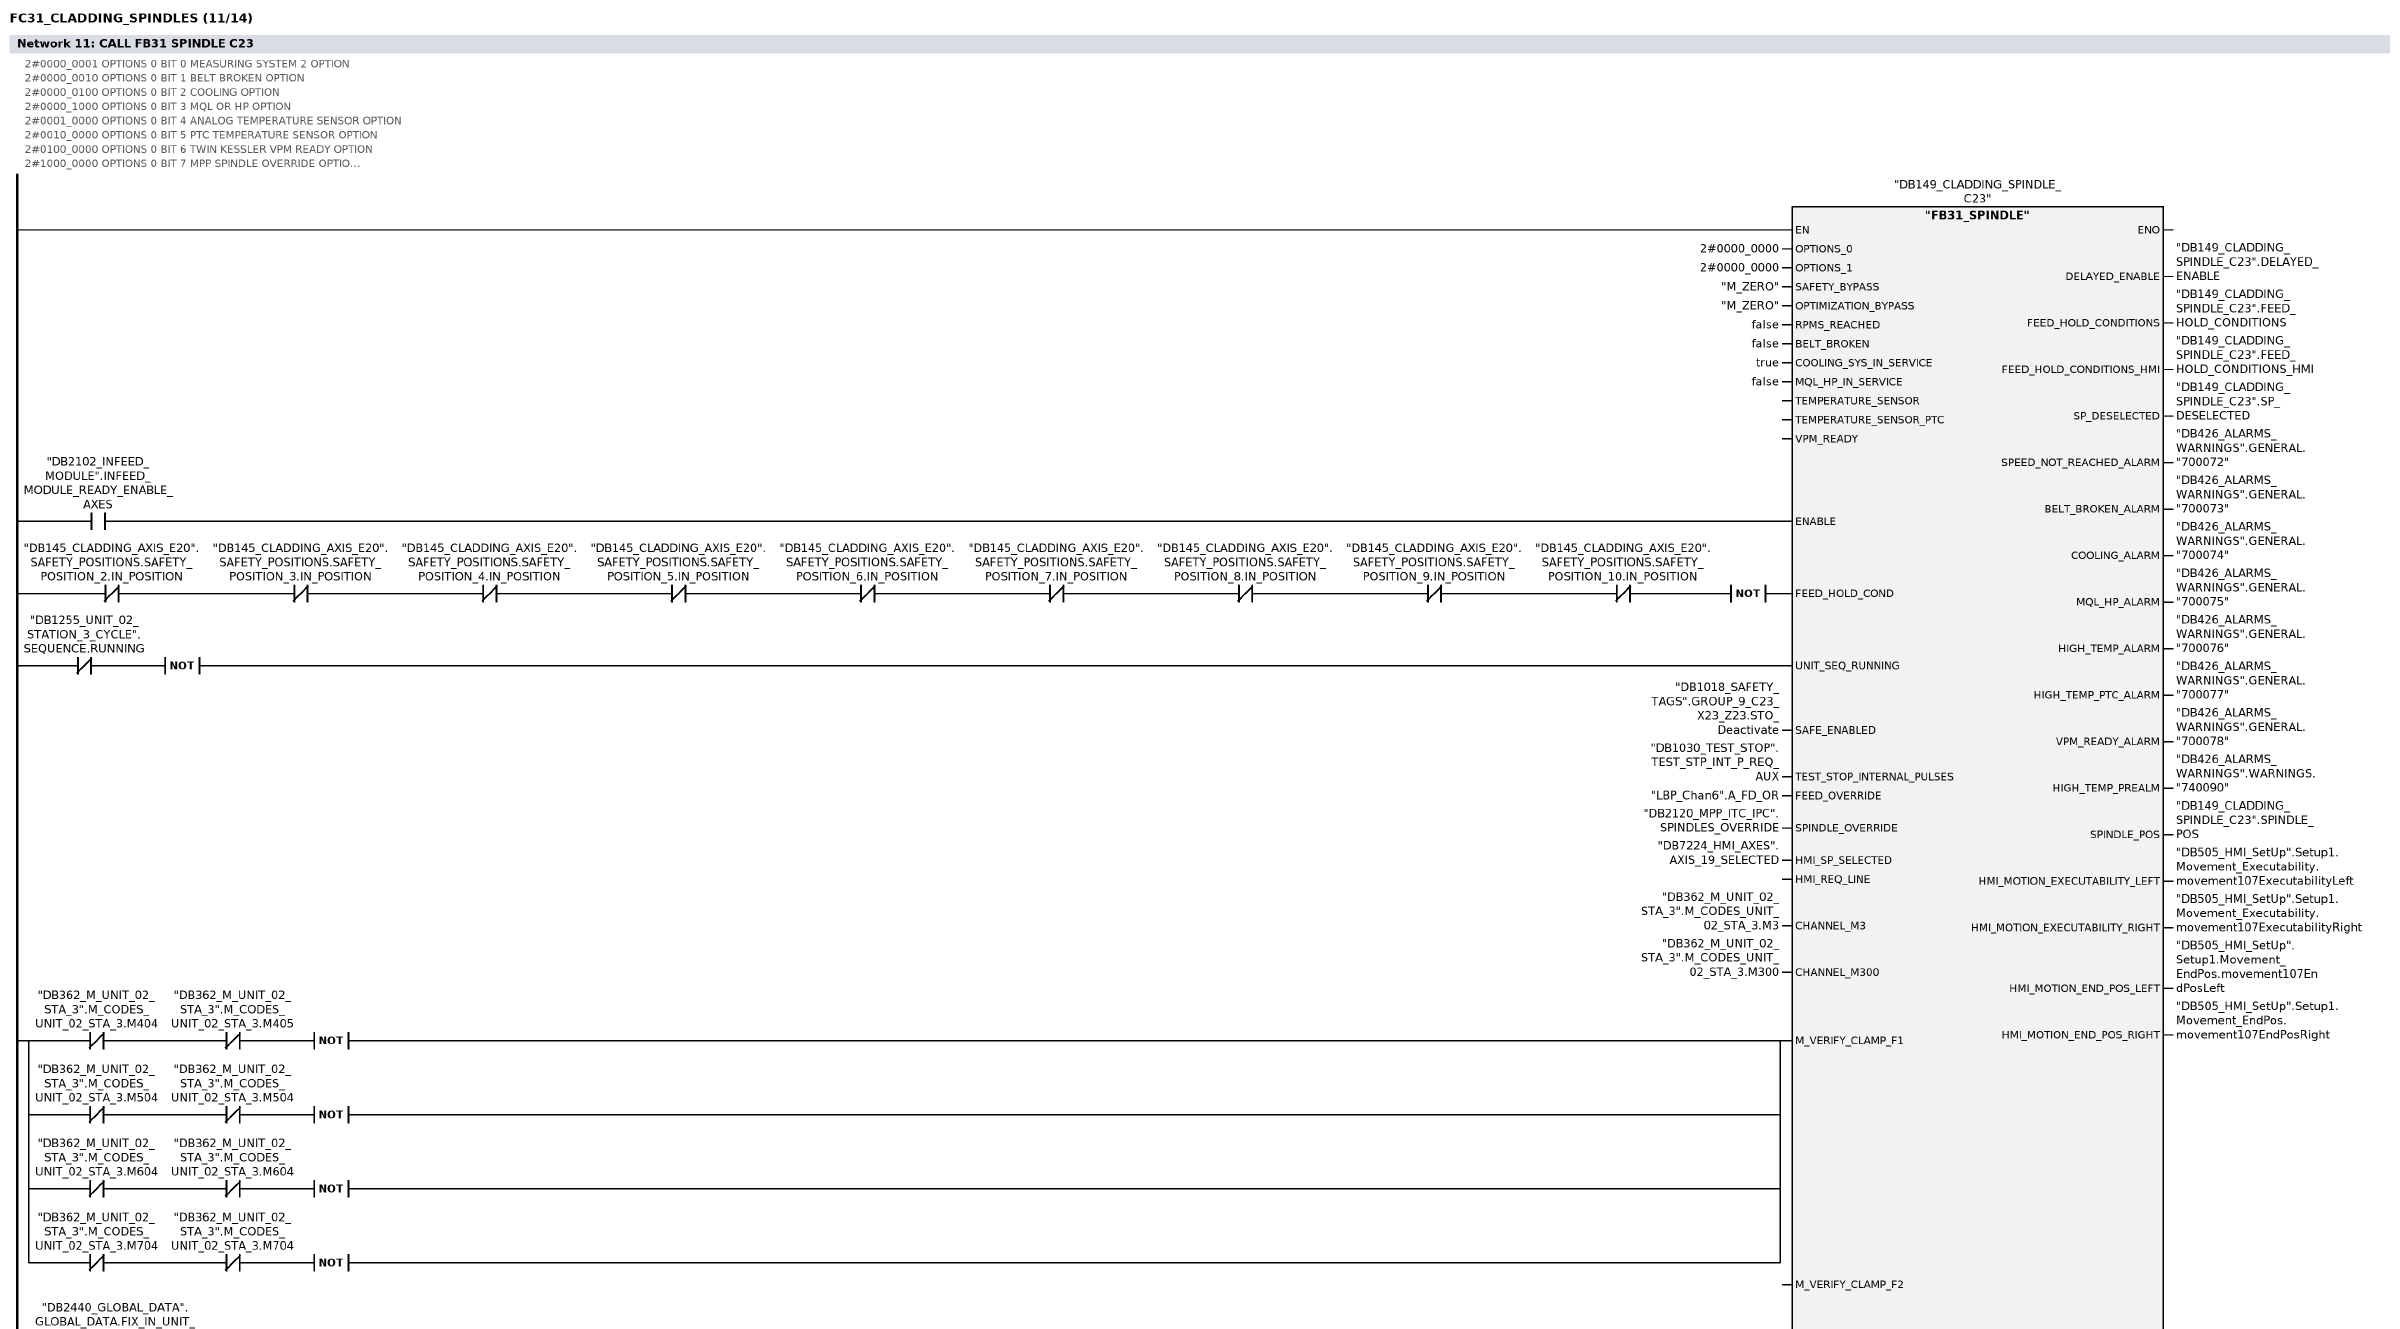
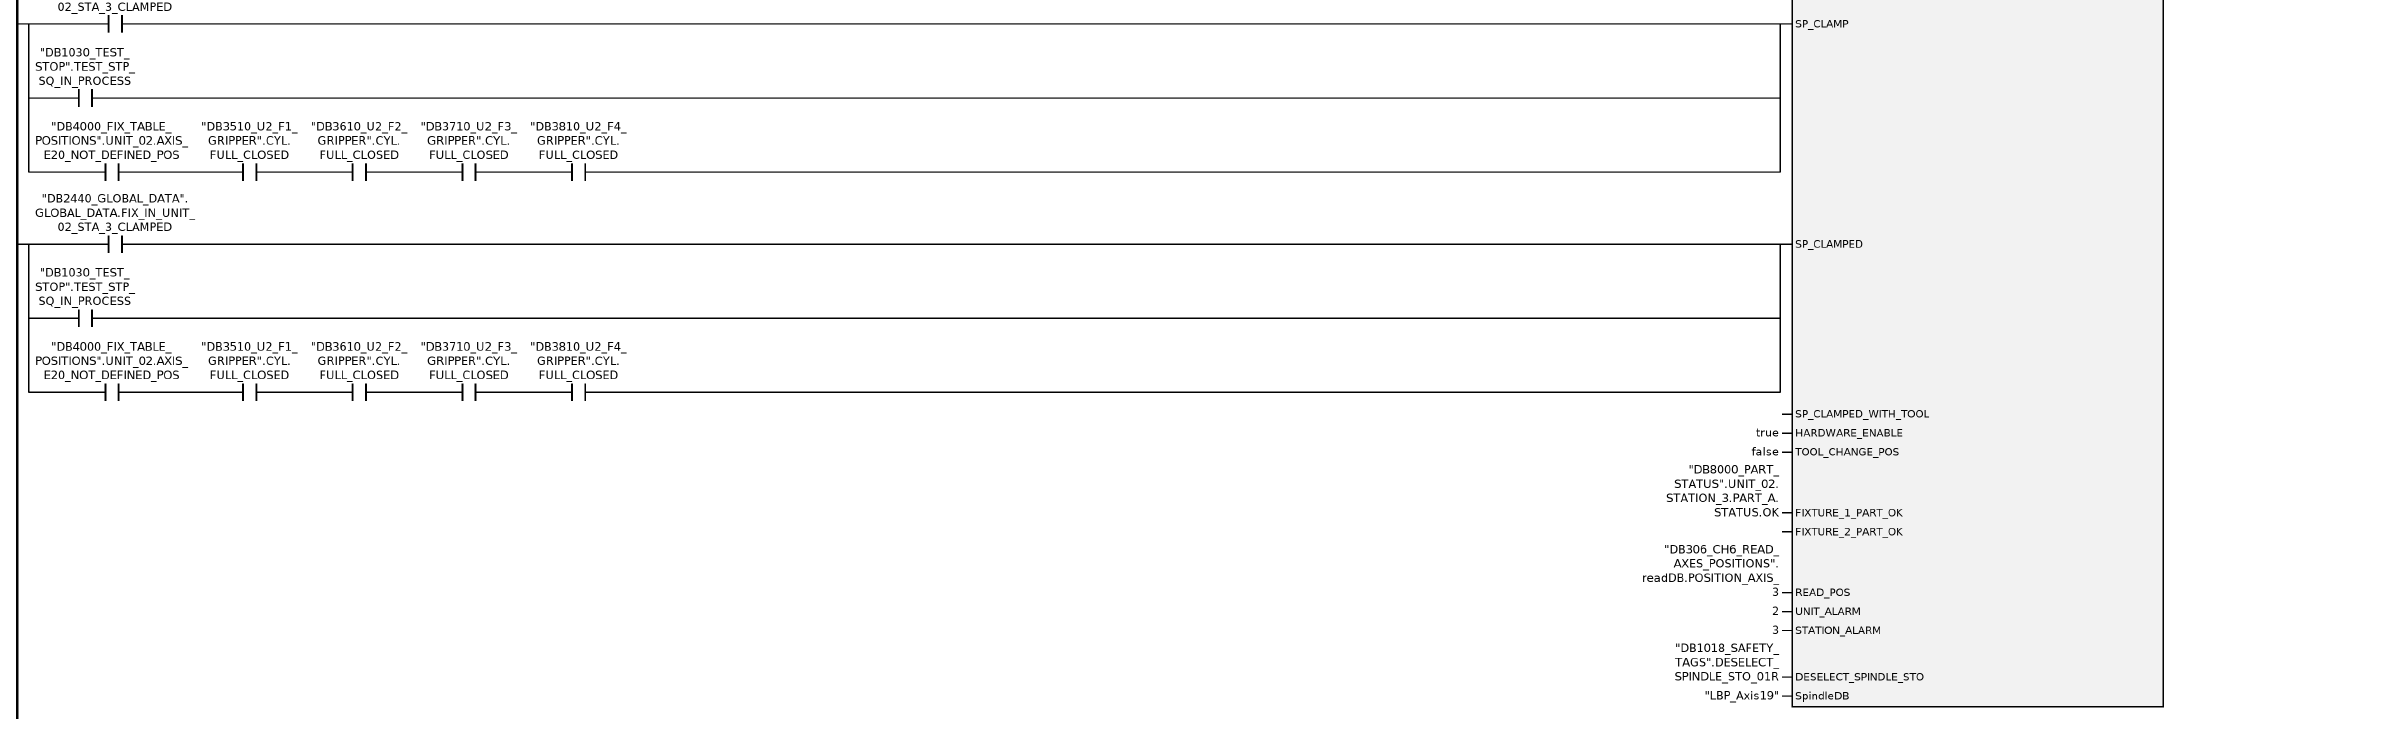
   RUNG wire#powerrail
      "DB149_CLADDING_SPINDLE_C23"(ENABLE := wire#w1, FEED_HOLD_COND := wire#w2, UNIT_SEQ_RUNNING := wire#w3, M_VERIFY_CLAMP_F1 := wire#w4, SP_CLAMP := wire#w5, SP_CLAMPED := wire#w6, OPTIONS_0 := 2#0000_0000, OPTIONS_1 := 2#0000_0000, SAFETY_BYPASS := "M_ZERO", OPTIMIZATION_BYPASS := "M_ZERO", RPMS_REACHED := false, BELT_BROKEN := false, COOLING_SYS_IN_SERVICE := true, MQL_HP_IN_SERVICE := false, TEMPERATURE_SENSOR :=, TEMPERATURE_SENSOR_PTC :=, VPM_READY :=, SAFE_ENABLED := "DB1018_SAFETY_TAGS".GROUP_9_C23_X23_Z23.STO_Deactivate, TEST_STOP_INTERNAL_PULSES := "DB1030_TEST_STOP".TEST_STP_INT_P_REQ_AUX, FEED_OVERRIDE := "LBP_Chan6".A_FD_OR, SPINDLE_OVERRIDE := "DB2120_MPP_ITC_IPC".SPINDLES_OVERRIDE, HMI_SP_SELECTED := "DB7224_HMI_AXES".AXIS_19_SELECTED, HMI_REQ_LINE :=, CHANNEL_M3 := "DB362_M_UNIT_02_STA_3".M_CODES_UNIT_02_STA_3.M3, CHANNEL_M300 := "DB362_M_UNIT_02_STA_3".M_CODES_UNIT_02_STA_3.M300, M_VERIFY_CLAMP_F2 :=, SP_CLAMPED_WITH_TOOL :=, HARDWARE_ENABLE := true, TOOL_CHANGE_POS := false, FIXTURE_1_PART_OK := "DB8000_PART_STATUS".UNIT_02.STATION_3.PART_A.STATUS.OK, FIXTURE_2_PART_OK :=, READ_POS := "DB306_CH6_READ_AXES_POSITIONS".readDB.POSITION_AXIS_3, UNIT_ALARM := 2, STATION_ALARM := 3, DESELECT_SPINDLE_STO := "DB1018_SAFETY_TAGS".DESELECT_SPINDLE_STO_01R, SpindleDB := "LBP_Axis19", DELAYED_ENABLE => "DB149_CLADDING_SPINDLE_C23".DELAYED_ENABLE, FEED_HOLD_CONDITIONS => "DB149_CLADDING_SPINDLE_C23".FEED_HOLD_CONDITIONS, FEED_HOLD_CONDITIONS_HMI => "DB149_CLADDING_SPINDLE_C23".FEED_HOLD_CONDITIONS_HMI, SP_DESELECTED => "DB149_CLADDING_SPINDLE_C23".SP_DESELECTED, SPEED_NOT_REACHED_ALARM => "DB426_ALARMS_WARNINGS".GENERAL."700072", BELT_BROKEN_ALARM => "DB426_ALARMS_WARNINGS".GENERAL."700073", COOLING_ALARM => "DB426_ALARMS_WARNINGS".GENERAL."700074", MQL_HP_ALARM => "DB426_ALARMS_WARNINGS".GENERAL."700075", HIGH_TEMP_ALARM => "DB426_ALARMS_WARNINGS".GENERAL."700076", HIGH_TEMP_PTC_ALARM => "DB426_ALARMS_WARNINGS".GENERAL."700077", VPM_READY_ALARM => "DB426_ALARMS_WARNINGS".GENERAL."700078", HIGH_TEMP_PREALM => "DB426_ALARMS_WARNINGS".WARNINGS."740090", SPINDLE_POS => "DB149_CLADDING_SPINDLE_C23".SPINDLE_POS, HMI_MOTION_EXECUTABILITY_LEFT => "DB505_HMI_SetUp".Setup1.Movement_Executability.movement107ExecutabilityLeft, HMI_MOTION_EXECUTABILITY_RIGHT => "DB505_HMI_SetUp".Setup1.Movement_Executability.movement107ExecutabilityRight, HMI_MOTION_END_POS_LEFT => "DB505_HMI_SetUp".Setup1.Movement_EndPos.movement107EndPosLeft, HMI_MOTION_END_POS_RIGHT => "DB505_HMI_SetUp".Setup1.Movement_EndPos.movement107EndPosRight)
   END_RUNG
   RUNG wire#powerrail
      Contact( "DB2102_INFEED_MODULE".INFEED_MODULE_READY_ENABLE_AXES )
   END_RUNG wire#w1
   RUNG wire#powerrail
      I_Contact( "DB145_CLADDING_AXIS_E20".SAFETY_POSITIONS.SAFETY_POSITION_2.IN_POSITION )
      I_Contact( "DB145_CLADDING_AXIS_E20".SAFETY_POSITIONS.SAFETY_POSITION_3.IN_POSITION )
      I_Contact( "DB145_CLADDING_AXIS_E20".SAFETY_POSITIONS.SAFETY_POSITION_4.IN_POSITION )
      I_Contact( "DB145_CLADDING_AXIS_E20".SAFETY_POSITIONS.SAFETY_POSITION_5.IN_POSITION )
      I_Contact( "DB145_CLADDING_AXIS_E20".SAFETY_POSITIONS.SAFETY_POSITION_6.IN_POSITION )
      I_Contact( "DB145_CLADDING_AXIS_E20".SAFETY_POSITIONS.SAFETY_POSITION_7.IN_POSITION )
      I_Contact( "DB145_CLADDING_AXIS_E20".SAFETY_POSITIONS.SAFETY_POSITION_8.IN_POSITION )
      I_Contact( "DB145_CLADDING_AXIS_E20".SAFETY_POSITIONS.SAFETY_POSITION_9.IN_POSITION )
      I_Contact( "DB145_CLADDING_AXIS_E20".SAFETY_POSITIONS.SAFETY_POSITION_10.IN_POSITION )
      Not()
   END_RUNG wire#w2
   RUNG wire#powerrail
      I_Contact( "DB1255_UNIT_02_STATION_3_CYCLE".SEQUENCE.RUNNING )
      Not()
   END_RUNG wire#w3
   RUNG wire#powerrail
      I_Contact( "DB362_M_UNIT_02_STA_3".M_CODES_UNIT_02_STA_3.M404 )
      I_Contact( "DB362_M_UNIT_02_STA_3".M_CODES_UNIT_02_STA_3.M405 )
      Not()
   END_RUNG wire#w4
   RUNG wire#powerrail
      I_Contact( "DB362_M_UNIT_02_STA_3".M_CODES_UNIT_02_STA_3.M504 )
      I_Contact( "DB362_M_UNIT_02_STA_3".M_CODES_UNIT_02_STA_3.M504 )
      Not()
   END_RUNG wire#w4
   RUNG wire#powerrail
      I_Contact( "DB362_M_UNIT_02_STA_3".M_CODES_UNIT_02_STA_3.M604 )
      I_Contact( "DB362_M_UNIT_02_STA_3".M_CODES_UNIT_02_STA_3.M604 )
      Not()
   END_RUNG wire#w4
   RUNG wire#powerrail
      I_Contact( "DB362_M_UNIT_02_STA_3".M_CODES_UNIT_02_STA_3.M704 )
      I_Contact( "DB362_M_UNIT_02_STA_3".M_CODES_UNIT_02_STA_3.M704 )
      Not()
   END_RUNG wire#w4
   RUNG wire#powerrail
      Contact( "DB2440_GLOBAL_DATA".GLOBAL_DATA.FIX_IN_UNIT_02_STA_3_CLAMPED )
   END_RUNG wire#w5
   RUNG wire#powerrail
      Contact( "DB1030_TEST_STOP".TEST_STP_SQ_IN_PROCESS )
   END_RUNG wire#w5
   RUNG wire#powerrail
      Contact( "DB4000_FIX_TABLE_POSITIONS".UNIT_02.AXIS_E20_NOT_DEFINED_POS )
      Contact( "DB3510_U2_F1_GRIPPER".CYL.FULL_CLOSED )
      Contact( "DB3610_U2_F2_GRIPPER".CYL.FULL_CLOSED )
      Contact( "DB3710_U2_F3_GRIPPER".CYL.FULL_CLOSED )
      Contact( "DB3810_U2_F4_GRIPPER".CYL.FULL_CLOSED )
   END_RUNG wire#w5
   RUNG wire#powerrail
      Contact( "DB2440_GLOBAL_DATA".GLOBAL_DATA.FIX_IN_UNIT_02_STA_3_CLAMPED )
   END_RUNG wire#w6
   RUNG wire#powerrail
      Contact( "DB1030_TEST_STOP".TEST_STP_SQ_IN_PROCESS )
   END_RUNG wire#w6
   RUNG wire#powerrail
      Contact( "DB4000_FIX_TABLE_POSITIONS".UNIT_02.AXIS_E20_NOT_DEFINED_POS )
      Contact( "DB3510_U2_F1_GRIPPER".CYL.FULL_CLOSED )
      Contact( "DB3610_U2_F2_GRIPPER".CYL.FULL_CLOSED )
      Contact( "DB3710_U2_F3_GRIPPER".CYL.FULL_CLOSED )
      Contact( "DB3810_U2_F4_GRIPPER".CYL.FULL_CLOSED )
   END_RUNG wire#w6
   // the same network as SCL:
   "DB149_CLADDING_SPINDLE_C23"(OPTIONS_0 := 2#0000_0000,   // "FB31_SPINDLE"
                           OPTIONS_1 := 2#0000_0000,
                           SAFETY_BYPASS := "M_ZERO",
                           OPTIMIZATION_BYPASS := "M_ZERO",
                           RPMS_REACHED := false,
                           BELT_BROKEN := false,
                           COOLING_SYS_IN_SERVICE := true,
                           MQL_HP_IN_SERVICE := false,
                           ENABLE := "DB2102_INFEED_MODULE".INFEED_MODULE_READY_ENABLE_AXES,
                           FEED_HOLD_COND := NOT (NOT "DB145_CLADDING_AXIS_E20".SAFETY_POSITIONS.SAFETY_POSITION_2.IN_POSITION AND NOT "DB145_CLADDING_AXIS_E20".SAFETY_POSITIONS.SAFETY_POSITION_3.IN_POSITION AND NOT "DB145_CLADDING_AXIS_E20".SAFETY_POSITIONS.SAFETY_POSITION_4.IN_POSITION AND NOT "DB145_CLADDING_AXIS_E20".SAFETY_POSITIONS.SAFETY_POSITION_5.IN_POSITION AND NOT "DB145_CLADDING_AXIS_E20".SAFETY_POSITIONS.SAFETY_POSITION_6.IN_POSITION AND NOT "DB145_CLADDING_AXIS_E20".SAFETY_POSITIONS.SAFETY_POSITION_7.IN_POSITION AND NOT "DB145_CLADDING_AXIS_E20".SAFETY_POSITIONS.SAFETY_POSITION_8.IN_POSITION AND NOT "DB145_CLADDING_AXIS_E20".SAFETY_POSITIONS.SAFETY_POSITION_9.IN_POSITION AND NOT "DB145_CLADDING_AXIS_E20".SAFETY_POSITIONS.SAFETY_POSITION_10.IN_POSITION),
                           UNIT_SEQ_RUNNING := NOT (NOT "DB1255_UNIT_02_STATION_3_CYCLE".SEQUENCE.RUNNING),
                           SAFE_ENABLED := "DB1018_SAFETY_TAGS".GROUP_9_C23_X23_Z23.STO_Deactivate,
                           TEST_STOP_INTERNAL_PULSES := "DB1030_TEST_STOP".TEST_STP_INT_P_REQ_AUX,
                           FEED_OVERRIDE := "LBP_Chan6".A_FD_OR,
                           SPINDLE_OVERRIDE := "DB2120_MPP_ITC_IPC".SPINDLES_OVERRIDE,
                           HMI_SP_SELECTED := "DB7224_HMI_AXES".AXIS_19_SELECTED,
                           CHANNEL_M3 := "DB362_M_UNIT_02_STA_3".M_CODES_UNIT_02_STA_3.M3,
                           CHANNEL_M300 := "DB362_M_UNIT_02_STA_3".M_CODES_UNIT_02_STA_3.M300,
                           M_VERIFY_CLAMP_F1 := NOT (NOT "DB362_M_UNIT_02_STA_3".M_CODES_UNIT_02_STA_3.M404 AND NOT "DB362_M_UNIT_02_STA_3".M_CODES_UNIT_02_STA_3.M405) OR NOT (NOT "DB362_M_UNIT_02_STA_3".M_CODES_UNIT_02_STA_3.M504 AND NOT "DB362_M_UNIT_02_STA_3".M_CODES_UNIT_02_STA_3.M504) OR NOT (NOT "DB362_M_UNIT_02_STA_3".M_CODES_UNIT_02_STA_3.M604 AND NOT "DB362_M_UNIT_02_STA_3".M_CODES_UNIT_02_STA_3.M604) OR NOT (NOT "DB362_M_UNIT_02_STA_3".M_CODES_UNIT_02_STA_3.M704 AND NOT "DB362_M_UNIT_02_STA_3".M_CODES_UNIT_02_STA_3.M704),
                           SP_CLAMP := "DB2440_GLOBAL_DATA".GLOBAL_DATA.FIX_IN_UNIT_02_STA_3_CLAMPED OR "DB1030_TEST_STOP".TEST_STP_SQ_IN_PROCESS OR ("DB4000_FIX_TABLE_POSITIONS".UNIT_02.AXIS_E20_NOT_DEFINED_POS AND "DB3510_U2_F1_GRIPPER".CYL.FULL_CLOSED AND "DB3610_U2_F2_GRIPPER".CYL.FULL_CLOSED AND "DB3710_U2_F3_GRIPPER".CYL.FULL_CLOSED AND "DB3810_U2_F4_GRIPPER".CYL.FULL_CLOSED),
                           SP_CLAMPED := "DB2440_GLOBAL_DATA".GLOBAL_DATA.FIX_IN_UNIT_02_STA_3_CLAMPED OR "DB1030_TEST_STOP".TEST_STP_SQ_IN_PROCESS OR ("DB4000_FIX_TABLE_POSITIONS".UNIT_02.AXIS_E20_NOT_DEFINED_POS AND "DB3510_U2_F1_GRIPPER".CYL.FULL_CLOSED AND "DB3610_U2_F2_GRIPPER".CYL.FULL_CLOSED AND "DB3710_U2_F3_GRIPPER".CYL.FULL_CLOSED AND "DB3810_U2_F4_GRIPPER".CYL.FULL_CLOSED),
                           HARDWARE_ENABLE := true,
                           TOOL_CHANGE_POS := false,
                           FIXTURE_1_PART_OK := "DB8000_PART_STATUS".UNIT_02.STATION_3.PART_A.STATUS.OK,
                           READ_POS := "DB306_CH6_READ_AXES_POSITIONS".readDB.POSITION_AXIS_3,
                           UNIT_ALARM := 2,
                           STATION_ALARM := 3,
                           DESELECT_SPINDLE_STO := "DB1018_SAFETY_TAGS".DESELECT_SPINDLE_STO_01R,
                           SpindleDB := "LBP_Axis19",
                           DELAYED_ENABLE => "DB149_CLADDING_SPINDLE_C23".DELAYED_ENABLE,
                           FEED_HOLD_CONDITIONS => "DB149_CLADDING_SPINDLE_C23".FEED_HOLD_CONDITIONS,
                           FEED_HOLD_CONDITIONS_HMI => "DB149_CLADDING_SPINDLE_C23".FEED_HOLD_CONDITIONS_HMI,
                           SP_DESELECTED => "DB149_CLADDING_SPINDLE_C23".SP_DESELECTED,
                           SPEED_NOT_REACHED_ALARM => "DB426_ALARMS_WARNINGS".GENERAL."700072",
                           BELT_BROKEN_ALARM => "DB426_ALARMS_WARNINGS".GENERAL."700073",
                           COOLING_ALARM => "DB426_ALARMS_WARNINGS".GENERAL."700074",
                           MQL_HP_ALARM => "DB426_ALARMS_WARNINGS".GENERAL."700075",
                           HIGH_TEMP_ALARM => "DB426_ALARMS_WARNINGS".GENERAL."700076",
                           HIGH_TEMP_PTC_ALARM => "DB426_ALARMS_WARNINGS".GENERAL."700077",
                           VPM_READY_ALARM => "DB426_ALARMS_WARNINGS".GENERAL."700078",
                           HIGH_TEMP_PREALM => "DB426_ALARMS_WARNINGS".WARNINGS."740090",
                           SPINDLE_POS => "DB149_CLADDING_SPINDLE_C23".SPINDLE_POS,
                           HMI_MOTION_EXECUTABILITY_LEFT => "DB505_HMI_SetUp".Setup1.Movement_Executability.movement107ExecutabilityLeft,
                           HMI_MOTION_EXECUTABILITY_RIGHT => "DB505_HMI_SetUp".Setup1.Movement_Executability.movement107ExecutabilityRight,
                           HMI_MOTION_END_POS_LEFT => "DB505_HMI_SetUp".Setup1.Movement_EndPos.movement107EndPosLeft,
                           HMI_MOTION_END_POS_RIGHT => "DB505_HMI_SetUp".Setup1.Movement_EndPos.movement107EndPosRight);
END_REGION

REGION Network 12: SPINDLE C23 OPERATOR HELP
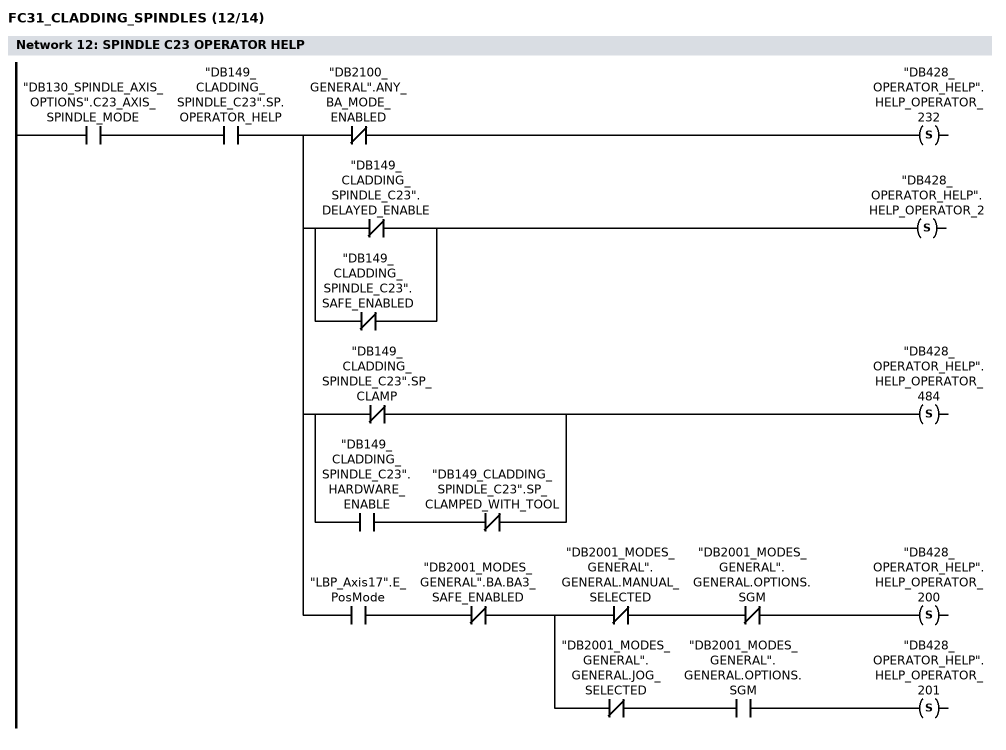
   RUNG wire#powerrail
      Contact( "DB130_SPINDLE_AXIS_OPTIONS".C23_AXIS_SPINDLE_MODE )
      Contact( "DB149_CLADDING_SPINDLE_C23".SP.OPERATOR_HELP )
      wire#w1
      I_Contact( "DB2100_GENERAL".ANY_BA_MODE_ENABLED )
      S_Coil( "DB428_OPERATOR_HELP".HELP_OPERATOR_232 )
   END_RUNG
   RUNG wire#w1
      I_Contact( "DB149_CLADDING_SPINDLE_C23".DELAYED_ENABLE )
      wire#w2
      S_Coil( "DB428_OPERATOR_HELP".HELP_OPERATOR_2 )
   END_RUNG
   RUNG wire#w1
      I_Contact( "DB149_CLADDING_SPINDLE_C23".SAFE_ENABLED )
   END_RUNG wire#w2
   RUNG wire#w1
      I_Contact( "DB149_CLADDING_SPINDLE_C23".SP_CLAMP )
      wire#w3
      S_Coil( "DB428_OPERATOR_HELP".HELP_OPERATOR_484 )
   END_RUNG
   RUNG wire#w1
      Contact( "DB149_CLADDING_SPINDLE_C23".HARDWARE_ENABLE )
      I_Contact( "DB149_CLADDING_SPINDLE_C23".SP_CLAMPED_WITH_TOOL )
   END_RUNG wire#w3
   RUNG wire#w1
      Contact( "LBP_Axis17".E_PosMode )
      I_Contact( "DB2001_MODES_GENERAL".BA.BA3_SAFE_ENABLED )
      wire#w4
      I_Contact( "DB2001_MODES_GENERAL".GENERAL.MANUAL_SELECTED )
      I_Contact( "DB2001_MODES_GENERAL".GENERAL.OPTIONS.SGM )
      S_Coil( "DB428_OPERATOR_HELP".HELP_OPERATOR_200 )
   END_RUNG
   RUNG wire#w4
      I_Contact( "DB2001_MODES_GENERAL".GENERAL.JOG_SELECTED )
      Contact( "DB2001_MODES_GENERAL".GENERAL.OPTIONS.SGM )
      S_Coil( "DB428_OPERATOR_HELP".HELP_OPERATOR_201 )
   END_RUNG
   // the same network as SCL:
   #_w1 := "DB130_SPINDLE_AXIS_OPTIONS".C23_AXIS_SPINDLE_MODE AND "DB149_CLADDING_SPINDLE_C23".SP.OPERATOR_HELP;
   IF #_w1 AND NOT "DB2100_GENERAL".ANY_BA_MODE_ENABLED THEN
       "DB428_OPERATOR_HELP".HELP_OPERATOR_232 := TRUE;
   END_IF;
   IF #_w1 AND (NOT "DB149_CLADDING_SPINDLE_C23".DELAYED_ENABLE OR NOT "DB149_CLADDING_SPINDLE_C23".SAFE_ENABLED) THEN
       "DB428_OPERATOR_HELP".HELP_OPERATOR_2 := TRUE;
   END_IF;
   IF #_w1 AND (NOT "DB149_CLADDING_SPINDLE_C23".SP_CLAMP OR ("DB149_CLADDING_SPINDLE_C23".HARDWARE_ENABLE AND NOT "DB149_CLADDING_SPINDLE_C23".SP_CLAMPED_WITH_TOOL)) THEN
       "DB428_OPERATOR_HELP".HELP_OPERATOR_484 := TRUE;
   END_IF;
   #_w2 := #_w1 AND "LBP_Axis17".E_PosMode AND NOT "DB2001_MODES_GENERAL".BA.BA3_SAFE_ENABLED;
   IF #_w2 AND NOT "DB2001_MODES_GENERAL".GENERAL.MANUAL_SELECTED AND NOT "DB2001_MODES_GENERAL".GENERAL.OPTIONS.SGM THEN
       "DB428_OPERATOR_HELP".HELP_OPERATOR_200 := TRUE;
   END_IF;
   IF #_w2 AND NOT "DB2001_MODES_GENERAL".GENERAL.JOG_SELECTED AND "DB2001_MODES_GENERAL".GENERAL.OPTIONS.SGM THEN
       "DB428_OPERATOR_HELP".HELP_OPERATOR_201 := TRUE;
   END_IF;
END_REGION

